// TIA Portal project "Simulate_HMI_FactoryIO_16" (V14)
// Vorlageprojekt für das Buch mit Zielsystem S7-1200

(* hardware
DEVICE "S7-1200-Station_1"  S7-1200 Station
   slot 0: "Baugruppenträger_0"  Rack  V1.0
   slot 1: "PLC_1"  CPU 1211C DC/DC/DC  6ES7 211-1AE40-0XB0  V4.1
DEVICE "HMI_1"  KTP1200 Basic PN
   slot 0: "KTP1200 Basic PN"  KTP1200 Basic PN  6AV2 123-2MB03-0AX0  14.0.1.0
   slot 1: "HMI_RT_1"  KTP1200 Basic PN  6AV2 123-2MB03-0AX0  14.0.1.0
   slot 5: "HMI_1.IE_CP_1"  PROFINET Interface  14.0.1.0
      slot 1: "PROFINET Interface_1"  PROFINET Interface
         slot 1: "Port_1"  Port
*)

// ===== PLC "PLC_1"  CPU 1211C DC/DC/DC =====

VAR_GLOBAL   // PLC tag table "Modes"
   "B_Pharmacy_ChooseRoom" AT %M0.1 : Bool;
   "B_Pharmacy_Go" AT %M0.2 : Bool;
   "B_Pharmacy_Room1" AT %MW2 : Int;
   "B_Pharmacy_Room2" AT %MW4 : Int;
   "B_Pharmacy_Room3" AT %MW6 : Int;
   "B_Pharmacy_Start" AT %M0.0 : Bool;
   "B_R1_Continue" AT %M20.2 : Bool;
   "B_R1_Return" AT %M20.3 : Bool;
   "B_R2_Continue" AT %M20.4 : Bool;
   "B_R2_Return" AT %M20.5 : Bool;
   "M_A_0_L2-L1_1" AT %M32.5 : Bool;
   "M_A_0_L2-L1_1_Trig" AT %M33.5 : Bool;
   "M_A_0_L2-L1_2" AT %M32.6 : Bool;
   "M_A_0_L2-L1_3" AT %M32.7 : Bool;
   "M_A_0_L2-L1_3_Trig" AT %M33.6 : Bool;
   "M_A_0_L2-L1_4" AT %M33.0 : Bool;
   "M_A_0_L2-L1_5" AT %M33.1 : Bool;
   "M_A_1to2_L1-L1_1" AT %M12.5 : Bool;
   "M_A_1to2_L1-L1_1_Trig" AT %M13.0 : Bool;
   "M_A_1to2_L1-L1_2" AT %M12.6 : Bool;
   "M_A_1to2_L1-L1_3" AT %M12.7 : Bool;
   "M_A_1to2_L1-L1_2_Trig" AT %M13.1 : Bool;
   "M_A_1to2_L1-L1_4" AT %M13.2 : Bool;
   "M_A_1to2_L1-L3_1" AT %M13.3 : Bool;
   "M_A_1to2_L1-L3_1_Trig" AT %M13.4 : Bool;
   "M_A_1to2_L1-L3_2" AT %M13.5 : Bool;
   "M_A_1to2_L1-L3_3" AT %M13.6 : Bool;
   "M_A_1to2_L1-L3_2_Trig" AT %M14.2 : Bool;
   "M_A_1to2_L1-L3_4" AT %M14.0 : Bool;
   "M_A_1to2_L1-L3_4_Trig" AT %M13.7 : Bool;
   "M_A_1to2_L1-L3_5" AT %M14.1 : Bool;
   "M_A_1to2_L2-L2_1" AT %M25.5 : Bool;
   "M_A_1to2_L2-L2_1_Trig" AT %M26.1 : Bool;
   "M_A_1to2_L2-L2_2" AT %M25.6 : Bool;
   "M_A_1to2_L2-L2_3" AT %M25.7 : Bool;
   "M_A_1to2_L2-L2_2_Trig" AT %M26.2 : Bool;
   "M_A_1to2_L2-L2_4" AT %M26.0 : Bool;
   "M_A_1to2_L2-L3_1" AT %M28.2 : Bool;
   "M_A_1to2_L2-L3_1_Trig" AT %M28.3 : Bool;
   "M_A_1to2_L2-L3_2" AT %M28.4 : Bool;
   "M_A_1to2_L2-L3_3" AT %M28.5 : Bool;
   "M_A_1to2_L2-L3_3_Trig" AT %M28.6 : Bool;
   "M_A_1to2_L2-L3_4" AT %M28.7 : Bool;
   "M_A_1to2_L2-L3_5" AT %M29.0 : Bool;
   "M_A_1to2_L4-L2_1" AT %M31.6 : Bool;
   "M_A_1to2_L4-L2_1_Trig" AT %M31.7 : Bool;
   "M_A_1to2_L4-L2_2" AT %M32.0 : Bool;
   "M_A_1to2_L4-L2_3" AT %M32.1 : Bool;
   "M_A_1to2_L4-L2_3_Trig" AT %M32.2 : Bool;
   "M_A_1to2_L4-L2_4" AT %M32.3 : Bool;
   "M_A_1to2_L4-L2_5" AT %M32.4 : Bool;
   "M_A_2to3_L1-L2_F1" AT %M14.3 : Bool;
   "M_A_2to3_L1-L2_F1_Trig" AT %M15.1 : Bool;
   "M_A_2to3_L1-L2_F2" AT %M14.4 : Bool;
   "M_A_2to3_L1-L2_F3" AT %M14.5 : Bool;
   "M_A_2to3_L1-L2_F2_Trig" AT %M15.2 : Bool;
   "M_A_2to3_L1-L2_F4" AT %M14.6 : Bool;
   "M_A_2to3_L2-L2_B1" AT %M24.0 : Bool;
   "M_A_2to3_L2-L2_B1_Trig" AT %M24.4 : Bool;
   "M_A_2to3_L2-L2_B2" AT %M24.1 : Bool;
   "M_A_2to3_L2-L2_B3" AT %M24.2 : Bool;
   "M_A_2to3_L2-L2_B3_Trig" AT %M24.5 : Bool;
   "M_A_2to3_L2-L2_B4" AT %M24.3 : Bool;
   "M_A_2to3_L2-L2_B5" AT %M24.6 : Bool;
   "M_A_2to4_L1-L2_F1" AT %M15.5 : Bool;
   "M_A_2to4_L1-L2_F1_Trig" AT %M15.6 : Bool;
   "M_A_2to4_L1-L2_F2" AT %M15.7 : Bool;
   "M_A_2to4_L1-L2_F3" AT %M16.0 : Bool;
   "M_A_2to4_L1-L2_F2_Trig" AT %M16.1 : Bool;
   "M_A_2to4_L1-L2_F4" AT %M16.2 : Bool;
   "M_A_2to4_L2-L2_B1" AT %M30.1 : Bool;
   "M_A_2to4_L2-L2_B1_Trig" AT %M30.2 : Bool;
   "M_A_2to4_L2-L2_B2" AT %M30.3 : Bool;
   "M_A_2to4_L2-L2_B3" AT %M30.4 : Bool;
   "M_A_2to4_L2-L2_B3_Trig" AT %M30.5 : Bool;
   "M_A_2to4_L2-L2_B4" AT %M30.6 : Bool;
   "M_A_2to4_L2-L2_B5" AT %M30.7 : Bool;
   "M_B_S0_1" AT %M27.7 : Bool;
   "M_B_S0_1_Trig" AT %M28.1 : Bool;
   "M_B_S0_2" AT %M28.0 : Bool;
   "M_B_S0_2_Trig1" AT %M33.2 : Bool;
   "M_B_S0_2_Trig2" AT %M33.3 : Bool;
   "M_B_S0_2_Trig3" AT %M33.4 : Bool;
   "M_B_S1-Cnv1_1" AT %M26.3 : Bool;
   "M_B_S1-Cnv1_1_Trig" AT %M26.4 : Bool;
   "M_B_S1-Cnv1_2" AT %M26.5 : Bool;
   "M_B_S1-Cnv1_2_Trig1" AT %M26.6 : Bool;
   "M_B_S1-Cnv1_2_Trig2" AT %M26.7 : Bool;
   "M_B_S2-1_1" AT %M24.7 : Bool;
   "M_B_S2-1_1_Trig" AT %M25.0 : Bool;
   "M_B_S2-1_2" AT %M25.1 : Bool;
   "M_B_S2-1_2_Trig1" AT %M25.2 : Bool;
   "M_B_S2-1_2_Trig2" AT %M25.3 : Bool;
   "M_B_S2-1_2_Trig3" AT %M25.4 : Bool;
   "M_B_S2-2_1" AT %M31.0 : Bool;
   "M_B_S2-2_1_Trig" AT %M31.1 : Bool;
   "M_B_S2-2_2" AT %M31.2 : Bool;
   "M_B_S2-2_2_Trig1" AT %M31.3 : Bool;
   "M_B_S2-2_2_Trig2" AT %M31.4 : Bool;
   "M_B_S2-2_2_Trig3" AT %M31.5 : Bool;
   "M_B2H_S3_1" AT %M23.2 : Bool;
   "M_B2H_S3_1_Trig" AT %M23.3 : Bool;
   "M_B2H_S3_2" AT %M23.4 : Bool;
   "M_B2H_S3_2_Trig1" AT %M23.5 : Bool;
   "M_B2H_S3_2_Trig2" AT %M23.6 : Bool;
   "M_B2H_S3_2_Trig3" AT %M23.7 : Bool;
   "M_B2H_S4_1" AT %M29.3 : Bool;
   "M_B2H_S4_1_Trig" AT %M29.4 : Bool;
   "M_B2H_S4_2" AT %M29.5 : Bool;
   "M_B2H_S4_2_Trig1" AT %M29.6 : Bool;
   "M_B2H_S4_2_Trig2" AT %M29.7 : Bool;
   "M_B2H_S4_2_Trig3" AT %M30.0 : Bool;
   "M_B2L_S3_1" AT %M20.6 : Bool;
   "M_B2L_S3_2" AT %M20.7 : Bool;
   "M_B2L_S3_2_Trig1" AT %M21.2 : Bool;
   "M_B2L_S3_2_Trig2" AT %M21.3 : Bool;
   "M_B2L_S4_1" AT %M21.0 : Bool;
   "M_B2L_S4_2" AT %M21.1 : Bool;
   "M_B2L_S4_2_Trig1" AT %M29.1 : Bool;
   "M_B2L_S4_2_Trig2" AT %M29.2 : Bool;
   "M_F_S0_1" AT %M1.1 : Bool;
   "M_F_S0_1_Trig" AT %M1.2 : Bool;
   "M_F_S0_2" AT %M1.3 : Bool;
   "M_F_S0_2_Trig1" AT %M1.4 : Bool;
   "M_F_S0_2_Trig2" AT %M8.0 : Bool;
   "M_F_S1_1" AT %M1.5 : Bool;
   "M_F_S1_1_Trig" AT %M1.6 : Bool;
   "M_F_S1_2" AT %M1.7 : Bool;
   "M_F_S1-Cnv1_2_Trig1" AT %M10.0 : Bool;
   "M_F_S1-Cnv1_2_Trig2" AT %M12.3 : Bool;
   "M_F_S1_2_Trig3" AT %M12.4 : Bool;
   "M_F_S2-1_1" AT %M10.1 : Bool;
   "M_F_S2-1_1_Trig" AT %M10.2 : Bool;
   "M_F_S2-1_2" AT %M10.3 : Bool;
   "M_F_S2-1_2_Trig1" AT %M10.4 : Bool;
   "M_F_S2-1_2_Trig2" AT %M14.7 : Bool;
   "M_F_S2-1_2_Trig3" AT %M15.0 : Bool;
   "M_F_S2-2_1" AT %M10.5 : Bool;
   "M_F_S2-2_1_Trig" AT %M10.6 : Bool;
   "M_F_S2-2_2" AT %M10.7 : Bool;
   "M_F_S2-2_2_Trig1" AT %M11.0 : Bool;
   "M_F_S2-2_2_Trig2" AT %M15.3 : Bool;
   "M_F_S2-2_2_Trig3" AT %M15.4 : Bool;
   "M_F2H_S3_1" AT %M8.1 : Bool;
   "M_F2H_S3_1_Trig" AT %M8.2 : Bool;
   "M_F2H_S3_2" AT %M8.3 : Bool;
   "M_F2H_S3_2_Trig1" AT %M8.4 : Bool;
   "M_F2H_S3_2_Trig2" AT %M8.5 : Bool;
   "M_F2H_S3_2_Trig3" AT %M8.6 : Bool;
   "M_F2H_S4_1" AT %M8.7 : Bool;
   "M_F2H_S4_1_Trig" AT %M9.0 : Bool;
   "M_F2H_S4_2" AT %M9.1 : Bool;
   "M_F2H_S4_2_Trig1" AT %M9.2 : Bool;
   "M_F2H_S4_2_Trig2" AT %M9.3 : Bool;
   "M_F2H_S4_2_Trig3" AT %M9.4 : Bool;
   "M_F2L_S3_1" AT %M9.5 : Bool;
   "M_F2L_S3_1_Trig" AT %M9.6 : Bool;
   "M_F2L_S3_2" AT %M9.7 : Bool;
   "M_F2L_S3_2_Trig" AT %M18.6 : Bool;
   "M_F2L_S4_1" AT %M19.6 : Bool;
   "M_F2L_S4_1_Trig" AT %M19.7 : Bool;
   "M_F2L_S4_2" AT %M20.0 : Bool;
   "M_F2L_S4_2_Trig" AT %M20.1 : Bool;
   "M_Pharmacy_ChooseRoom" AT %M0.6 : Bool;
   "M_Pharmacy_Go" AT %M0.7 : Bool;
   "M_Pharmacy_Go_Trig" AT %M1.0 : Bool;
   "M_Pharmacy_Start" AT %M0.4 : Bool;
   "M_Pharmacy_Start_Trig" AT %M0.5 : Bool;
   "M_Pharmacy_Wait" AT %M0.3 : Bool;
   "M_R1_ChooseRoom" AT %M17.2 : Bool;
   "M_R1_Go" AT %M17.3 : Bool;
   "M_R1_Go_Trig" AT %M17.4 : Bool;
   "M_R1_Start" AT %M17.5 : Bool;
   "M_R1_Start_Trig" AT %M17.6 : Bool;
   "M_R1_Wait" AT %M17.7 : Bool;
   "M_R2_ChooseRoom" AT %M18.0 : Bool;
   "M_R2_Go" AT %M18.1 : Bool;
   "M_R2_Go_Trig" AT %M18.2 : Bool;
   "M_R2_Start" AT %M18.3 : Bool;
   "M_R2_Start_Trig" AT %M18.4 : Bool;
   "M_R2_Wait" AT %M18.5 : Bool;
   "M_UD_0to1_B_1" AT %M27.0 : Bool;
   "M_UD_0to1_B_1_Trig" AT %M27.5 : Bool;
   "M_UD_0to1_B_2" AT %M27.1 : Bool;
   "M_UD_0to1_B_3" AT %M27.2 : Bool;
   "M_UD_0to1_B_3_Trig" AT %M27.6 : Bool;
   "M_UD_0to1_B_4" AT %M27.3 : Bool;
   "M_UD_0to1_B_5" AT %M27.4 : Bool;
   "M_UD_0to1_F_1" AT %M11.1 : Bool;
   "M_UD_0to1_F_1_Trig" AT %M11.2 : Bool;
   "M_UD_0to1_F_2" AT %M11.3 : Bool;
   "M_UD_0to1_F_2_Trig" AT %M11.4 : Bool;
   "M_UD_0to1_F_3" AT %M11.5 : Bool;
   "M_UD_0to1_F_3_Trig" AT %M11.6 : Bool;
   "M_UD_0to1_F_4" AT %M11.7 : Bool;
   "M_UD_0to1_F_4_Trig" AT %M12.0 : Bool;
   "M_UD_0to1_F_5" AT %M12.1 : Bool;
   "M_UD_3_B_1" AT %M21.4 : Bool;
   "M_UD_3_B_1_Trig" AT %M21.5 : Bool;
   "M_UD_3_B_2" AT %M21.6 : Bool;
   "M_UD_3_B_3" AT %M21.7 : Bool;
   "M_UD_3_B_3_Trig" AT %M22.0 : Bool;
   "M_UD_3_B_4" AT %M22.1 : Bool;
   "M_UD_3_B_5" AT %M22.2 : Bool;
   "M_UD_3_F_1" AT %M16.3 : Bool;
   "M_UD_3_F_1_Trig" AT %M17.0 : Bool;
   "M_UD_3_F_2" AT %M16.4 : Bool;
   "M_UD_3_F_3" AT %M16.5 : Bool;
   "M_UD_3_F_3_Trig" AT %M17.1 : Bool;
   "M_UD_3_F_4" AT %M16.6 : Bool;
   "M_UD_3_F_5" AT %M16.7 : Bool;
   "M_UD_4_B_1" AT %M22.3 : Bool;
   "M_UD_4_B_1_Trig" AT %M22.4 : Bool;
   "M_UD_4_B_2" AT %M22.5 : Bool;
   "M_UD_4_B_3" AT %M22.6 : Bool;
   "M_UD_4_B_3_Trig" AT %M22.7 : Bool;
   "M_UD_4_B_4" AT %M23.0 : Bool;
   "M_UD_4_B_5" AT %M23.1 : Bool;
   "M_UD_4_F_1" AT %M18.7 : Bool;
   "M_UD_4_F_1_Trig" AT %M19.0 : Bool;
   "M_UD_4_F_2" AT %M19.1 : Bool;
   "M_UD_4_F_3" AT %M19.2 : Bool;
   "M_UD_4_F_3_Trig" AT %M19.3 : Bool;
   "M_UD_4_F_4" AT %M19.4 : Bool;
   "M_UD_4_F_5" AT %M19.5 : Bool;
   "M_Elevator1_Trig1" AT %M33.7 : Bool;
   "M_UD_0to1_F_6" AT %M34.0 : Bool;
   "M_UD_3_F_6" AT %M34.1 : Bool;
   "M_UD_0to1_F_7" AT %M34.2 : Bool;
   "M_UD_3_F_7" AT %M34.3 : Bool;
   "M_Elevator3_Trig1" AT %M34.4 : Bool;
   "M_Elevator4_Trig1" AT %M34.5 : Bool;
   "M_UD_4_F_6" AT %M34.6 : Bool;
   "M_UD_4_F_7" AT %M34.7 : Bool;
   "M_Elevator3_Trig2" AT %M35.0 : Bool;
   "M_UD_3_B_6" AT %M35.1 : Bool;
   "M_UD_3_B_7" AT %M35.2 : Bool;
   "M_Elevator4_Trig2" AT %M35.3 : Bool;
   "M_UD_4_B_6" AT %M35.4 : Bool;
   "M_UD_4_B_7" AT %M35.5 : Bool;
   "M_B_S1-Cnv2_1" AT %M35.6 : Bool;
   "M_B_S1-Cnv2_1_Trig1" AT %M35.7 : Bool;
   "M_B_S1-Cnv2_2" AT %M36.0 : Bool;
   "M_B_S1-Cnv2_2_Trig1" AT %M36.1 : Bool;
   "M_B_S1-Cnv2_1_Trig2" AT %M36.2 : Bool;
   "M_B_S1-Cnv2_3" AT %M36.3 : Bool;
   "M_B_S1-Cnv2_3_Trig1" AT %M36.4 : Bool;
   "M_B_S1-Cnv2_3_Trig2" AT %M36.5 : Bool;
   "M_UD_0to1_B_6" AT %M36.6 : Bool;
   "M_UD_0to1_B_7" AT %M36.7 : Bool;
   "M_Elevator2_Trig1" AT %M37.0 : Bool;
   "M_A_0_L2-L1_2_Trig1" AT %M37.1 : Bool;
   "M_A_0_L2-L1_Trig" AT %M37.2 : Bool;
   "M_A_0_L2-L1_2_Trig2" AT %M37.3 : Bool;
   "F_0_1_1_Stt" AT %MW100 : Int;
   "F_1_1_1_Stt" AT %MW102 : Int;
   "F_2_1_1_Stt" AT %MW104 : Int;
   "F_2_2_1_Stt" AT %MW106 : Int;
   "B_0_1_1_Stt" AT %MW108 : Int;
   "B_1_1_1_Stt" AT %MW110 : Int;
   "B_2_1_1_Stt" AT %MW112 : Int;
   "B_2_2_1_Stt" AT %MW114 : Int;
   "2d_3_H_Stt" AT %MW116 : Int;
   "2d_3_H_Dir" AT %MW118 : Int;
   "2d_3_L_Stt" AT %MW120 : Int;
   "2d_3_L_Dir" AT %MW122 : Int;
   "2d_4_H_Stt" AT %MW124 : Int;
   "2d_4_H_Dir" AT %MW126 : Int;
   "2d_4_L_Stt" AT %MW128 : Int;
   "2d_4_L_Dir" AT %MW130 : Int;
   "av2_0to0_Stt" AT %MW132 : Int;
   "av2_0to0_Dir" AT %MW134 : Int;
   "av4_1to2_Stt" AT %MW136 : Word;
   "av4_1to2_Dir" AT %MW138 : Word;
   "av2_2to3_Stt" AT %MW140 : Int;
   "av2_2to3_Dir" AT %MW142 : Int;
   "av2_2to4_Stt" AT %MW144 : Int;
   "av2_2to4_Dir" AT %MW146 : Int;
   "ud_0to1_1_Stt" AT %MW148 : Int;
   "ud_0to1_1_Dir" AT %MW150 : Int;
   "ud_0to1_2_Stt" AT %MW152 : Int;
   "ud_0to1_2_Dir" AT %MW154 : Int;
   "ud_3_Stt" AT %MW156 : Int;
   "ud_3_Dir" AT %MW158 : Int;
   "ud_4_Stt" AT %MW160 : Int;
   "ud_4_Dir" AT %MW162 : Int;
   "av2_0to0_LS1" AT %M300.0 : Bool;
   "av2_0to0_LS2" AT %M300.1 : Bool;
   "av4_1to2_LS1" AT %M300.2 : Bool;
   "av4_1to2_LS2" AT %M300.3 : Bool;
   "av4_1to2_LS3" AT %M300.4 : Bool;
   "av4_1to2_LS4" AT %M300.5 : Bool;
   "av2_2to3_LS1" AT %M300.6 : Bool;
   "av2_2to3_LS2" AT %M300.7 : Bool;
   "av2_2to4_LS1" AT %M301.0 : Bool;
   "av2_2to4_LS2" AT %M301.1 : Bool;
   "ud_0to1_f_ls_H" AT %M301.2 : Bool;
   "ud_0to1_f_ls_L" AT %M301.3 : Bool;
   "ud_3_ls_H" AT %M301.6 : Bool;
   "ud_3_ls_L" AT %M301.7 : Bool;
   "ud_4_ls_H" AT %M302.0 : Bool;
   "ud_4_ls_L" AT %M302.1 : Bool;
   "ud_0to1_b_ls_H" AT %M301.4 : Bool;
   "ud_0to1_b_ls_L" AT %M301.5 : Bool;
   "M_B_S1-Cnv2_3_Trig3" AT %M37.4 : Bool;
   "box1_f_0_1_1" AT %MW164 : Int;
   "box2_f_0_1_1" AT %MW166 : Word;
   "box3_f_0_1_1" AT %MW168 : Word;
   "box1_f_1_1_1" AT %MW170 : Word;
   "box2_f_1_1_1" AT %MW172 : Word;
   "box3_f_1_1_1" AT %MW174 : Word;
   "box1_f_2_1_1" AT %MW176 : Word;
   "box2_f_2_1_1" AT %MW178 : Word;
   "box3_f_2_1_1" AT %MW180 : Word;
   "box1_f_2_2_1" AT %MW182 : Word;
   "box2_f_2_2_1" AT %MW184 : Word;
   "box3_f_2_2_1" AT %MW186 : Word;
   "box1_b_0_1_1" AT %MW188 : Word;
   "box2_b_0_1_1" AT %MW190 : Word;
   "box3_b_0_1_1" AT %MW192 : Word;
   "box1_b_1_1_1" AT %MW194 : Word;
   "box2_b_1_1_1" AT %MW196 : Word;
   "box3_b_1_1_1" AT %MW198 : Word;
   "box1_b_2_1_1" AT %MW200 : Word;
   "box2_b_2_1_1" AT %MW202 : Word;
   "box3_b_2_1_1" AT %MW204 : Word;
   "box1_b_2_2_1" AT %MW206 : Word;
   "box2_b_2_2_1" AT %MW208 : Word;
   "box3_b_2_2_1" AT %MW210 : Word;
   "box_av2_0to0" AT %MW212 : Word;
   "box_av4_1to2" AT %MW214 : Word;
   "box_av2_2to3" AT %MW216 : Word;
   "box_av2_2to4" AT %MW218 : Word;
   "box_ud2_0to1_f" AT %MW220 : Word;
   "box_ud2_0to1_b" AT %MW222 : Word;
   "box_ud_3" AT %MW224 : Word;
   "box_ud_4" AT %MW226 : Word;
   "box1_2d_3h" AT %MW228 : Word;
   "box2_2d_3h" AT %MW230 : Word;
   "box3_2d_3h" AT %MW232 : Word;
   "box1_2d_3l" AT %MW234 : Word;
   "box2_2d_3l" AT %MW236 : Word;
   "box3_2d_3l" AT %MW238 : Word;
   "box1_2d_4h" AT %MW240 : Word;
   "box2_2d_4h" AT %MW242 : Word;
   "box3_2d_4h" AT %MW244 : Word;
   "box1_2d_4l" AT %MW246 : Word;
   "box2_2d_4l" AT %MW248 : Word;
   "box3_2d_4l" AT %MW250 : Word;
   "M_R1_Cont_Trig" AT %M37.5 : Bool;
   "M_R1_Return_Trig" AT %M37.6 : Bool;
   "M_R2_Cont_Trig" AT %M37.7 : Bool;
   "M_R2_Return_Trig" AT %M38.0 : Bool;
   "M_A_1to2_L4-L1_1" AT %M38.1 : Bool;
   "M_A_1to2_L4-L1_1_Trig" AT %M38.2 : Bool;
   "M_A_1to2_L4-L1_2" AT %M38.3 : Bool;
   "M_A_1to2_L4-L1_3" AT %M38.4 : Bool;
   "M_A_1to2_L4-L1_3_Trig" AT %M38.5 : Bool;
   "M_A_1to2_L4-L1_4" AT %M38.6 : Bool;
   "M_A_1to2_L4-L1_5" AT %M38.7 : Bool;
   "box1_des1" AT %MW252 : Word;
   "box1_des2" AT %MW254 : Word;
   "box1_des3" AT %MW256 : Word;
   "box2_des1" AT %MW258 : Word;
   "box2_des2" AT %MW260 : Word;
   "box2_des3" AT %MW262 : Word;
   "box3_des1" AT %MW264 : Word;
   "box3_des2" AT %MW266 : Word;
   "box3_des3" AT %MW268 : Word;
   "box4_des1" AT %MW270 : Word;
   "box4_des2" AT %MW272 : Word;
   "box4_des3" AT %MW274 : Word;
   "box5_des1" AT %MW276 : Word;
   "box5_des2" AT %MW278 : Word;
   "box5_des3" AT %MW280 : Word;
   "Tag_1" AT %M500.0 : Bool;
   "R1_has_box" AT %M39.0 : Bool;
   "R2_has_box" AT %M39.1 : Bool;
END_VAR

VAR_GLOBAL   // PLC tag table "Hardware Input"
   "Elevator1_SS_Back" AT %I0.0 : Bool;
   "Elevator1_SS_Front" AT %I0.1 : Bool;
   "Elevator2_SS_Back" AT %I0.2 : Bool;
   "Elevator2_SS_Front" AT %I0.3 : Bool;
   "Elevator3_SS_Back" AT %I0.4 : Bool;
   "Elevator3_SS_Front" AT %I0.5 : Bool;
   "Elevator4_SS_Back" AT %I0.6 : Bool;
   "Elevator4_SS_Front" AT %I0.7 : Bool;
   "Cnv2_S3_H_VS1_Bool0" AT %I1.0 : Bool;
   "Cnv2_S3_H_VS1_Bool1" AT %I1.1 : Bool;
   "Cnv2_S3_H_VS1_Bool2" AT %I1.2 : Bool;
   "Cnv2_S3_H_VS2_Bool0" AT %I1.3 : Bool;
   "Cnv2_S3_H_VS2_Bool1" AT %I1.4 : Bool;
   "Cnv2_S3_H_VS2_Bool2" AT %I1.5 : Bool;
   "Cnv2_S3_L_VS1_Bool0" AT %I1.6 : Bool;
   "Cnv2_S3_L_VS1_Bool1" AT %I1.7 : Bool;
   "Cnv2_S3_L_VS1_Bool2" AT %I2.0 : Bool;
   "Cnv2_S3_L_VS2_Bool0" AT %I2.1 : Bool;
   "Cnv2_S3_L_VS2_Bool1" AT %I2.2 : Bool;
   "Cnv2_S3_L_VS2_Bool2" AT %I2.3 : Bool;
   "Cnv2_S4_H_VS1_Bool0" AT %I2.4 : Bool;
   "Cnv2_S4_H_VS1_Bool1" AT %I2.5 : Bool;
   "Cnv2_S4_H_VS1_Bool2" AT %I2.6 : Bool;
   "Cnv2_S4_H_VS2_Bool0" AT %I2.7 : Bool;
   "Cnv2_S4_H_VS2_Bool1" AT %I3.0 : Bool;
   "Cnv2_S4_H_VS2_Bool2" AT %I3.1 : Bool;
   "Cnv2_S4_L_VS1_Bool0" AT %I3.2 : Bool;
   "Cnv2_S4_L_VS1_Bool1" AT %I3.3 : Bool;
   "Cnv2_S4_L_VS1_Bool2" AT %I3.4 : Bool;
   "Cnv2_S4_L_VS2_Bool0" AT %I3.5 : Bool;
   "Cnv2_S4_L_VS2_Bool1" AT %I3.6 : Bool;
   "Cnv2_S4_L_VS2_Bool2" AT %I3.7 : Bool;
   "CnvB_S0_VS1_Bool0" AT %I4.0 : Bool;
   "CnvB_S0_VS1_Bool1" AT %I4.1 : Bool;
   "CnvB_S0_VS1_Bool2" AT %I4.2 : Bool;
   "CnvB_S0_VS2_Bool0" AT %I4.3 : Bool;
   "CnvB_S0_VS2_Bool1" AT %I4.4 : Bool;
   "CnvB_S0_VS2_Bool2" AT %I4.5 : Bool;
   "CnvB_S1_VS1_Bool0" AT %I4.6 : Bool;
   "CnvB_S1_VS1_Bool1" AT %I4.7 : Bool;
   "CnvB_S1_VS1_Bool2" AT %I5.0 : Bool;
   "CnvB_S1_VS2_Bool0" AT %I5.1 : Bool;
   "CnvB_S1_VS2_Bool1" AT %I5.2 : Bool;
   "CnvB_S1_VS2_Bool2" AT %I5.3 : Bool;
   "CnvB_S2-1_VS1_Bool0" AT %I5.4 : Bool;
   "CnvB_S2-1_VS1_Bool1" AT %I5.5 : Bool;
   "CnvB_S2-1_VS1_Bool2" AT %I5.6 : Bool;
   "CnvB_S2-1_VS2_Bool0" AT %I5.7 : Bool;
   "CnvB_S2-1_VS2_Bool1" AT %I6.0 : Bool;
   "CnvB_S2-1_VS2_Bool2" AT %I6.1 : Bool;
   "CnvB_S2-2_VS1_Bool0" AT %I6.2 : Bool;
   "CnvB_S2-2_VS1_Bool1" AT %I6.3 : Bool;
   "CnvB_S2-2_VS1_Bool2" AT %I6.4 : Bool;
   "CnvB_S2-2_VS2_Bool0" AT %I6.5 : Bool;
   "CnvB_S2-2_VS2_Bool1" AT %I6.6 : Bool;
   "CnvB_S2-2_VS2_Bool2" AT %I6.7 : Bool;
   "CnvF_S0_VS1_Bool0" AT %I7.0 : Bool;
   "CnvF_S0_VS1_Bool1" AT %I7.1 : Bool;
   "CnvF_S0_VS1_Bool2" AT %I7.2 : Bool;
   "CnvF_S0_VS2_Bool0" AT %I7.3 : Bool;
   "CnvF_S0_VS2_Bool1" AT %I7.4 : Bool;
   "CnvF_S0_VS2_Bool2" AT %I7.5 : Bool;
   "CnvF_S1_VS1_Bool0" AT %I7.6 : Bool;
   "CnvF_S1_VS1_Bool1" AT %I7.7 : Bool;
   "CnvF_S1_VS1_Bool2" AT %I8.0 : Bool;
   "CnvF_S1_VS2_Bool0" AT %I8.1 : Bool;
   "CnvF_S1_VS2_Bool1" AT %I8.2 : Bool;
   "CnvF_S1_VS2_Bool2" AT %I8.3 : Bool;
   "CnvF_S2-1_VS1_Bool0" AT %I8.4 : Bool;
   "CnvF_S2-1_VS1_Bool1" AT %I8.5 : Bool;
   "CnvF_S2-1_VS1_Bool2" AT %I8.6 : Bool;
   "CnvF_S2-1_VS2_Bool0" AT %I8.7 : Bool;
   "CnvF_S2-1_VS2_Bool1" AT %I9.0 : Bool;
   "CnvF_S2-1_VS2_Bool2" AT %I9.1 : Bool;
   "CnvF_S2-2_VS1_Bool0" AT %I9.2 : Bool;
   "CnvF_S2-2_VS1_Bool1" AT %I9.3 : Bool;
   "CnvF_S2-2_VS1_Bool2" AT %I9.4 : Bool;
   "CnvF_S2-2_VS2_Bool0" AT %I9.5 : Bool;
   "CnvF_S2-2_VS2_Bool1" AT %I9.6 : Bool;
   "CnvF_S2-2_VS2_Bool2" AT %I9.7 : Bool;
   "Srt_3_SS1" AT %I10.0 : Bool;
   "Srt_3_SS2" AT %I10.1 : Bool;
   "Srt_4_SS1" AT %I10.2 : Bool;
   "Srt_4_SS2" AT %I10.3 : Bool;
   "Srt_1to2_SS1" AT %I10.4 : Bool;
   "Srt_1to2_SS2" AT %I10.5 : Bool;
   "Srt_1to2_SS3" AT %I10.6 : Bool;
   "Srt_1to2_SS4" AT %I10.7 : Bool;
   "CnvB_Srt1_SS" AT %I11.0 : Bool;
   "CnvB_Srt2_SS" AT %I11.1 : Bool;
   "Srt_0_SS1" AT %I11.2 : Bool;
   "Srt_0_SS2" AT %I11.3 : Bool;
   "Elevator1_ssH1" AT %I11.4 : Bool;
   "Elevator1_ssH2" AT %I11.5 : Bool;
   "Elevator1_ssL" AT %I11.6 : Bool;
   "Elevator2_ssH1" AT %I11.7 : Bool;
   "Elevator2_ssH2" AT %I12.0 : Bool;
   "Elevator2_ssL" AT %I12.1 : Bool;
   "Elevator3_ssH1" AT %I12.2 : Bool;
   "Elevator3_ssH2" AT %I12.3 : Bool;
   "Elevator3_ssL" AT %I12.4 : Bool;
   "Elevator4_ssH1" AT %I12.5 : Bool;
   "Elevator4_ssH2" AT %I12.6 : Bool;
   "Elevator4_ssL" AT %I12.7 : Bool;
END_VAR

VAR_GLOBAL   // PLC tag table "Hardware Output"
   "Elevator1_F" AT %Q0.0 : Bool;
   "Elevator1_B" AT %Q0.1 : Bool;
   "Elevator2_F" AT %Q0.2 : Bool;
   "Elevator2_B" AT %Q0.3 : Bool;
   "Elevator3_F" AT %Q0.4 : Bool;
   "Elevator3_B" AT %Q0.5 : Bool;
   "Elevator4_F" AT %Q0.6 : Bool;
   "Elevator4_B" AT %Q0.7 : Bool;
   "Elevator1_U" AT %Q1.0 : Bool;
   "Elevator1_D" AT %Q1.1 : Bool;
   "Elevator1_Slow" AT %Q1.2 : Bool;
   "Elevator2_U" AT %Q1.3 : Bool;
   "Elevator2_D" AT %Q1.4 : Bool;
   "Elevator2_Slow" AT %Q1.5 : Bool;
   "Elevator3_U" AT %Q1.6 : Bool;
   "Elevator3_D" AT %Q1.7 : Bool;
   "Elevator3_Slow" AT %Q2.0 : Bool;
   "Elevator4_U" AT %Q2.1 : Bool;
   "Elevator4_D" AT %Q2.2 : Bool;
   "Elevator4_Slow" AT %Q2.3 : Bool;
   "Cnv2_S4_H_B" AT %Q2.4 : Bool;
   "Cnv2_S4_H_F" AT %Q2.5 : Bool;
   "Cnv2_S3_H_B" AT %Q2.6 : Bool;
   "Cnv2_S3_H_F" AT %Q2.7 : Bool;
   "Cnv2_S3_L_B" AT %Q3.0 : Bool;
   "Cnv2_S3_L_F" AT %Q3.1 : Bool;
   "Cnv2_S4_L_B" AT %Q3.2 : Bool;
   "Cnv2_S4_L_F" AT %Q3.3 : Bool;
   "CnvB_S0" AT %Q3.4 : Bool;
   "CnvB_S1_1" AT %Q3.5 : Bool;
   "CnvB_S1_2" AT %Q3.6 : Bool;
   "CnvB_S2-1" AT %Q4.2 : Bool;
   "CnvB_S2-2" AT %Q4.3 : Bool;
   "CnvF_S0" AT %Q4.4 : Bool;
   "CnvF_S1_1" AT %Q4.5 : Bool;
   "CnvF_S1_2" AT %Q4.6 : Bool;
   "CnvF_S2-1" AT %Q5.0 : Bool;
   "CnvF_S2-2" AT %Q5.1 : Bool;
   "CnvF_S1_Srt" AT %Q5.2 : Bool;
   "Srt_3_B1" AT %Q5.3 : Bool;
   "Srt_3_B2" AT %Q5.4 : Bool;
   "Srt_3_F1" AT %Q5.5 : Bool;
   "Srt_3_F2" AT %Q5.6 : Bool;
   "Srt_3_L1" AT %Q5.7 : Bool;
   "Srt_3_L2" AT %Q6.0 : Bool;
   "Srt_3_R1" AT %Q6.1 : Bool;
   "Srt_3_R2" AT %Q6.2 : Bool;
   "Srt_4_B1" AT %Q6.3 : Bool;
   "Srt_4_B2" AT %Q6.4 : Bool;
   "Srt_4_F1" AT %Q6.5 : Bool;
   "Srt_4_F2" AT %Q6.6 : Bool;
   "Srt_4_L1" AT %Q6.7 : Bool;
   "Srt_4_L2" AT %Q7.0 : Bool;
   "Srt_4_R1" AT %Q7.1 : Bool;
   "Srt_4_R2" AT %Q7.2 : Bool;
   "Srt_1to2_B1" AT %Q7.3 : Bool;
   "Srt_1to2_B2" AT %Q7.4 : Bool;
   "Srt_1to2_B3" AT %Q7.5 : Bool;
   "Srt_1to2_B4" AT %Q7.6 : Bool;
   "Srt_1to2_F1" AT %Q7.7 : Bool;
   "Srt_1to2_F2" AT %Q8.0 : Bool;
   "Srt_1to2_F3" AT %Q8.1 : Bool;
   "Srt_1to2_F4" AT %Q8.2 : Bool;
   "Srt_1to2_L1" AT %Q8.3 : Bool;
   "Srt_1to2_L2" AT %Q8.4 : Bool;
   "Srt_1to2_L3" AT %Q8.5 : Bool;
   "Srt_1to2_L4" AT %Q8.6 : Bool;
   "Srt_1to2_R1" AT %Q8.7 : Bool;
   "Srt_1to2_R2" AT %Q9.0 : Bool;
   "Srt_1to2_R3" AT %Q9.1 : Bool;
   "Srt_1to2_R4" AT %Q9.2 : Bool;
   "Srt_0_F1" AT %Q9.3 : Bool;
   "Srt_0_L1" AT %Q9.4 : Bool;
   "Srt_0_R1" AT %Q9.5 : Bool;
   "Srt_0_B2" AT %Q9.6 : Bool;
   "Srt_0_L2" AT %Q9.7 : Bool;
   "Srt_0_R2" AT %Q10.0 : Bool;
   "Srt_0_Connect" AT %Q10.1 : Bool;
   "CnvB_S1_3" AT %Q3.7 : Bool;
   "CnvB_S1_4" AT %Q4.0 : Bool;
   "CnvB_S1_5" AT %Q4.1 : Bool;
   "CnvF_S1_4" AT %Q10.2 : Bool;
   "CnvF_S1_3" AT %Q4.7 : Bool;
END_VAR

TYPE "Box"
   STRUCT
      V_Destination : Array[1..3] of DInt;
      V_Completed : Array[1..3] of DInt;
      V_SentFrom : DInt;
      V_NumOfDes : DInt;
      V_SectionOn : DInt;
      V_ConveyorOn : DInt;
      V_TypeOn : Byte;
      V_Direction : Byte;
      V_NumOfComp : DInt;
   END_STRUCT;
END_TYPE

TYPE "Cnv2d"
   STRUCT
      I_RFID_1 : DInt;
      I_RFID_2 : DInt;
      O_Motor_F : Bool;
      O_Motor_B : Bool;
      V_Busy : DInt;
      V_ArrayOfBox : Array[1..3] of DInt;
      V_NumOfBox : DInt;
      V_BoxOut : DInt;
   END_STRUCT;
END_TYPE

TYPE "Avoidance4"
   STRUCT
      Srt : Array[1..4] of "Sorter";
      V_BoxQueue : Array[1..3] of DInt;
      V_BoxID : DInt;
      V_Busy : DInt;
      V_NumOfBoxWaiting : DInt;
      V_BoxOut : DInt;
   END_STRUCT;
END_TYPE

TYPE "UpDown2"
   STRUCT
      I_SS_F_1 : Bool;
      I_SS_F_2 : Bool;
      I_SS_B_1 : Bool;
      I_SS_B_2 : Bool;
      I_SS_FH1 : Bool;
      I_SS_FH2 : Bool;
      I_SS_FL : Bool;
      I_SS_BH1 : Bool;
      I_SS_BH2 : Bool;
      I_SS_BL : Bool;
      O_Motor_FU : Bool;
      O_Motor_FD : Bool;
      O_Motor_BU : Bool;
      O_Motor_BD : Bool;
      O_Motor_FU_Slow : Bool;
      O_Motor_BU_Slow : Bool;
      O_Motor_F : Bool;
      O_Motor_B : Bool;
      V_BoxID_F : DInt;
      V_BoxID_B : DInt;
      V_Busy_F : DInt;
      V_Busy_B : DInt;
      V_Waiting_F : Bool;
      V_Waiting_B : Bool;
   END_STRUCT;
END_TYPE

TYPE "Sorter"
   STRUCT
      I_SS : Bool;
      O_Motor_F : Bool;
      O_Motor_B : Bool;
      O_Motor_L : Bool;
      O_Motor_R : Bool;
      V_Busy : Byte;
      V_BoxID : Byte;
   END_STRUCT;
END_TYPE

TYPE "Avoidance2"
   STRUCT
      Srt : Array[1..2] of "Sorter";
      V_BoxQueue : Array[1..3] of DInt;
      V_BoxID : DInt;
      V_Busy : DInt;
      V_NumOfBoxWaiting : DInt;
      V_BoxOut : DInt;
   END_STRUCT;
END_TYPE

TYPE "UpDown1"
   STRUCT
      I_SS_Front : Bool;
      I_SS_Back : Bool;
      I_SS_H1 : Bool;
      I_SS_H2 : Bool;
      I_SS_L : Bool;
      O_Motor_U : Bool;
      O_Motor_D : Bool;
      O_Motor_Slow : Bool;
      O_Motor_F : Bool;
      O_Motor_B : Bool;
      V_BoxID : DInt;
      V_Busy : DInt;
      V_Waiting_F : Bool;
      V_Waiting_B : Bool;
   END_STRUCT;
END_TYPE

TYPE "Cnv1d"
   STRUCT
      I_RFID_1 : DInt;
      I_RFID_2 : DInt;
      O_Motor : Bool;
      V_Busy : DInt;
      V_NumOfBox : DInt;
      V_BoxOut : DInt;
      V_ArrayBox : Array[1..3] of DInt;
   END_STRUCT;
END_TYPE

DATA_BLOCK "Boxes"   // DB1
{ S7_Optimized_Access := 'TRUE' }
VERSION : 0.1
   VAR
      Boxes : Array[1..5] of "Box";
   END_VAR
BEGIN
END_DATA_BLOCK

DATA_BLOCK "CnvF"   // DB2
{ S7_Optimized_Access := 'TRUE' }
VERSION : 0.1
   VAR
      Sect0 : "Cnv1d";
      Sect1 : Struct
         Cnv1 : "Cnv1d";
         Cnv2 : "Cnv1d";
         Cnv3 : "Cnv1d";
         Cnv4 : "Cnv1d";
         V_ArrayBox : Array[1..3] of DInt;
         V_BoxOut : DInt;
         V_NumOfBox : DInt;
         V_Busy : DInt;
      END_STRUCT;
      Sect2_1 : "Cnv1d";
      Sect2_2 : "Cnv1d";
   END_VAR
BEGIN
END_DATA_BLOCK

DATA_BLOCK "Cnv2"   // DB3
{ S7_Optimized_Access := 'TRUE' }
VERSION : 0.1
   VAR
      Sect3 : Struct
         H : "Cnv2d";
         L : "Cnv2d";
         Direction : Byte;
      END_STRUCT;
      Sect4 : Struct
         H : "Cnv2d";
         L : "Cnv2d";
         Direction : Byte;
      END_STRUCT;
   END_VAR
BEGIN
END_DATA_BLOCK

DATA_BLOCK "Avoid"   // DB4
{ S7_Optimized_Access := 'TRUE' }
VERSION : 0.1
   VAR
      Av_0 : Struct
         Av : "Avoidance2";
         Cnv_motor : Bool;
      END_STRUCT;
      Av_1to2 : "Avoidance4";
      Av_2to3 : "Avoidance2";
      Av_2to4 : "Avoidance2";
   END_VAR
BEGIN
END_DATA_BLOCK

DATA_BLOCK "UpDown"   // DB5
{ S7_Optimized_Access := 'TRUE' }
VERSION : 0.1
   VAR
      UD_0to1 : "UpDown2";
      UD_3 : "UpDown1";
      UD_4 : "UpDown1";
   END_VAR
BEGIN
   UD_0to1.I_SS_FL := 1;
   UD_0to1.I_SS_BL := 1;
   UD_3.I_SS_L := 1;
   UD_4.I_SS_L := 1;
END_DATA_BLOCK

DATA_BLOCK "CnvB"   // DB6
{ S7_Optimized_Access := 'TRUE' }
VERSION : 0.1
   VAR
      Sect0 : "Cnv1d";
      Sect1 : Struct
         Cnv1 : "Cnv1d";
         Cnv2 : "Cnv1d";
         Cnv3 : "Cnv1d";
         Cnv4 : "Cnv1d";
         Cnv5 : "Cnv1d";
         V_Busy : DInt;
         V_NumOfBox : DInt;
         V_BoxOut : DInt;
         V_ArrayOfBox : Array[1..3] of DInt;
      END_STRUCT;
      Sect2_1 : "Cnv1d";
      Sect2_2 : "Cnv1d";
   END_VAR
BEGIN
END_DATA_BLOCK

FUNCTION "Enqueue3" : Void   // FC1, SCL
{ S7_Optimized_Access := 'TRUE' }
VERSION : 0.1
   VAR_IN_OUT
      "Array" : Array[1..3] of DInt;
      Input : DInt;
      size : DInt;
   END_VAR
   VAR_TEMP
      idx : DInt;
   END_VAR
BEGIN
   #"Array"[#size+1] := #Input;
   #size := #size + 1;
END_FUNCTION

FUNCTION "Dequeue3" : Void   // FC2, SCL
{ S7_Optimized_Access := 'TRUE' }
VERSION : 0.1
   VAR_IN_OUT
      "array" : Array[1..3] of DInt;
      size : DInt;
      output : DInt;
   END_VAR
   VAR_TEMP
      idx : DInt;
   END_VAR
BEGIN
   #output := #"array"[1];
   FOR #idx := 1 TO 2 DO
       // Statement section FOR
       #"array"[#idx] := #"array"[#idx+1];
       #"array"[#idx + 1] := 0;
   END_FOR;
   #size := #size - 1;
END_FUNCTION

FUNCTION "Read" : Void   // FC3, LAD
{ S7_Optimized_Access := 'TRUE' }
VERSION : 0.1
BEGIN

REGION Network 1: Read RFID sect 0F - 1
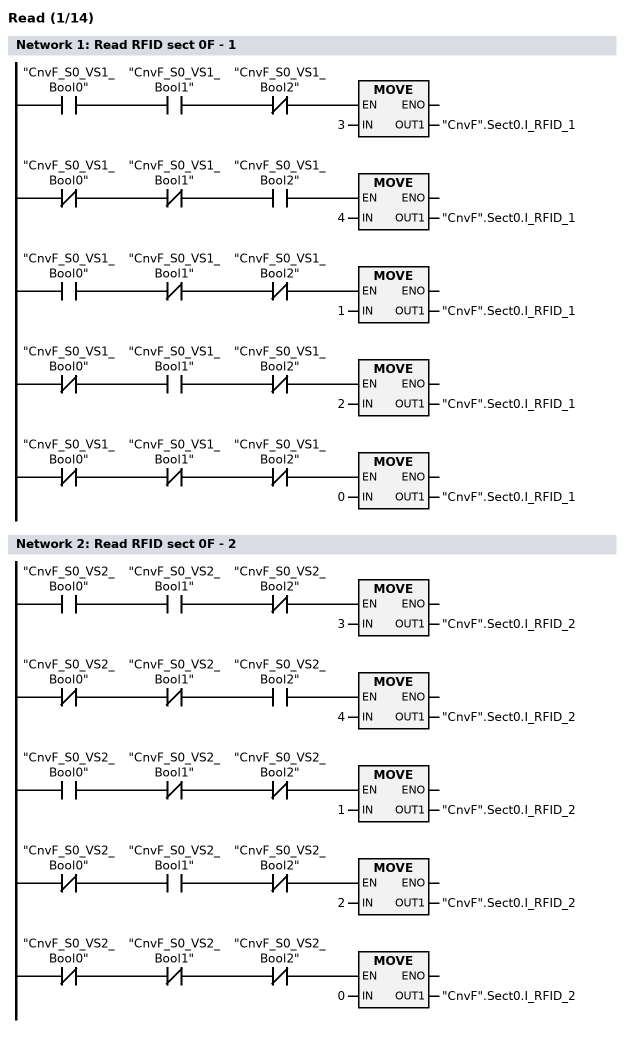
   RUNG wire#powerrail
      Contact( "CnvF_S0_VS1_Bool0" )
      Contact( "CnvF_S0_VS1_Bool1" )
      I_Contact( "CnvF_S0_VS1_Bool2" )
      Move(in := 3, out1 => "CnvF".Sect0.I_RFID_1)
   END_RUNG
   RUNG wire#powerrail
      I_Contact( "CnvF_S0_VS1_Bool0" )
      I_Contact( "CnvF_S0_VS1_Bool1" )
      Contact( "CnvF_S0_VS1_Bool2" )
      Move(in := 4, out1 => "CnvF".Sect0.I_RFID_1)
   END_RUNG
   RUNG wire#powerrail
      Contact( "CnvF_S0_VS1_Bool0" )
      I_Contact( "CnvF_S0_VS1_Bool1" )
      I_Contact( "CnvF_S0_VS1_Bool2" )
      Move(in := 1, out1 => "CnvF".Sect0.I_RFID_1)
   END_RUNG
   RUNG wire#powerrail
      I_Contact( "CnvF_S0_VS1_Bool0" )
      Contact( "CnvF_S0_VS1_Bool1" )
      I_Contact( "CnvF_S0_VS1_Bool2" )
      Move(in := 2, out1 => "CnvF".Sect0.I_RFID_1)
   END_RUNG
   RUNG wire#powerrail
      I_Contact( "CnvF_S0_VS1_Bool0" )
      I_Contact( "CnvF_S0_VS1_Bool1" )
      I_Contact( "CnvF_S0_VS1_Bool2" )
      Move(in := 0, out1 => "CnvF".Sect0.I_RFID_1)
   END_RUNG
   // the same network as SCL:
   IF "CnvF_S0_VS1_Bool0" AND "CnvF_S0_VS1_Bool1" AND NOT "CnvF_S0_VS1_Bool2" THEN
       "CnvF".Sect0.I_RFID_1 := 3;
   END_IF;
   IF NOT "CnvF_S0_VS1_Bool0" AND NOT "CnvF_S0_VS1_Bool1" AND "CnvF_S0_VS1_Bool2" THEN
       "CnvF".Sect0.I_RFID_1 := 4;
   END_IF;
   IF "CnvF_S0_VS1_Bool0" AND NOT "CnvF_S0_VS1_Bool1" AND NOT "CnvF_S0_VS1_Bool2" THEN
       "CnvF".Sect0.I_RFID_1 := 1;
   END_IF;
   IF NOT "CnvF_S0_VS1_Bool0" AND "CnvF_S0_VS1_Bool1" AND NOT "CnvF_S0_VS1_Bool2" THEN
       "CnvF".Sect0.I_RFID_1 := 2;
   END_IF;
   IF NOT "CnvF_S0_VS1_Bool0" AND NOT "CnvF_S0_VS1_Bool1" AND NOT "CnvF_S0_VS1_Bool2" THEN
       "CnvF".Sect0.I_RFID_1 := 0;
   END_IF;
END_REGION

REGION Network 2: Read RFID sect 0F - 2
   RUNG wire#powerrail
      Contact( "CnvF_S0_VS2_Bool0" )
      Contact( "CnvF_S0_VS2_Bool1" )
      I_Contact( "CnvF_S0_VS2_Bool2" )
      Move(in := 3, out1 => "CnvF".Sect0.I_RFID_2)
   END_RUNG
   RUNG wire#powerrail
      I_Contact( "CnvF_S0_VS2_Bool0" )
      I_Contact( "CnvF_S0_VS2_Bool1" )
      Contact( "CnvF_S0_VS2_Bool2" )
      Move(in := 4, out1 => "CnvF".Sect0.I_RFID_2)
   END_RUNG
   RUNG wire#powerrail
      Contact( "CnvF_S0_VS2_Bool0" )
      I_Contact( "CnvF_S0_VS2_Bool1" )
      I_Contact( "CnvF_S0_VS2_Bool2" )
      Move(in := 1, out1 => "CnvF".Sect0.I_RFID_2)
   END_RUNG
   RUNG wire#powerrail
      I_Contact( "CnvF_S0_VS2_Bool0" )
      Contact( "CnvF_S0_VS2_Bool1" )
      I_Contact( "CnvF_S0_VS2_Bool2" )
      Move(in := 2, out1 => "CnvF".Sect0.I_RFID_2)
   END_RUNG
   RUNG wire#powerrail
      I_Contact( "CnvF_S0_VS2_Bool0" )
      I_Contact( "CnvF_S0_VS2_Bool1" )
      I_Contact( "CnvF_S0_VS2_Bool2" )
      Move(in := 0, out1 => "CnvF".Sect0.I_RFID_2)
   END_RUNG
   // the same network as SCL:
   IF "CnvF_S0_VS2_Bool0" AND "CnvF_S0_VS2_Bool1" AND NOT "CnvF_S0_VS2_Bool2" THEN
       "CnvF".Sect0.I_RFID_2 := 3;
   END_IF;
   IF NOT "CnvF_S0_VS2_Bool0" AND NOT "CnvF_S0_VS2_Bool1" AND "CnvF_S0_VS2_Bool2" THEN
       "CnvF".Sect0.I_RFID_2 := 4;
   END_IF;
   IF "CnvF_S0_VS2_Bool0" AND NOT "CnvF_S0_VS2_Bool1" AND NOT "CnvF_S0_VS2_Bool2" THEN
       "CnvF".Sect0.I_RFID_2 := 1;
   END_IF;
   IF NOT "CnvF_S0_VS2_Bool0" AND "CnvF_S0_VS2_Bool1" AND NOT "CnvF_S0_VS2_Bool2" THEN
       "CnvF".Sect0.I_RFID_2 := 2;
   END_IF;
   IF NOT "CnvF_S0_VS2_Bool0" AND NOT "CnvF_S0_VS2_Bool1" AND NOT "CnvF_S0_VS2_Bool2" THEN
       "CnvF".Sect0.I_RFID_2 := 0;
   END_IF;
END_REGION

REGION Network 3: Read RFID sect 1F - 1
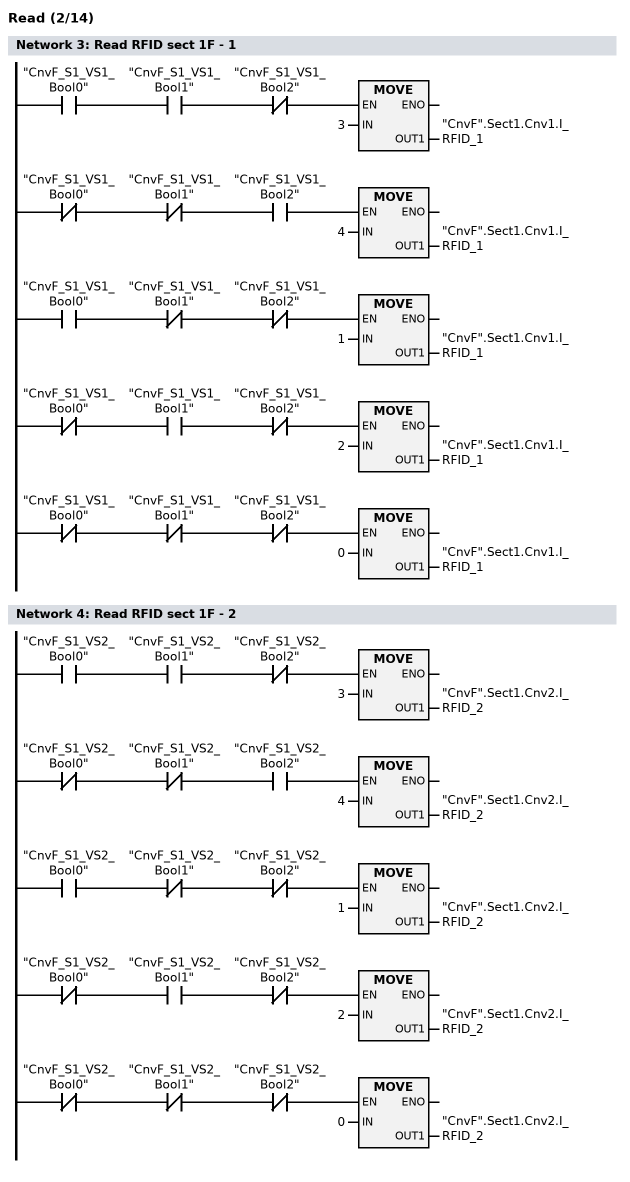
   RUNG wire#powerrail
      Contact( "CnvF_S1_VS1_Bool0" )
      Contact( "CnvF_S1_VS1_Bool1" )
      I_Contact( "CnvF_S1_VS1_Bool2" )
      Move(in := 3, out1 => "CnvF".Sect1.Cnv1.I_RFID_1)
   END_RUNG
   RUNG wire#powerrail
      I_Contact( "CnvF_S1_VS1_Bool0" )
      I_Contact( "CnvF_S1_VS1_Bool1" )
      Contact( "CnvF_S1_VS1_Bool2" )
      Move(in := 4, out1 => "CnvF".Sect1.Cnv1.I_RFID_1)
   END_RUNG
   RUNG wire#powerrail
      Contact( "CnvF_S1_VS1_Bool0" )
      I_Contact( "CnvF_S1_VS1_Bool1" )
      I_Contact( "CnvF_S1_VS1_Bool2" )
      Move(in := 1, out1 => "CnvF".Sect1.Cnv1.I_RFID_1)
   END_RUNG
   RUNG wire#powerrail
      I_Contact( "CnvF_S1_VS1_Bool0" )
      Contact( "CnvF_S1_VS1_Bool1" )
      I_Contact( "CnvF_S1_VS1_Bool2" )
      Move(in := 2, out1 => "CnvF".Sect1.Cnv1.I_RFID_1)
   END_RUNG
   RUNG wire#powerrail
      I_Contact( "CnvF_S1_VS1_Bool0" )
      I_Contact( "CnvF_S1_VS1_Bool1" )
      I_Contact( "CnvF_S1_VS1_Bool2" )
      Move(in := 0, out1 => "CnvF".Sect1.Cnv1.I_RFID_1)
   END_RUNG
   // the same network as SCL:
   IF "CnvF_S1_VS1_Bool0" AND "CnvF_S1_VS1_Bool1" AND NOT "CnvF_S1_VS1_Bool2" THEN
       "CnvF".Sect1.Cnv1.I_RFID_1 := 3;
   END_IF;
   IF NOT "CnvF_S1_VS1_Bool0" AND NOT "CnvF_S1_VS1_Bool1" AND "CnvF_S1_VS1_Bool2" THEN
       "CnvF".Sect1.Cnv1.I_RFID_1 := 4;
   END_IF;
   IF "CnvF_S1_VS1_Bool0" AND NOT "CnvF_S1_VS1_Bool1" AND NOT "CnvF_S1_VS1_Bool2" THEN
       "CnvF".Sect1.Cnv1.I_RFID_1 := 1;
   END_IF;
   IF NOT "CnvF_S1_VS1_Bool0" AND "CnvF_S1_VS1_Bool1" AND NOT "CnvF_S1_VS1_Bool2" THEN
       "CnvF".Sect1.Cnv1.I_RFID_1 := 2;
   END_IF;
   IF NOT "CnvF_S1_VS1_Bool0" AND NOT "CnvF_S1_VS1_Bool1" AND NOT "CnvF_S1_VS1_Bool2" THEN
       "CnvF".Sect1.Cnv1.I_RFID_1 := 0;
   END_IF;
END_REGION

REGION Network 4: Read RFID sect 1F - 2
   RUNG wire#powerrail
      Contact( "CnvF_S1_VS2_Bool0" )
      Contact( "CnvF_S1_VS2_Bool1" )
      I_Contact( "CnvF_S1_VS2_Bool2" )
      Move(in := 3, out1 => "CnvF".Sect1.Cnv2.I_RFID_2)
   END_RUNG
   RUNG wire#powerrail
      I_Contact( "CnvF_S1_VS2_Bool0" )
      I_Contact( "CnvF_S1_VS2_Bool1" )
      Contact( "CnvF_S1_VS2_Bool2" )
      Move(in := 4, out1 => "CnvF".Sect1.Cnv2.I_RFID_2)
   END_RUNG
   RUNG wire#powerrail
      Contact( "CnvF_S1_VS2_Bool0" )
      I_Contact( "CnvF_S1_VS2_Bool1" )
      I_Contact( "CnvF_S1_VS2_Bool2" )
      Move(in := 1, out1 => "CnvF".Sect1.Cnv2.I_RFID_2)
   END_RUNG
   RUNG wire#powerrail
      I_Contact( "CnvF_S1_VS2_Bool0" )
      Contact( "CnvF_S1_VS2_Bool1" )
      I_Contact( "CnvF_S1_VS2_Bool2" )
      Move(in := 2, out1 => "CnvF".Sect1.Cnv2.I_RFID_2)
   END_RUNG
   RUNG wire#powerrail
      I_Contact( "CnvF_S1_VS2_Bool0" )
      I_Contact( "CnvF_S1_VS2_Bool1" )
      I_Contact( "CnvF_S1_VS2_Bool2" )
      Move(in := 0, out1 => "CnvF".Sect1.Cnv2.I_RFID_2)
   END_RUNG
   // the same network as SCL:
   IF "CnvF_S1_VS2_Bool0" AND "CnvF_S1_VS2_Bool1" AND NOT "CnvF_S1_VS2_Bool2" THEN
       "CnvF".Sect1.Cnv2.I_RFID_2 := 3;
   END_IF;
   IF NOT "CnvF_S1_VS2_Bool0" AND NOT "CnvF_S1_VS2_Bool1" AND "CnvF_S1_VS2_Bool2" THEN
       "CnvF".Sect1.Cnv2.I_RFID_2 := 4;
   END_IF;
   IF "CnvF_S1_VS2_Bool0" AND NOT "CnvF_S1_VS2_Bool1" AND NOT "CnvF_S1_VS2_Bool2" THEN
       "CnvF".Sect1.Cnv2.I_RFID_2 := 1;
   END_IF;
   IF NOT "CnvF_S1_VS2_Bool0" AND "CnvF_S1_VS2_Bool1" AND NOT "CnvF_S1_VS2_Bool2" THEN
       "CnvF".Sect1.Cnv2.I_RFID_2 := 2;
   END_IF;
   IF NOT "CnvF_S1_VS2_Bool0" AND NOT "CnvF_S1_VS2_Bool1" AND NOT "CnvF_S1_VS2_Bool2" THEN
       "CnvF".Sect1.Cnv2.I_RFID_2 := 0;
   END_IF;
END_REGION

REGION Network 5: Read RFID sect 2-1F - 1
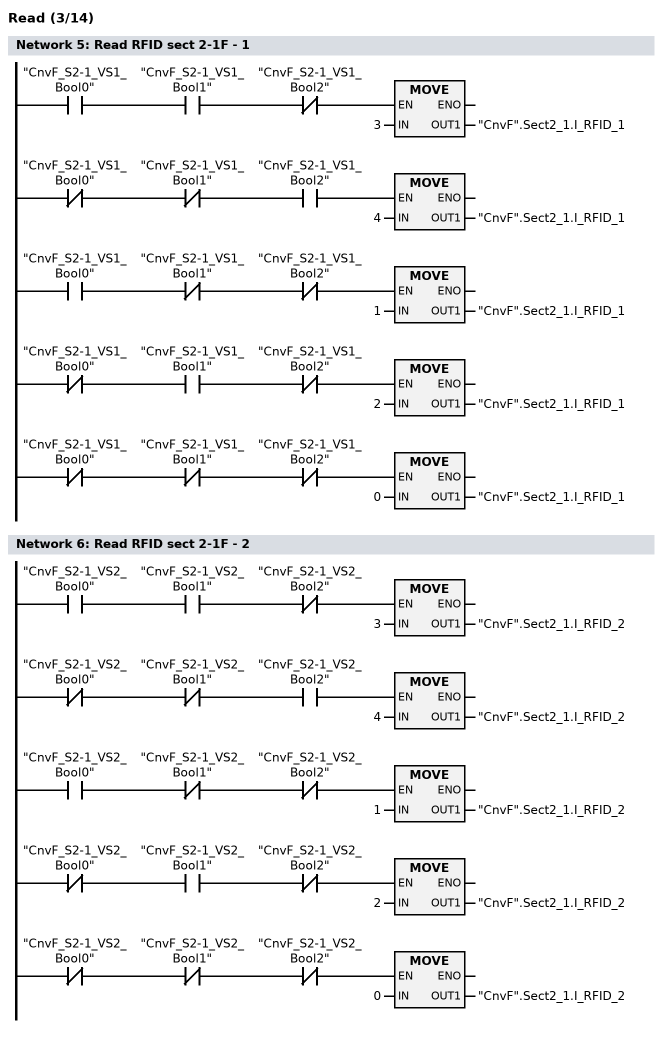
   RUNG wire#powerrail
      Contact( "CnvF_S2-1_VS1_Bool0" )
      Contact( "CnvF_S2-1_VS1_Bool1" )
      I_Contact( "CnvF_S2-1_VS1_Bool2" )
      Move(in := 3, out1 => "CnvF".Sect2_1.I_RFID_1)
   END_RUNG
   RUNG wire#powerrail
      I_Contact( "CnvF_S2-1_VS1_Bool0" )
      I_Contact( "CnvF_S2-1_VS1_Bool1" )
      Contact( "CnvF_S2-1_VS1_Bool2" )
      Move(in := 4, out1 => "CnvF".Sect2_1.I_RFID_1)
   END_RUNG
   RUNG wire#powerrail
      Contact( "CnvF_S2-1_VS1_Bool0" )
      I_Contact( "CnvF_S2-1_VS1_Bool1" )
      I_Contact( "CnvF_S2-1_VS1_Bool2" )
      Move(in := 1, out1 => "CnvF".Sect2_1.I_RFID_1)
   END_RUNG
   RUNG wire#powerrail
      I_Contact( "CnvF_S2-1_VS1_Bool0" )
      Contact( "CnvF_S2-1_VS1_Bool1" )
      I_Contact( "CnvF_S2-1_VS1_Bool2" )
      Move(in := 2, out1 => "CnvF".Sect2_1.I_RFID_1)
   END_RUNG
   RUNG wire#powerrail
      I_Contact( "CnvF_S2-1_VS1_Bool0" )
      I_Contact( "CnvF_S2-1_VS1_Bool1" )
      I_Contact( "CnvF_S2-1_VS1_Bool2" )
      Move(in := 0, out1 => "CnvF".Sect2_1.I_RFID_1)
   END_RUNG
   // the same network as SCL:
   IF "CnvF_S2-1_VS1_Bool0" AND "CnvF_S2-1_VS1_Bool1" AND NOT "CnvF_S2-1_VS1_Bool2" THEN
       "CnvF".Sect2_1.I_RFID_1 := 3;
   END_IF;
   IF NOT "CnvF_S2-1_VS1_Bool0" AND NOT "CnvF_S2-1_VS1_Bool1" AND "CnvF_S2-1_VS1_Bool2" THEN
       "CnvF".Sect2_1.I_RFID_1 := 4;
   END_IF;
   IF "CnvF_S2-1_VS1_Bool0" AND NOT "CnvF_S2-1_VS1_Bool1" AND NOT "CnvF_S2-1_VS1_Bool2" THEN
       "CnvF".Sect2_1.I_RFID_1 := 1;
   END_IF;
   IF NOT "CnvF_S2-1_VS1_Bool0" AND "CnvF_S2-1_VS1_Bool1" AND NOT "CnvF_S2-1_VS1_Bool2" THEN
       "CnvF".Sect2_1.I_RFID_1 := 2;
   END_IF;
   IF NOT "CnvF_S2-1_VS1_Bool0" AND NOT "CnvF_S2-1_VS1_Bool1" AND NOT "CnvF_S2-1_VS1_Bool2" THEN
       "CnvF".Sect2_1.I_RFID_1 := 0;
   END_IF;
END_REGION

REGION Network 6: Read RFID sect 2-1F - 2
   RUNG wire#powerrail
      Contact( "CnvF_S2-1_VS2_Bool0" )
      Contact( "CnvF_S2-1_VS2_Bool1" )
      I_Contact( "CnvF_S2-1_VS2_Bool2" )
      Move(in := 3, out1 => "CnvF".Sect2_1.I_RFID_2)
   END_RUNG
   RUNG wire#powerrail
      I_Contact( "CnvF_S2-1_VS2_Bool0" )
      I_Contact( "CnvF_S2-1_VS2_Bool1" )
      Contact( "CnvF_S2-1_VS2_Bool2" )
      Move(in := 4, out1 => "CnvF".Sect2_1.I_RFID_2)
   END_RUNG
   RUNG wire#powerrail
      Contact( "CnvF_S2-1_VS2_Bool0" )
      I_Contact( "CnvF_S2-1_VS2_Bool1" )
      I_Contact( "CnvF_S2-1_VS2_Bool2" )
      Move(in := 1, out1 => "CnvF".Sect2_1.I_RFID_2)
   END_RUNG
   RUNG wire#powerrail
      I_Contact( "CnvF_S2-1_VS2_Bool0" )
      Contact( "CnvF_S2-1_VS2_Bool1" )
      I_Contact( "CnvF_S2-1_VS2_Bool2" )
      Move(in := 2, out1 => "CnvF".Sect2_1.I_RFID_2)
   END_RUNG
   RUNG wire#powerrail
      I_Contact( "CnvF_S2-1_VS2_Bool0" )
      I_Contact( "CnvF_S2-1_VS2_Bool1" )
      I_Contact( "CnvF_S2-1_VS2_Bool2" )
      Move(in := 0, out1 => "CnvF".Sect2_1.I_RFID_2)
   END_RUNG
   // the same network as SCL:
   IF "CnvF_S2-1_VS2_Bool0" AND "CnvF_S2-1_VS2_Bool1" AND NOT "CnvF_S2-1_VS2_Bool2" THEN
       "CnvF".Sect2_1.I_RFID_2 := 3;
   END_IF;
   IF NOT "CnvF_S2-1_VS2_Bool0" AND NOT "CnvF_S2-1_VS2_Bool1" AND "CnvF_S2-1_VS2_Bool2" THEN
       "CnvF".Sect2_1.I_RFID_2 := 4;
   END_IF;
   IF "CnvF_S2-1_VS2_Bool0" AND NOT "CnvF_S2-1_VS2_Bool1" AND NOT "CnvF_S2-1_VS2_Bool2" THEN
       "CnvF".Sect2_1.I_RFID_2 := 1;
   END_IF;
   IF NOT "CnvF_S2-1_VS2_Bool0" AND "CnvF_S2-1_VS2_Bool1" AND NOT "CnvF_S2-1_VS2_Bool2" THEN
       "CnvF".Sect2_1.I_RFID_2 := 2;
   END_IF;
   IF NOT "CnvF_S2-1_VS2_Bool0" AND NOT "CnvF_S2-1_VS2_Bool1" AND NOT "CnvF_S2-1_VS2_Bool2" THEN
       "CnvF".Sect2_1.I_RFID_2 := 0;
   END_IF;
END_REGION

REGION Network 7: Read RFID sect 2-2F - 1
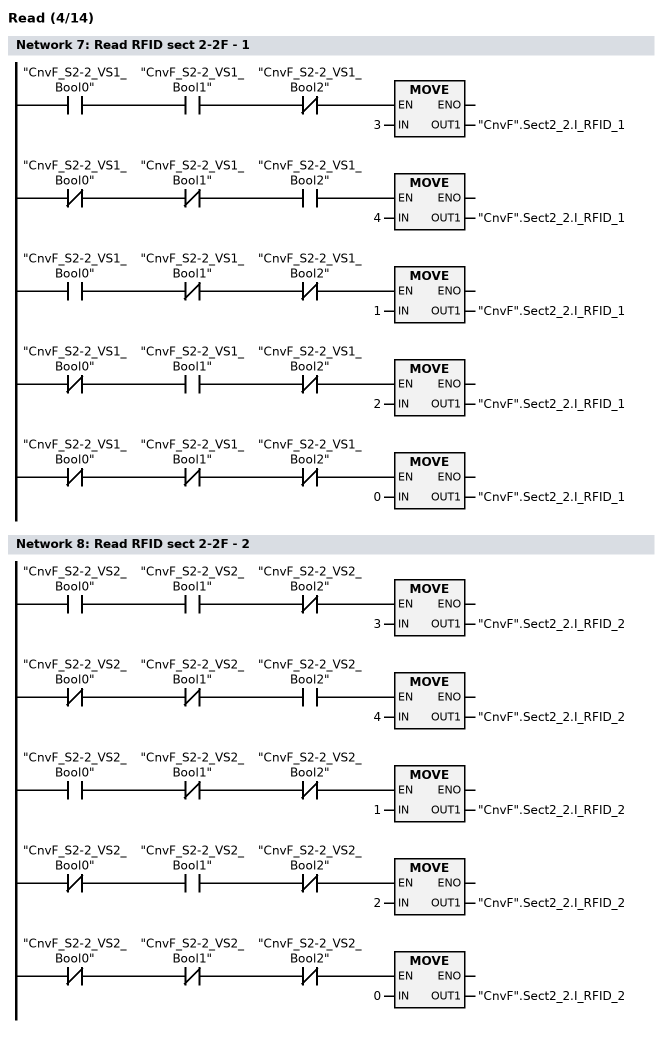
   RUNG wire#powerrail
      Contact( "CnvF_S2-2_VS1_Bool0" )
      Contact( "CnvF_S2-2_VS1_Bool1" )
      I_Contact( "CnvF_S2-2_VS1_Bool2" )
      Move(in := 3, out1 => "CnvF".Sect2_2.I_RFID_1)
   END_RUNG
   RUNG wire#powerrail
      I_Contact( "CnvF_S2-2_VS1_Bool0" )
      I_Contact( "CnvF_S2-2_VS1_Bool1" )
      Contact( "CnvF_S2-2_VS1_Bool2" )
      Move(in := 4, out1 => "CnvF".Sect2_2.I_RFID_1)
   END_RUNG
   RUNG wire#powerrail
      Contact( "CnvF_S2-2_VS1_Bool0" )
      I_Contact( "CnvF_S2-2_VS1_Bool1" )
      I_Contact( "CnvF_S2-2_VS1_Bool2" )
      Move(in := 1, out1 => "CnvF".Sect2_2.I_RFID_1)
   END_RUNG
   RUNG wire#powerrail
      I_Contact( "CnvF_S2-2_VS1_Bool0" )
      Contact( "CnvF_S2-2_VS1_Bool1" )
      I_Contact( "CnvF_S2-2_VS1_Bool2" )
      Move(in := 2, out1 => "CnvF".Sect2_2.I_RFID_1)
   END_RUNG
   RUNG wire#powerrail
      I_Contact( "CnvF_S2-2_VS1_Bool0" )
      I_Contact( "CnvF_S2-2_VS1_Bool1" )
      I_Contact( "CnvF_S2-2_VS1_Bool2" )
      Move(in := 0, out1 => "CnvF".Sect2_2.I_RFID_1)
   END_RUNG
   // the same network as SCL:
   IF "CnvF_S2-2_VS1_Bool0" AND "CnvF_S2-2_VS1_Bool1" AND NOT "CnvF_S2-2_VS1_Bool2" THEN
       "CnvF".Sect2_2.I_RFID_1 := 3;
   END_IF;
   IF NOT "CnvF_S2-2_VS1_Bool0" AND NOT "CnvF_S2-2_VS1_Bool1" AND "CnvF_S2-2_VS1_Bool2" THEN
       "CnvF".Sect2_2.I_RFID_1 := 4;
   END_IF;
   IF "CnvF_S2-2_VS1_Bool0" AND NOT "CnvF_S2-2_VS1_Bool1" AND NOT "CnvF_S2-2_VS1_Bool2" THEN
       "CnvF".Sect2_2.I_RFID_1 := 1;
   END_IF;
   IF NOT "CnvF_S2-2_VS1_Bool0" AND "CnvF_S2-2_VS1_Bool1" AND NOT "CnvF_S2-2_VS1_Bool2" THEN
       "CnvF".Sect2_2.I_RFID_1 := 2;
   END_IF;
   IF NOT "CnvF_S2-2_VS1_Bool0" AND NOT "CnvF_S2-2_VS1_Bool1" AND NOT "CnvF_S2-2_VS1_Bool2" THEN
       "CnvF".Sect2_2.I_RFID_1 := 0;
   END_IF;
END_REGION

REGION Network 8: Read RFID sect 2-2F - 2
   RUNG wire#powerrail
      Contact( "CnvF_S2-2_VS2_Bool0" )
      Contact( "CnvF_S2-2_VS2_Bool1" )
      I_Contact( "CnvF_S2-2_VS2_Bool2" )
      Move(in := 3, out1 => "CnvF".Sect2_2.I_RFID_2)
   END_RUNG
   RUNG wire#powerrail
      I_Contact( "CnvF_S2-2_VS2_Bool0" )
      I_Contact( "CnvF_S2-2_VS2_Bool1" )
      Contact( "CnvF_S2-2_VS2_Bool2" )
      Move(in := 4, out1 => "CnvF".Sect2_2.I_RFID_2)
   END_RUNG
   RUNG wire#powerrail
      Contact( "CnvF_S2-2_VS2_Bool0" )
      I_Contact( "CnvF_S2-2_VS2_Bool1" )
      I_Contact( "CnvF_S2-2_VS2_Bool2" )
      Move(in := 1, out1 => "CnvF".Sect2_2.I_RFID_2)
   END_RUNG
   RUNG wire#powerrail
      I_Contact( "CnvF_S2-2_VS2_Bool0" )
      Contact( "CnvF_S2-2_VS2_Bool1" )
      I_Contact( "CnvF_S2-2_VS2_Bool2" )
      Move(in := 2, out1 => "CnvF".Sect2_2.I_RFID_2)
   END_RUNG
   RUNG wire#powerrail
      I_Contact( "CnvF_S2-2_VS2_Bool0" )
      I_Contact( "CnvF_S2-2_VS2_Bool1" )
      I_Contact( "CnvF_S2-2_VS2_Bool2" )
      Move(in := 0, out1 => "CnvF".Sect2_2.I_RFID_2)
   END_RUNG
   // the same network as SCL:
   IF "CnvF_S2-2_VS2_Bool0" AND "CnvF_S2-2_VS2_Bool1" AND NOT "CnvF_S2-2_VS2_Bool2" THEN
       "CnvF".Sect2_2.I_RFID_2 := 3;
   END_IF;
   IF NOT "CnvF_S2-2_VS2_Bool0" AND NOT "CnvF_S2-2_VS2_Bool1" AND "CnvF_S2-2_VS2_Bool2" THEN
       "CnvF".Sect2_2.I_RFID_2 := 4;
   END_IF;
   IF "CnvF_S2-2_VS2_Bool0" AND NOT "CnvF_S2-2_VS2_Bool1" AND NOT "CnvF_S2-2_VS2_Bool2" THEN
       "CnvF".Sect2_2.I_RFID_2 := 1;
   END_IF;
   IF NOT "CnvF_S2-2_VS2_Bool0" AND "CnvF_S2-2_VS2_Bool1" AND NOT "CnvF_S2-2_VS2_Bool2" THEN
       "CnvF".Sect2_2.I_RFID_2 := 2;
   END_IF;
   IF NOT "CnvF_S2-2_VS2_Bool0" AND NOT "CnvF_S2-2_VS2_Bool1" AND NOT "CnvF_S2-2_VS2_Bool2" THEN
       "CnvF".Sect2_2.I_RFID_2 := 0;
   END_IF;
END_REGION

REGION Network 9: Read RFID sect 3H - 1
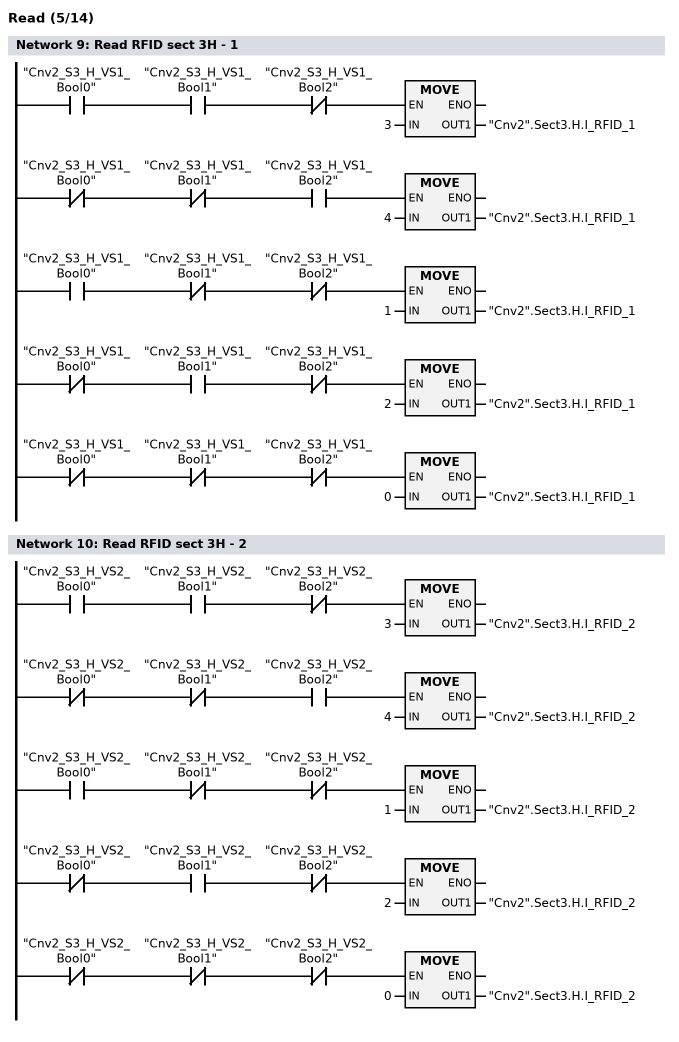
   RUNG wire#powerrail
      Contact( "Cnv2_S3_H_VS1_Bool0" )
      Contact( "Cnv2_S3_H_VS1_Bool1" )
      I_Contact( "Cnv2_S3_H_VS1_Bool2" )
      Move(in := 3, out1 => "Cnv2".Sect3.H.I_RFID_1)
   END_RUNG
   RUNG wire#powerrail
      I_Contact( "Cnv2_S3_H_VS1_Bool0" )
      I_Contact( "Cnv2_S3_H_VS1_Bool1" )
      Contact( "Cnv2_S3_H_VS1_Bool2" )
      Move(in := 4, out1 => "Cnv2".Sect3.H.I_RFID_1)
   END_RUNG
   RUNG wire#powerrail
      Contact( "Cnv2_S3_H_VS1_Bool0" )
      I_Contact( "Cnv2_S3_H_VS1_Bool1" )
      I_Contact( "Cnv2_S3_H_VS1_Bool2" )
      Move(in := 1, out1 => "Cnv2".Sect3.H.I_RFID_1)
   END_RUNG
   RUNG wire#powerrail
      I_Contact( "Cnv2_S3_H_VS1_Bool0" )
      Contact( "Cnv2_S3_H_VS1_Bool1" )
      I_Contact( "Cnv2_S3_H_VS1_Bool2" )
      Move(in := 2, out1 => "Cnv2".Sect3.H.I_RFID_1)
   END_RUNG
   RUNG wire#powerrail
      I_Contact( "Cnv2_S3_H_VS1_Bool0" )
      I_Contact( "Cnv2_S3_H_VS1_Bool1" )
      I_Contact( "Cnv2_S3_H_VS1_Bool2" )
      Move(in := 0, out1 => "Cnv2".Sect3.H.I_RFID_1)
   END_RUNG
   // the same network as SCL:
   IF "Cnv2_S3_H_VS1_Bool0" AND "Cnv2_S3_H_VS1_Bool1" AND NOT "Cnv2_S3_H_VS1_Bool2" THEN
       "Cnv2".Sect3.H.I_RFID_1 := 3;
   END_IF;
   IF NOT "Cnv2_S3_H_VS1_Bool0" AND NOT "Cnv2_S3_H_VS1_Bool1" AND "Cnv2_S3_H_VS1_Bool2" THEN
       "Cnv2".Sect3.H.I_RFID_1 := 4;
   END_IF;
   IF "Cnv2_S3_H_VS1_Bool0" AND NOT "Cnv2_S3_H_VS1_Bool1" AND NOT "Cnv2_S3_H_VS1_Bool2" THEN
       "Cnv2".Sect3.H.I_RFID_1 := 1;
   END_IF;
   IF NOT "Cnv2_S3_H_VS1_Bool0" AND "Cnv2_S3_H_VS1_Bool1" AND NOT "Cnv2_S3_H_VS1_Bool2" THEN
       "Cnv2".Sect3.H.I_RFID_1 := 2;
   END_IF;
   IF NOT "Cnv2_S3_H_VS1_Bool0" AND NOT "Cnv2_S3_H_VS1_Bool1" AND NOT "Cnv2_S3_H_VS1_Bool2" THEN
       "Cnv2".Sect3.H.I_RFID_1 := 0;
   END_IF;
END_REGION

REGION Network 10: Read RFID sect 3H - 2
   RUNG wire#powerrail
      Contact( "Cnv2_S3_H_VS2_Bool0" )
      Contact( "Cnv2_S3_H_VS2_Bool1" )
      I_Contact( "Cnv2_S3_H_VS2_Bool2" )
      Move(in := 3, out1 => "Cnv2".Sect3.H.I_RFID_2)
   END_RUNG
   RUNG wire#powerrail
      I_Contact( "Cnv2_S3_H_VS2_Bool0" )
      I_Contact( "Cnv2_S3_H_VS2_Bool1" )
      Contact( "Cnv2_S3_H_VS2_Bool2" )
      Move(in := 4, out1 => "Cnv2".Sect3.H.I_RFID_2)
   END_RUNG
   RUNG wire#powerrail
      Contact( "Cnv2_S3_H_VS2_Bool0" )
      I_Contact( "Cnv2_S3_H_VS2_Bool1" )
      I_Contact( "Cnv2_S3_H_VS2_Bool2" )
      Move(in := 1, out1 => "Cnv2".Sect3.H.I_RFID_2)
   END_RUNG
   RUNG wire#powerrail
      I_Contact( "Cnv2_S3_H_VS2_Bool0" )
      Contact( "Cnv2_S3_H_VS2_Bool1" )
      I_Contact( "Cnv2_S3_H_VS2_Bool2" )
      Move(in := 2, out1 => "Cnv2".Sect3.H.I_RFID_2)
   END_RUNG
   RUNG wire#powerrail
      I_Contact( "Cnv2_S3_H_VS2_Bool0" )
      I_Contact( "Cnv2_S3_H_VS2_Bool1" )
      I_Contact( "Cnv2_S3_H_VS2_Bool2" )
      Move(in := 0, out1 => "Cnv2".Sect3.H.I_RFID_2)
   END_RUNG
   // the same network as SCL:
   IF "Cnv2_S3_H_VS2_Bool0" AND "Cnv2_S3_H_VS2_Bool1" AND NOT "Cnv2_S3_H_VS2_Bool2" THEN
       "Cnv2".Sect3.H.I_RFID_2 := 3;
   END_IF;
   IF NOT "Cnv2_S3_H_VS2_Bool0" AND NOT "Cnv2_S3_H_VS2_Bool1" AND "Cnv2_S3_H_VS2_Bool2" THEN
       "Cnv2".Sect3.H.I_RFID_2 := 4;
   END_IF;
   IF "Cnv2_S3_H_VS2_Bool0" AND NOT "Cnv2_S3_H_VS2_Bool1" AND NOT "Cnv2_S3_H_VS2_Bool2" THEN
       "Cnv2".Sect3.H.I_RFID_2 := 1;
   END_IF;
   IF NOT "Cnv2_S3_H_VS2_Bool0" AND "Cnv2_S3_H_VS2_Bool1" AND NOT "Cnv2_S3_H_VS2_Bool2" THEN
       "Cnv2".Sect3.H.I_RFID_2 := 2;
   END_IF;
   IF NOT "Cnv2_S3_H_VS2_Bool0" AND NOT "Cnv2_S3_H_VS2_Bool1" AND NOT "Cnv2_S3_H_VS2_Bool2" THEN
       "Cnv2".Sect3.H.I_RFID_2 := 0;
   END_IF;
END_REGION

REGION Network 11: Read RFID sect 3L - 1
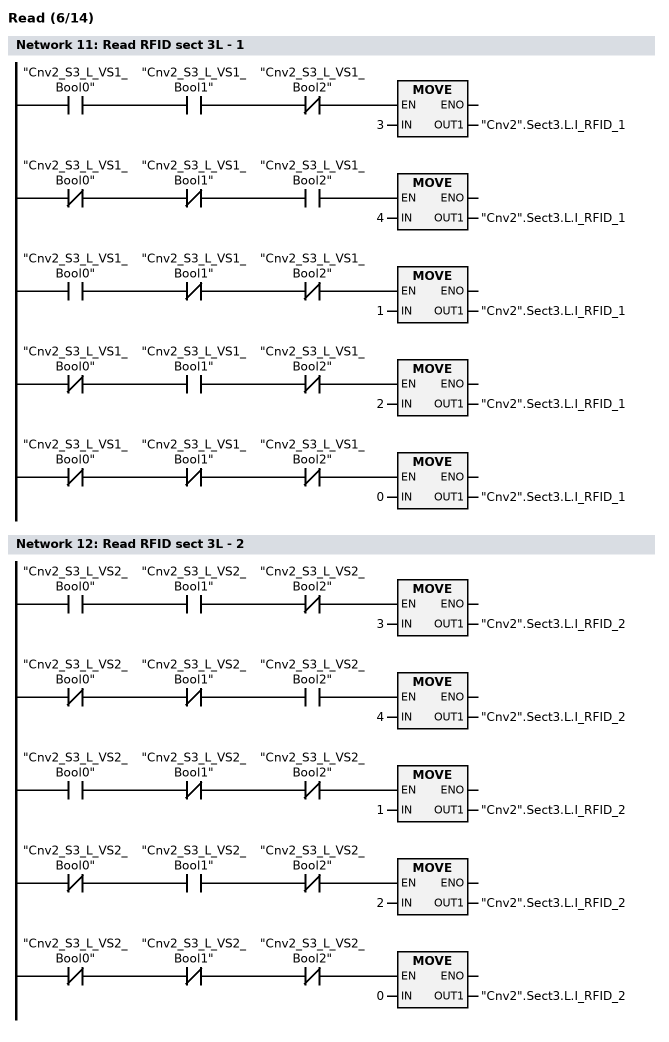
   RUNG wire#powerrail
      Contact( "Cnv2_S3_L_VS1_Bool0" )
      Contact( "Cnv2_S3_L_VS1_Bool1" )
      I_Contact( "Cnv2_S3_L_VS1_Bool2" )
      Move(in := 3, out1 => "Cnv2".Sect3.L.I_RFID_1)
   END_RUNG
   RUNG wire#powerrail
      I_Contact( "Cnv2_S3_L_VS1_Bool0" )
      I_Contact( "Cnv2_S3_L_VS1_Bool1" )
      Contact( "Cnv2_S3_L_VS1_Bool2" )
      Move(in := 4, out1 => "Cnv2".Sect3.L.I_RFID_1)
   END_RUNG
   RUNG wire#powerrail
      Contact( "Cnv2_S3_L_VS1_Bool0" )
      I_Contact( "Cnv2_S3_L_VS1_Bool1" )
      I_Contact( "Cnv2_S3_L_VS1_Bool2" )
      Move(in := 1, out1 => "Cnv2".Sect3.L.I_RFID_1)
   END_RUNG
   RUNG wire#powerrail
      I_Contact( "Cnv2_S3_L_VS1_Bool0" )
      Contact( "Cnv2_S3_L_VS1_Bool1" )
      I_Contact( "Cnv2_S3_L_VS1_Bool2" )
      Move(in := 2, out1 => "Cnv2".Sect3.L.I_RFID_1)
   END_RUNG
   RUNG wire#powerrail
      I_Contact( "Cnv2_S3_L_VS1_Bool0" )
      I_Contact( "Cnv2_S3_L_VS1_Bool1" )
      I_Contact( "Cnv2_S3_L_VS1_Bool2" )
      Move(in := 0, out1 => "Cnv2".Sect3.L.I_RFID_1)
   END_RUNG
   // the same network as SCL:
   IF "Cnv2_S3_L_VS1_Bool0" AND "Cnv2_S3_L_VS1_Bool1" AND NOT "Cnv2_S3_L_VS1_Bool2" THEN
       "Cnv2".Sect3.L.I_RFID_1 := 3;
   END_IF;
   IF NOT "Cnv2_S3_L_VS1_Bool0" AND NOT "Cnv2_S3_L_VS1_Bool1" AND "Cnv2_S3_L_VS1_Bool2" THEN
       "Cnv2".Sect3.L.I_RFID_1 := 4;
   END_IF;
   IF "Cnv2_S3_L_VS1_Bool0" AND NOT "Cnv2_S3_L_VS1_Bool1" AND NOT "Cnv2_S3_L_VS1_Bool2" THEN
       "Cnv2".Sect3.L.I_RFID_1 := 1;
   END_IF;
   IF NOT "Cnv2_S3_L_VS1_Bool0" AND "Cnv2_S3_L_VS1_Bool1" AND NOT "Cnv2_S3_L_VS1_Bool2" THEN
       "Cnv2".Sect3.L.I_RFID_1 := 2;
   END_IF;
   IF NOT "Cnv2_S3_L_VS1_Bool0" AND NOT "Cnv2_S3_L_VS1_Bool1" AND NOT "Cnv2_S3_L_VS1_Bool2" THEN
       "Cnv2".Sect3.L.I_RFID_1 := 0;
   END_IF;
END_REGION

REGION Network 12: Read RFID sect 3L - 2
   RUNG wire#powerrail
      Contact( "Cnv2_S3_L_VS2_Bool0" )
      Contact( "Cnv2_S3_L_VS2_Bool1" )
      I_Contact( "Cnv2_S3_L_VS2_Bool2" )
      Move(in := 3, out1 => "Cnv2".Sect3.L.I_RFID_2)
   END_RUNG
   RUNG wire#powerrail
      I_Contact( "Cnv2_S3_L_VS2_Bool0" )
      I_Contact( "Cnv2_S3_L_VS2_Bool1" )
      Contact( "Cnv2_S3_L_VS2_Bool2" )
      Move(in := 4, out1 => "Cnv2".Sect3.L.I_RFID_2)
   END_RUNG
   RUNG wire#powerrail
      Contact( "Cnv2_S3_L_VS2_Bool0" )
      I_Contact( "Cnv2_S3_L_VS2_Bool1" )
      I_Contact( "Cnv2_S3_L_VS2_Bool2" )
      Move(in := 1, out1 => "Cnv2".Sect3.L.I_RFID_2)
   END_RUNG
   RUNG wire#powerrail
      I_Contact( "Cnv2_S3_L_VS2_Bool0" )
      Contact( "Cnv2_S3_L_VS2_Bool1" )
      I_Contact( "Cnv2_S3_L_VS2_Bool2" )
      Move(in := 2, out1 => "Cnv2".Sect3.L.I_RFID_2)
   END_RUNG
   RUNG wire#powerrail
      I_Contact( "Cnv2_S3_L_VS2_Bool0" )
      I_Contact( "Cnv2_S3_L_VS2_Bool1" )
      I_Contact( "Cnv2_S3_L_VS2_Bool2" )
      Move(in := 0, out1 => "Cnv2".Sect3.L.I_RFID_2)
   END_RUNG
   // the same network as SCL:
   IF "Cnv2_S3_L_VS2_Bool0" AND "Cnv2_S3_L_VS2_Bool1" AND NOT "Cnv2_S3_L_VS2_Bool2" THEN
       "Cnv2".Sect3.L.I_RFID_2 := 3;
   END_IF;
   IF NOT "Cnv2_S3_L_VS2_Bool0" AND NOT "Cnv2_S3_L_VS2_Bool1" AND "Cnv2_S3_L_VS2_Bool2" THEN
       "Cnv2".Sect3.L.I_RFID_2 := 4;
   END_IF;
   IF "Cnv2_S3_L_VS2_Bool0" AND NOT "Cnv2_S3_L_VS2_Bool1" AND NOT "Cnv2_S3_L_VS2_Bool2" THEN
       "Cnv2".Sect3.L.I_RFID_2 := 1;
   END_IF;
   IF NOT "Cnv2_S3_L_VS2_Bool0" AND "Cnv2_S3_L_VS2_Bool1" AND NOT "Cnv2_S3_L_VS2_Bool2" THEN
       "Cnv2".Sect3.L.I_RFID_2 := 2;
   END_IF;
   IF NOT "Cnv2_S3_L_VS2_Bool0" AND NOT "Cnv2_S3_L_VS2_Bool1" AND NOT "Cnv2_S3_L_VS2_Bool2" THEN
       "Cnv2".Sect3.L.I_RFID_2 := 0;
   END_IF;
END_REGION

REGION Network 13: Read RFID sect 4H - 1
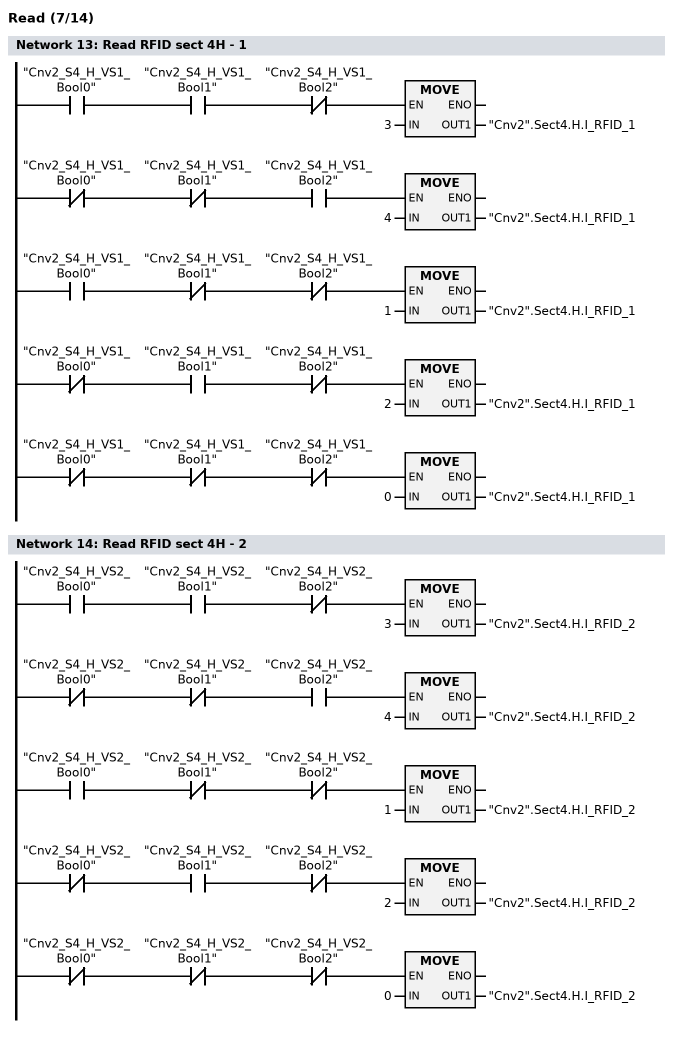
   RUNG wire#powerrail
      Contact( "Cnv2_S4_H_VS1_Bool0" )
      Contact( "Cnv2_S4_H_VS1_Bool1" )
      I_Contact( "Cnv2_S4_H_VS1_Bool2" )
      Move(in := 3, out1 => "Cnv2".Sect4.H.I_RFID_1)
   END_RUNG
   RUNG wire#powerrail
      I_Contact( "Cnv2_S4_H_VS1_Bool0" )
      I_Contact( "Cnv2_S4_H_VS1_Bool1" )
      Contact( "Cnv2_S4_H_VS1_Bool2" )
      Move(in := 4, out1 => "Cnv2".Sect4.H.I_RFID_1)
   END_RUNG
   RUNG wire#powerrail
      Contact( "Cnv2_S4_H_VS1_Bool0" )
      I_Contact( "Cnv2_S4_H_VS1_Bool1" )
      I_Contact( "Cnv2_S4_H_VS1_Bool2" )
      Move(in := 1, out1 => "Cnv2".Sect4.H.I_RFID_1)
   END_RUNG
   RUNG wire#powerrail
      I_Contact( "Cnv2_S4_H_VS1_Bool0" )
      Contact( "Cnv2_S4_H_VS1_Bool1" )
      I_Contact( "Cnv2_S4_H_VS1_Bool2" )
      Move(in := 2, out1 => "Cnv2".Sect4.H.I_RFID_1)
   END_RUNG
   RUNG wire#powerrail
      I_Contact( "Cnv2_S4_H_VS1_Bool0" )
      I_Contact( "Cnv2_S4_H_VS1_Bool1" )
      I_Contact( "Cnv2_S4_H_VS1_Bool2" )
      Move(in := 0, out1 => "Cnv2".Sect4.H.I_RFID_1)
   END_RUNG
   // the same network as SCL:
   IF "Cnv2_S4_H_VS1_Bool0" AND "Cnv2_S4_H_VS1_Bool1" AND NOT "Cnv2_S4_H_VS1_Bool2" THEN
       "Cnv2".Sect4.H.I_RFID_1 := 3;
   END_IF;
   IF NOT "Cnv2_S4_H_VS1_Bool0" AND NOT "Cnv2_S4_H_VS1_Bool1" AND "Cnv2_S4_H_VS1_Bool2" THEN
       "Cnv2".Sect4.H.I_RFID_1 := 4;
   END_IF;
   IF "Cnv2_S4_H_VS1_Bool0" AND NOT "Cnv2_S4_H_VS1_Bool1" AND NOT "Cnv2_S4_H_VS1_Bool2" THEN
       "Cnv2".Sect4.H.I_RFID_1 := 1;
   END_IF;
   IF NOT "Cnv2_S4_H_VS1_Bool0" AND "Cnv2_S4_H_VS1_Bool1" AND NOT "Cnv2_S4_H_VS1_Bool2" THEN
       "Cnv2".Sect4.H.I_RFID_1 := 2;
   END_IF;
   IF NOT "Cnv2_S4_H_VS1_Bool0" AND NOT "Cnv2_S4_H_VS1_Bool1" AND NOT "Cnv2_S4_H_VS1_Bool2" THEN
       "Cnv2".Sect4.H.I_RFID_1 := 0;
   END_IF;
END_REGION

REGION Network 14: Read RFID sect 4H - 2
   RUNG wire#powerrail
      Contact( "Cnv2_S4_H_VS2_Bool0" )
      Contact( "Cnv2_S4_H_VS2_Bool1" )
      I_Contact( "Cnv2_S4_H_VS2_Bool2" )
      Move(in := 3, out1 => "Cnv2".Sect4.H.I_RFID_2)
   END_RUNG
   RUNG wire#powerrail
      I_Contact( "Cnv2_S4_H_VS2_Bool0" )
      I_Contact( "Cnv2_S4_H_VS2_Bool1" )
      Contact( "Cnv2_S4_H_VS2_Bool2" )
      Move(in := 4, out1 => "Cnv2".Sect4.H.I_RFID_2)
   END_RUNG
   RUNG wire#powerrail
      Contact( "Cnv2_S4_H_VS2_Bool0" )
      I_Contact( "Cnv2_S4_H_VS2_Bool1" )
      I_Contact( "Cnv2_S4_H_VS2_Bool2" )
      Move(in := 1, out1 => "Cnv2".Sect4.H.I_RFID_2)
   END_RUNG
   RUNG wire#powerrail
      I_Contact( "Cnv2_S4_H_VS2_Bool0" )
      Contact( "Cnv2_S4_H_VS2_Bool1" )
      I_Contact( "Cnv2_S4_H_VS2_Bool2" )
      Move(in := 2, out1 => "Cnv2".Sect4.H.I_RFID_2)
   END_RUNG
   RUNG wire#powerrail
      I_Contact( "Cnv2_S4_H_VS2_Bool0" )
      I_Contact( "Cnv2_S4_H_VS2_Bool1" )
      I_Contact( "Cnv2_S4_H_VS2_Bool2" )
      Move(in := 0, out1 => "Cnv2".Sect4.H.I_RFID_2)
   END_RUNG
   // the same network as SCL:
   IF "Cnv2_S4_H_VS2_Bool0" AND "Cnv2_S4_H_VS2_Bool1" AND NOT "Cnv2_S4_H_VS2_Bool2" THEN
       "Cnv2".Sect4.H.I_RFID_2 := 3;
   END_IF;
   IF NOT "Cnv2_S4_H_VS2_Bool0" AND NOT "Cnv2_S4_H_VS2_Bool1" AND "Cnv2_S4_H_VS2_Bool2" THEN
       "Cnv2".Sect4.H.I_RFID_2 := 4;
   END_IF;
   IF "Cnv2_S4_H_VS2_Bool0" AND NOT "Cnv2_S4_H_VS2_Bool1" AND NOT "Cnv2_S4_H_VS2_Bool2" THEN
       "Cnv2".Sect4.H.I_RFID_2 := 1;
   END_IF;
   IF NOT "Cnv2_S4_H_VS2_Bool0" AND "Cnv2_S4_H_VS2_Bool1" AND NOT "Cnv2_S4_H_VS2_Bool2" THEN
       "Cnv2".Sect4.H.I_RFID_2 := 2;
   END_IF;
   IF NOT "Cnv2_S4_H_VS2_Bool0" AND NOT "Cnv2_S4_H_VS2_Bool1" AND NOT "Cnv2_S4_H_VS2_Bool2" THEN
       "Cnv2".Sect4.H.I_RFID_2 := 0;
   END_IF;
END_REGION

REGION Network 15: Read RFID sect 4L - 1
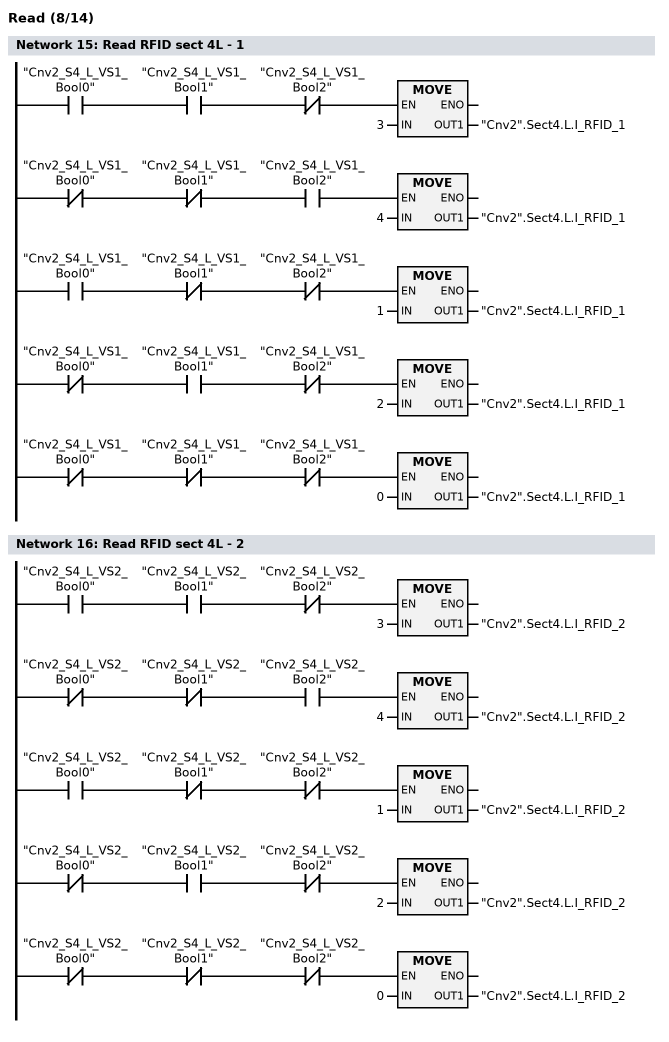
   RUNG wire#powerrail
      Contact( "Cnv2_S4_L_VS1_Bool0" )
      Contact( "Cnv2_S4_L_VS1_Bool1" )
      I_Contact( "Cnv2_S4_L_VS1_Bool2" )
      Move(in := 3, out1 => "Cnv2".Sect4.L.I_RFID_1)
   END_RUNG
   RUNG wire#powerrail
      I_Contact( "Cnv2_S4_L_VS1_Bool0" )
      I_Contact( "Cnv2_S4_L_VS1_Bool1" )
      Contact( "Cnv2_S4_L_VS1_Bool2" )
      Move(in := 4, out1 => "Cnv2".Sect4.L.I_RFID_1)
   END_RUNG
   RUNG wire#powerrail
      Contact( "Cnv2_S4_L_VS1_Bool0" )
      I_Contact( "Cnv2_S4_L_VS1_Bool1" )
      I_Contact( "Cnv2_S4_L_VS1_Bool2" )
      Move(in := 1, out1 => "Cnv2".Sect4.L.I_RFID_1)
   END_RUNG
   RUNG wire#powerrail
      I_Contact( "Cnv2_S4_L_VS1_Bool0" )
      Contact( "Cnv2_S4_L_VS1_Bool1" )
      I_Contact( "Cnv2_S4_L_VS1_Bool2" )
      Move(in := 2, out1 => "Cnv2".Sect4.L.I_RFID_1)
   END_RUNG
   RUNG wire#powerrail
      I_Contact( "Cnv2_S4_L_VS1_Bool0" )
      I_Contact( "Cnv2_S4_L_VS1_Bool1" )
      I_Contact( "Cnv2_S4_L_VS1_Bool2" )
      Move(in := 0, out1 => "Cnv2".Sect4.L.I_RFID_1)
   END_RUNG
   // the same network as SCL:
   IF "Cnv2_S4_L_VS1_Bool0" AND "Cnv2_S4_L_VS1_Bool1" AND NOT "Cnv2_S4_L_VS1_Bool2" THEN
       "Cnv2".Sect4.L.I_RFID_1 := 3;
   END_IF;
   IF NOT "Cnv2_S4_L_VS1_Bool0" AND NOT "Cnv2_S4_L_VS1_Bool1" AND "Cnv2_S4_L_VS1_Bool2" THEN
       "Cnv2".Sect4.L.I_RFID_1 := 4;
   END_IF;
   IF "Cnv2_S4_L_VS1_Bool0" AND NOT "Cnv2_S4_L_VS1_Bool1" AND NOT "Cnv2_S4_L_VS1_Bool2" THEN
       "Cnv2".Sect4.L.I_RFID_1 := 1;
   END_IF;
   IF NOT "Cnv2_S4_L_VS1_Bool0" AND "Cnv2_S4_L_VS1_Bool1" AND NOT "Cnv2_S4_L_VS1_Bool2" THEN
       "Cnv2".Sect4.L.I_RFID_1 := 2;
   END_IF;
   IF NOT "Cnv2_S4_L_VS1_Bool0" AND NOT "Cnv2_S4_L_VS1_Bool1" AND NOT "Cnv2_S4_L_VS1_Bool2" THEN
       "Cnv2".Sect4.L.I_RFID_1 := 0;
   END_IF;
END_REGION

REGION Network 16: Read RFID sect 4L - 2
   RUNG wire#powerrail
      Contact( "Cnv2_S4_L_VS2_Bool0" )
      Contact( "Cnv2_S4_L_VS2_Bool1" )
      I_Contact( "Cnv2_S4_L_VS2_Bool2" )
      Move(in := 3, out1 => "Cnv2".Sect4.L.I_RFID_2)
   END_RUNG
   RUNG wire#powerrail
      I_Contact( "Cnv2_S4_L_VS2_Bool0" )
      I_Contact( "Cnv2_S4_L_VS2_Bool1" )
      Contact( "Cnv2_S4_L_VS2_Bool2" )
      Move(in := 4, out1 => "Cnv2".Sect4.L.I_RFID_2)
   END_RUNG
   RUNG wire#powerrail
      Contact( "Cnv2_S4_L_VS2_Bool0" )
      I_Contact( "Cnv2_S4_L_VS2_Bool1" )
      I_Contact( "Cnv2_S4_L_VS2_Bool2" )
      Move(in := 1, out1 => "Cnv2".Sect4.L.I_RFID_2)
   END_RUNG
   RUNG wire#powerrail
      I_Contact( "Cnv2_S4_L_VS2_Bool0" )
      Contact( "Cnv2_S4_L_VS2_Bool1" )
      I_Contact( "Cnv2_S4_L_VS2_Bool2" )
      Move(in := 2, out1 => "Cnv2".Sect4.L.I_RFID_2)
   END_RUNG
   RUNG wire#powerrail
      I_Contact( "Cnv2_S4_L_VS2_Bool0" )
      I_Contact( "Cnv2_S4_L_VS2_Bool1" )
      I_Contact( "Cnv2_S4_L_VS2_Bool2" )
      Move(in := 0, out1 => "Cnv2".Sect4.L.I_RFID_2)
   END_RUNG
   // the same network as SCL:
   IF "Cnv2_S4_L_VS2_Bool0" AND "Cnv2_S4_L_VS2_Bool1" AND NOT "Cnv2_S4_L_VS2_Bool2" THEN
       "Cnv2".Sect4.L.I_RFID_2 := 3;
   END_IF;
   IF NOT "Cnv2_S4_L_VS2_Bool0" AND NOT "Cnv2_S4_L_VS2_Bool1" AND "Cnv2_S4_L_VS2_Bool2" THEN
       "Cnv2".Sect4.L.I_RFID_2 := 4;
   END_IF;
   IF "Cnv2_S4_L_VS2_Bool0" AND NOT "Cnv2_S4_L_VS2_Bool1" AND NOT "Cnv2_S4_L_VS2_Bool2" THEN
       "Cnv2".Sect4.L.I_RFID_2 := 1;
   END_IF;
   IF NOT "Cnv2_S4_L_VS2_Bool0" AND "Cnv2_S4_L_VS2_Bool1" AND NOT "Cnv2_S4_L_VS2_Bool2" THEN
       "Cnv2".Sect4.L.I_RFID_2 := 2;
   END_IF;
   IF NOT "Cnv2_S4_L_VS2_Bool0" AND NOT "Cnv2_S4_L_VS2_Bool1" AND NOT "Cnv2_S4_L_VS2_Bool2" THEN
       "Cnv2".Sect4.L.I_RFID_2 := 0;
   END_IF;
END_REGION

REGION Network 17: Read RFID sect 0B - 1
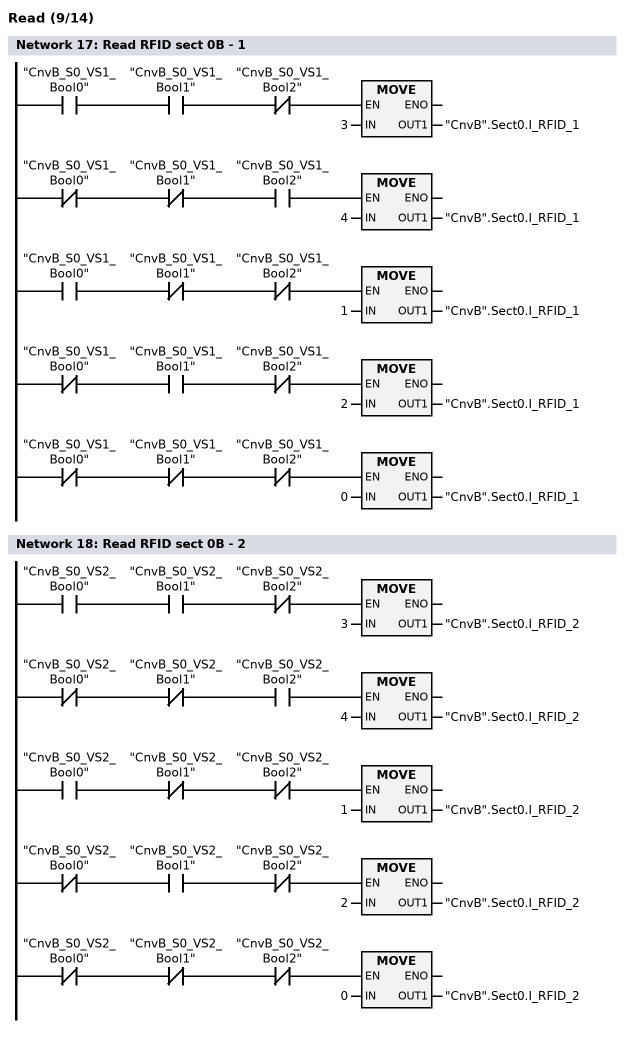
   RUNG wire#powerrail
      Contact( "CnvB_S0_VS1_Bool0" )
      Contact( "CnvB_S0_VS1_Bool1" )
      I_Contact( "CnvB_S0_VS1_Bool2" )
      Move(in := 3, out1 => "CnvB".Sect0.I_RFID_1)
   END_RUNG
   RUNG wire#powerrail
      I_Contact( "CnvB_S0_VS1_Bool0" )
      I_Contact( "CnvB_S0_VS1_Bool1" )
      Contact( "CnvB_S0_VS1_Bool2" )
      Move(in := 4, out1 => "CnvB".Sect0.I_RFID_1)
   END_RUNG
   RUNG wire#powerrail
      Contact( "CnvB_S0_VS1_Bool0" )
      I_Contact( "CnvB_S0_VS1_Bool1" )
      I_Contact( "CnvB_S0_VS1_Bool2" )
      Move(in := 1, out1 => "CnvB".Sect0.I_RFID_1)
   END_RUNG
   RUNG wire#powerrail
      I_Contact( "CnvB_S0_VS1_Bool0" )
      Contact( "CnvB_S0_VS1_Bool1" )
      I_Contact( "CnvB_S0_VS1_Bool2" )
      Move(in := 2, out1 => "CnvB".Sect0.I_RFID_1)
   END_RUNG
   RUNG wire#powerrail
      I_Contact( "CnvB_S0_VS1_Bool0" )
      I_Contact( "CnvB_S0_VS1_Bool1" )
      I_Contact( "CnvB_S0_VS1_Bool2" )
      Move(in := 0, out1 => "CnvB".Sect0.I_RFID_1)
   END_RUNG
   // the same network as SCL:
   IF "CnvB_S0_VS1_Bool0" AND "CnvB_S0_VS1_Bool1" AND NOT "CnvB_S0_VS1_Bool2" THEN
       "CnvB".Sect0.I_RFID_1 := 3;
   END_IF;
   IF NOT "CnvB_S0_VS1_Bool0" AND NOT "CnvB_S0_VS1_Bool1" AND "CnvB_S0_VS1_Bool2" THEN
       "CnvB".Sect0.I_RFID_1 := 4;
   END_IF;
   IF "CnvB_S0_VS1_Bool0" AND NOT "CnvB_S0_VS1_Bool1" AND NOT "CnvB_S0_VS1_Bool2" THEN
       "CnvB".Sect0.I_RFID_1 := 1;
   END_IF;
   IF NOT "CnvB_S0_VS1_Bool0" AND "CnvB_S0_VS1_Bool1" AND NOT "CnvB_S0_VS1_Bool2" THEN
       "CnvB".Sect0.I_RFID_1 := 2;
   END_IF;
   IF NOT "CnvB_S0_VS1_Bool0" AND NOT "CnvB_S0_VS1_Bool1" AND NOT "CnvB_S0_VS1_Bool2" THEN
       "CnvB".Sect0.I_RFID_1 := 0;
   END_IF;
END_REGION

REGION Network 18: Read RFID sect 0B - 2
   RUNG wire#powerrail
      Contact( "CnvB_S0_VS2_Bool0" )
      Contact( "CnvB_S0_VS2_Bool1" )
      I_Contact( "CnvB_S0_VS2_Bool2" )
      Move(in := 3, out1 => "CnvB".Sect0.I_RFID_2)
   END_RUNG
   RUNG wire#powerrail
      I_Contact( "CnvB_S0_VS2_Bool0" )
      I_Contact( "CnvB_S0_VS2_Bool1" )
      Contact( "CnvB_S0_VS2_Bool2" )
      Move(in := 4, out1 => "CnvB".Sect0.I_RFID_2)
   END_RUNG
   RUNG wire#powerrail
      Contact( "CnvB_S0_VS2_Bool0" )
      I_Contact( "CnvB_S0_VS2_Bool1" )
      I_Contact( "CnvB_S0_VS2_Bool2" )
      Move(in := 1, out1 => "CnvB".Sect0.I_RFID_2)
   END_RUNG
   RUNG wire#powerrail
      I_Contact( "CnvB_S0_VS2_Bool0" )
      Contact( "CnvB_S0_VS2_Bool1" )
      I_Contact( "CnvB_S0_VS2_Bool2" )
      Move(in := 2, out1 => "CnvB".Sect0.I_RFID_2)
   END_RUNG
   RUNG wire#powerrail
      I_Contact( "CnvB_S0_VS2_Bool0" )
      I_Contact( "CnvB_S0_VS2_Bool1" )
      I_Contact( "CnvB_S0_VS2_Bool2" )
      Move(in := 0, out1 => "CnvB".Sect0.I_RFID_2)
   END_RUNG
   // the same network as SCL:
   IF "CnvB_S0_VS2_Bool0" AND "CnvB_S0_VS2_Bool1" AND NOT "CnvB_S0_VS2_Bool2" THEN
       "CnvB".Sect0.I_RFID_2 := 3;
   END_IF;
   IF NOT "CnvB_S0_VS2_Bool0" AND NOT "CnvB_S0_VS2_Bool1" AND "CnvB_S0_VS2_Bool2" THEN
       "CnvB".Sect0.I_RFID_2 := 4;
   END_IF;
   IF "CnvB_S0_VS2_Bool0" AND NOT "CnvB_S0_VS2_Bool1" AND NOT "CnvB_S0_VS2_Bool2" THEN
       "CnvB".Sect0.I_RFID_2 := 1;
   END_IF;
   IF NOT "CnvB_S0_VS2_Bool0" AND "CnvB_S0_VS2_Bool1" AND NOT "CnvB_S0_VS2_Bool2" THEN
       "CnvB".Sect0.I_RFID_2 := 2;
   END_IF;
   IF NOT "CnvB_S0_VS2_Bool0" AND NOT "CnvB_S0_VS2_Bool1" AND NOT "CnvB_S0_VS2_Bool2" THEN
       "CnvB".Sect0.I_RFID_2 := 0;
   END_IF;
END_REGION

REGION Network 19: Read RFID sect 1B - 1
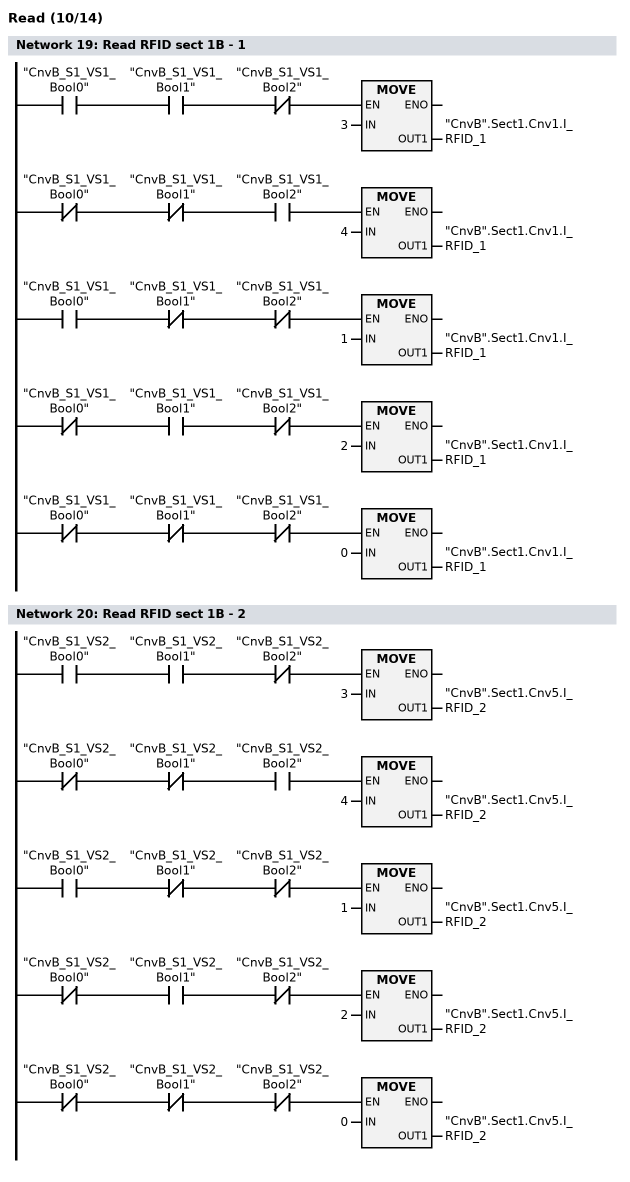
   RUNG wire#powerrail
      Contact( "CnvB_S1_VS1_Bool0" )
      Contact( "CnvB_S1_VS1_Bool1" )
      I_Contact( "CnvB_S1_VS1_Bool2" )
      Move(in := 3, out1 => "CnvB".Sect1.Cnv1.I_RFID_1)
   END_RUNG
   RUNG wire#powerrail
      I_Contact( "CnvB_S1_VS1_Bool0" )
      I_Contact( "CnvB_S1_VS1_Bool1" )
      Contact( "CnvB_S1_VS1_Bool2" )
      Move(in := 4, out1 => "CnvB".Sect1.Cnv1.I_RFID_1)
   END_RUNG
   RUNG wire#powerrail
      Contact( "CnvB_S1_VS1_Bool0" )
      I_Contact( "CnvB_S1_VS1_Bool1" )
      I_Contact( "CnvB_S1_VS1_Bool2" )
      Move(in := 1, out1 => "CnvB".Sect1.Cnv1.I_RFID_1)
   END_RUNG
   RUNG wire#powerrail
      I_Contact( "CnvB_S1_VS1_Bool0" )
      Contact( "CnvB_S1_VS1_Bool1" )
      I_Contact( "CnvB_S1_VS1_Bool2" )
      Move(in := 2, out1 => "CnvB".Sect1.Cnv1.I_RFID_1)
   END_RUNG
   RUNG wire#powerrail
      I_Contact( "CnvB_S1_VS1_Bool0" )
      I_Contact( "CnvB_S1_VS1_Bool1" )
      I_Contact( "CnvB_S1_VS1_Bool2" )
      Move(in := 0, out1 => "CnvB".Sect1.Cnv1.I_RFID_1)
   END_RUNG
   // the same network as SCL:
   IF "CnvB_S1_VS1_Bool0" AND "CnvB_S1_VS1_Bool1" AND NOT "CnvB_S1_VS1_Bool2" THEN
       "CnvB".Sect1.Cnv1.I_RFID_1 := 3;
   END_IF;
   IF NOT "CnvB_S1_VS1_Bool0" AND NOT "CnvB_S1_VS1_Bool1" AND "CnvB_S1_VS1_Bool2" THEN
       "CnvB".Sect1.Cnv1.I_RFID_1 := 4;
   END_IF;
   IF "CnvB_S1_VS1_Bool0" AND NOT "CnvB_S1_VS1_Bool1" AND NOT "CnvB_S1_VS1_Bool2" THEN
       "CnvB".Sect1.Cnv1.I_RFID_1 := 1;
   END_IF;
   IF NOT "CnvB_S1_VS1_Bool0" AND "CnvB_S1_VS1_Bool1" AND NOT "CnvB_S1_VS1_Bool2" THEN
       "CnvB".Sect1.Cnv1.I_RFID_1 := 2;
   END_IF;
   IF NOT "CnvB_S1_VS1_Bool0" AND NOT "CnvB_S1_VS1_Bool1" AND NOT "CnvB_S1_VS1_Bool2" THEN
       "CnvB".Sect1.Cnv1.I_RFID_1 := 0;
   END_IF;
END_REGION

REGION Network 20: Read RFID sect 1B - 2
   RUNG wire#powerrail
      Contact( "CnvB_S1_VS2_Bool0" )
      Contact( "CnvB_S1_VS2_Bool1" )
      I_Contact( "CnvB_S1_VS2_Bool2" )
      Move(in := 3, out1 => "CnvB".Sect1.Cnv5.I_RFID_2)
   END_RUNG
   RUNG wire#powerrail
      I_Contact( "CnvB_S1_VS2_Bool0" )
      I_Contact( "CnvB_S1_VS2_Bool1" )
      Contact( "CnvB_S1_VS2_Bool2" )
      Move(in := 4, out1 => "CnvB".Sect1.Cnv5.I_RFID_2)
   END_RUNG
   RUNG wire#powerrail
      Contact( "CnvB_S1_VS2_Bool0" )
      I_Contact( "CnvB_S1_VS2_Bool1" )
      I_Contact( "CnvB_S1_VS2_Bool2" )
      Move(in := 1, out1 => "CnvB".Sect1.Cnv5.I_RFID_2)
   END_RUNG
   RUNG wire#powerrail
      I_Contact( "CnvB_S1_VS2_Bool0" )
      Contact( "CnvB_S1_VS2_Bool1" )
      I_Contact( "CnvB_S1_VS2_Bool2" )
      Move(in := 2, out1 => "CnvB".Sect1.Cnv5.I_RFID_2)
   END_RUNG
   RUNG wire#powerrail
      I_Contact( "CnvB_S1_VS2_Bool0" )
      I_Contact( "CnvB_S1_VS2_Bool1" )
      I_Contact( "CnvB_S1_VS2_Bool2" )
      Move(in := 0, out1 => "CnvB".Sect1.Cnv5.I_RFID_2)
   END_RUNG
   // the same network as SCL:
   IF "CnvB_S1_VS2_Bool0" AND "CnvB_S1_VS2_Bool1" AND NOT "CnvB_S1_VS2_Bool2" THEN
       "CnvB".Sect1.Cnv5.I_RFID_2 := 3;
   END_IF;
   IF NOT "CnvB_S1_VS2_Bool0" AND NOT "CnvB_S1_VS2_Bool1" AND "CnvB_S1_VS2_Bool2" THEN
       "CnvB".Sect1.Cnv5.I_RFID_2 := 4;
   END_IF;
   IF "CnvB_S1_VS2_Bool0" AND NOT "CnvB_S1_VS2_Bool1" AND NOT "CnvB_S1_VS2_Bool2" THEN
       "CnvB".Sect1.Cnv5.I_RFID_2 := 1;
   END_IF;
   IF NOT "CnvB_S1_VS2_Bool0" AND "CnvB_S1_VS2_Bool1" AND NOT "CnvB_S1_VS2_Bool2" THEN
       "CnvB".Sect1.Cnv5.I_RFID_2 := 2;
   END_IF;
   IF NOT "CnvB_S1_VS2_Bool0" AND NOT "CnvB_S1_VS2_Bool1" AND NOT "CnvB_S1_VS2_Bool2" THEN
       "CnvB".Sect1.Cnv5.I_RFID_2 := 0;
   END_IF;
END_REGION

REGION Network 21: Read RFID sect 2-1B - 1
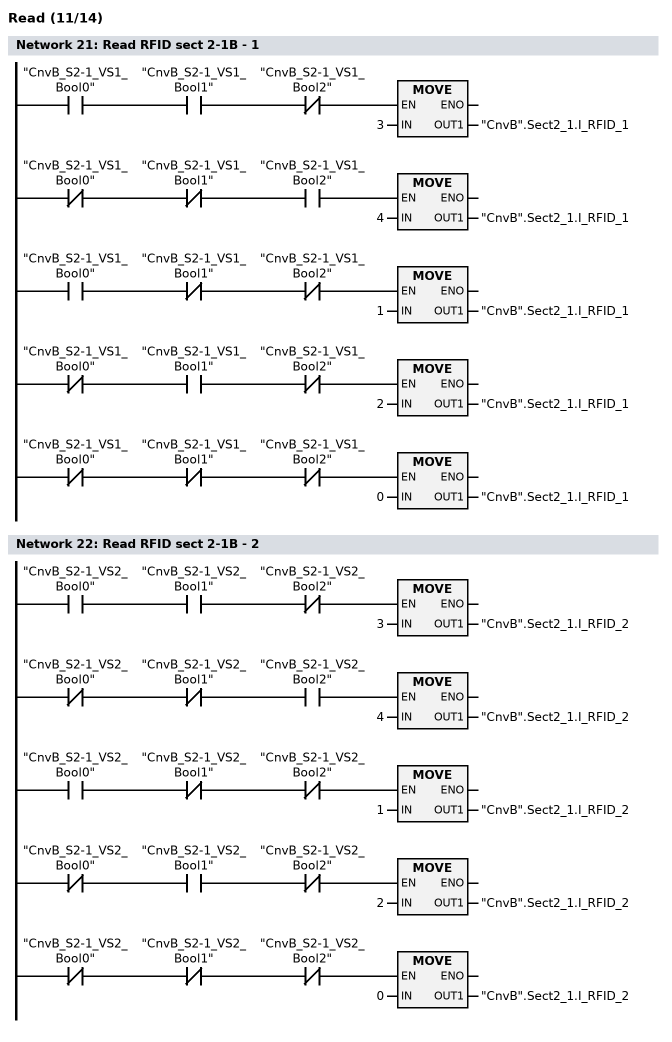
   RUNG wire#powerrail
      Contact( "CnvB_S2-1_VS1_Bool0" )
      Contact( "CnvB_S2-1_VS1_Bool1" )
      I_Contact( "CnvB_S2-1_VS1_Bool2" )
      Move(in := 3, out1 => "CnvB".Sect2_1.I_RFID_1)
   END_RUNG
   RUNG wire#powerrail
      I_Contact( "CnvB_S2-1_VS1_Bool0" )
      I_Contact( "CnvB_S2-1_VS1_Bool1" )
      Contact( "CnvB_S2-1_VS1_Bool2" )
      Move(in := 4, out1 => "CnvB".Sect2_1.I_RFID_1)
   END_RUNG
   RUNG wire#powerrail
      Contact( "CnvB_S2-1_VS1_Bool0" )
      I_Contact( "CnvB_S2-1_VS1_Bool1" )
      I_Contact( "CnvB_S2-1_VS1_Bool2" )
      Move(in := 1, out1 => "CnvB".Sect2_1.I_RFID_1)
   END_RUNG
   RUNG wire#powerrail
      I_Contact( "CnvB_S2-1_VS1_Bool0" )
      Contact( "CnvB_S2-1_VS1_Bool1" )
      I_Contact( "CnvB_S2-1_VS1_Bool2" )
      Move(in := 2, out1 => "CnvB".Sect2_1.I_RFID_1)
   END_RUNG
   RUNG wire#powerrail
      I_Contact( "CnvB_S2-1_VS1_Bool0" )
      I_Contact( "CnvB_S2-1_VS1_Bool1" )
      I_Contact( "CnvB_S2-1_VS1_Bool2" )
      Move(in := 0, out1 => "CnvB".Sect2_1.I_RFID_1)
   END_RUNG
   // the same network as SCL:
   IF "CnvB_S2-1_VS1_Bool0" AND "CnvB_S2-1_VS1_Bool1" AND NOT "CnvB_S2-1_VS1_Bool2" THEN
       "CnvB".Sect2_1.I_RFID_1 := 3;
   END_IF;
   IF NOT "CnvB_S2-1_VS1_Bool0" AND NOT "CnvB_S2-1_VS1_Bool1" AND "CnvB_S2-1_VS1_Bool2" THEN
       "CnvB".Sect2_1.I_RFID_1 := 4;
   END_IF;
   IF "CnvB_S2-1_VS1_Bool0" AND NOT "CnvB_S2-1_VS1_Bool1" AND NOT "CnvB_S2-1_VS1_Bool2" THEN
       "CnvB".Sect2_1.I_RFID_1 := 1;
   END_IF;
   IF NOT "CnvB_S2-1_VS1_Bool0" AND "CnvB_S2-1_VS1_Bool1" AND NOT "CnvB_S2-1_VS1_Bool2" THEN
       "CnvB".Sect2_1.I_RFID_1 := 2;
   END_IF;
   IF NOT "CnvB_S2-1_VS1_Bool0" AND NOT "CnvB_S2-1_VS1_Bool1" AND NOT "CnvB_S2-1_VS1_Bool2" THEN
       "CnvB".Sect2_1.I_RFID_1 := 0;
   END_IF;
END_REGION

REGION Network 22: Read RFID sect 2-1B - 2
   RUNG wire#powerrail
      Contact( "CnvB_S2-1_VS2_Bool0" )
      Contact( "CnvB_S2-1_VS2_Bool1" )
      I_Contact( "CnvB_S2-1_VS2_Bool2" )
      Move(in := 3, out1 => "CnvB".Sect2_1.I_RFID_2)
   END_RUNG
   RUNG wire#powerrail
      I_Contact( "CnvB_S2-1_VS2_Bool0" )
      I_Contact( "CnvB_S2-1_VS2_Bool1" )
      Contact( "CnvB_S2-1_VS2_Bool2" )
      Move(in := 4, out1 => "CnvB".Sect2_1.I_RFID_2)
   END_RUNG
   RUNG wire#powerrail
      Contact( "CnvB_S2-1_VS2_Bool0" )
      I_Contact( "CnvB_S2-1_VS2_Bool1" )
      I_Contact( "CnvB_S2-1_VS2_Bool2" )
      Move(in := 1, out1 => "CnvB".Sect2_1.I_RFID_2)
   END_RUNG
   RUNG wire#powerrail
      I_Contact( "CnvB_S2-1_VS2_Bool0" )
      Contact( "CnvB_S2-1_VS2_Bool1" )
      I_Contact( "CnvB_S2-1_VS2_Bool2" )
      Move(in := 2, out1 => "CnvB".Sect2_1.I_RFID_2)
   END_RUNG
   RUNG wire#powerrail
      I_Contact( "CnvB_S2-1_VS2_Bool0" )
      I_Contact( "CnvB_S2-1_VS2_Bool1" )
      I_Contact( "CnvB_S2-1_VS2_Bool2" )
      Move(in := 0, out1 => "CnvB".Sect2_1.I_RFID_2)
   END_RUNG
   // the same network as SCL:
   IF "CnvB_S2-1_VS2_Bool0" AND "CnvB_S2-1_VS2_Bool1" AND NOT "CnvB_S2-1_VS2_Bool2" THEN
       "CnvB".Sect2_1.I_RFID_2 := 3;
   END_IF;
   IF NOT "CnvB_S2-1_VS2_Bool0" AND NOT "CnvB_S2-1_VS2_Bool1" AND "CnvB_S2-1_VS2_Bool2" THEN
       "CnvB".Sect2_1.I_RFID_2 := 4;
   END_IF;
   IF "CnvB_S2-1_VS2_Bool0" AND NOT "CnvB_S2-1_VS2_Bool1" AND NOT "CnvB_S2-1_VS2_Bool2" THEN
       "CnvB".Sect2_1.I_RFID_2 := 1;
   END_IF;
   IF NOT "CnvB_S2-1_VS2_Bool0" AND "CnvB_S2-1_VS2_Bool1" AND NOT "CnvB_S2-1_VS2_Bool2" THEN
       "CnvB".Sect2_1.I_RFID_2 := 2;
   END_IF;
   IF NOT "CnvB_S2-1_VS2_Bool0" AND NOT "CnvB_S2-1_VS2_Bool1" AND NOT "CnvB_S2-1_VS2_Bool2" THEN
       "CnvB".Sect2_1.I_RFID_2 := 0;
   END_IF;
END_REGION

REGION Network 23: Read RFID sect 2-2B - 1
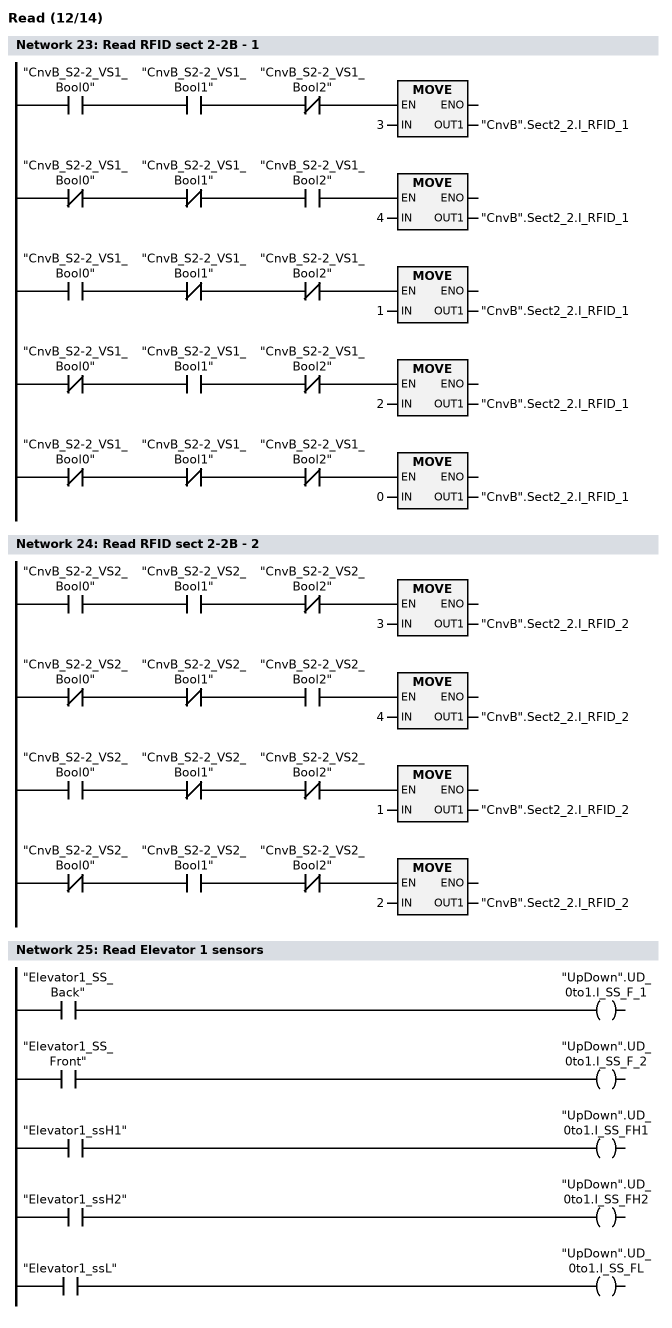
   RUNG wire#powerrail
      Contact( "CnvB_S2-2_VS1_Bool0" )
      Contact( "CnvB_S2-2_VS1_Bool1" )
      I_Contact( "CnvB_S2-2_VS1_Bool2" )
      Move(in := 3, out1 => "CnvB".Sect2_2.I_RFID_1)
   END_RUNG
   RUNG wire#powerrail
      I_Contact( "CnvB_S2-2_VS1_Bool0" )
      I_Contact( "CnvB_S2-2_VS1_Bool1" )
      Contact( "CnvB_S2-2_VS1_Bool2" )
      Move(in := 4, out1 => "CnvB".Sect2_2.I_RFID_1)
   END_RUNG
   RUNG wire#powerrail
      Contact( "CnvB_S2-2_VS1_Bool0" )
      I_Contact( "CnvB_S2-2_VS1_Bool1" )
      I_Contact( "CnvB_S2-2_VS1_Bool2" )
      Move(in := 1, out1 => "CnvB".Sect2_2.I_RFID_1)
   END_RUNG
   RUNG wire#powerrail
      I_Contact( "CnvB_S2-2_VS1_Bool0" )
      Contact( "CnvB_S2-2_VS1_Bool1" )
      I_Contact( "CnvB_S2-2_VS1_Bool2" )
      Move(in := 2, out1 => "CnvB".Sect2_2.I_RFID_1)
   END_RUNG
   RUNG wire#powerrail
      I_Contact( "CnvB_S2-2_VS1_Bool0" )
      I_Contact( "CnvB_S2-2_VS1_Bool1" )
      I_Contact( "CnvB_S2-2_VS1_Bool2" )
      Move(in := 0, out1 => "CnvB".Sect2_2.I_RFID_1)
   END_RUNG
   // the same network as SCL:
   IF "CnvB_S2-2_VS1_Bool0" AND "CnvB_S2-2_VS1_Bool1" AND NOT "CnvB_S2-2_VS1_Bool2" THEN
       "CnvB".Sect2_2.I_RFID_1 := 3;
   END_IF;
   IF NOT "CnvB_S2-2_VS1_Bool0" AND NOT "CnvB_S2-2_VS1_Bool1" AND "CnvB_S2-2_VS1_Bool2" THEN
       "CnvB".Sect2_2.I_RFID_1 := 4;
   END_IF;
   IF "CnvB_S2-2_VS1_Bool0" AND NOT "CnvB_S2-2_VS1_Bool1" AND NOT "CnvB_S2-2_VS1_Bool2" THEN
       "CnvB".Sect2_2.I_RFID_1 := 1;
   END_IF;
   IF NOT "CnvB_S2-2_VS1_Bool0" AND "CnvB_S2-2_VS1_Bool1" AND NOT "CnvB_S2-2_VS1_Bool2" THEN
       "CnvB".Sect2_2.I_RFID_1 := 2;
   END_IF;
   IF NOT "CnvB_S2-2_VS1_Bool0" AND NOT "CnvB_S2-2_VS1_Bool1" AND NOT "CnvB_S2-2_VS1_Bool2" THEN
       "CnvB".Sect2_2.I_RFID_1 := 0;
   END_IF;
END_REGION

REGION Network 24: Read RFID sect 2-2B - 2
   RUNG wire#powerrail
      Contact( "CnvB_S2-2_VS2_Bool0" )
      Contact( "CnvB_S2-2_VS2_Bool1" )
      I_Contact( "CnvB_S2-2_VS2_Bool2" )
      Move(in := 3, out1 => "CnvB".Sect2_2.I_RFID_2)
   END_RUNG
   RUNG wire#powerrail
      I_Contact( "CnvB_S2-2_VS2_Bool0" )
      I_Contact( "CnvB_S2-2_VS2_Bool1" )
      Contact( "CnvB_S2-2_VS2_Bool2" )
      Move(in := 4, out1 => "CnvB".Sect2_2.I_RFID_2)
   END_RUNG
   RUNG wire#powerrail
      Contact( "CnvB_S2-2_VS2_Bool0" )
      I_Contact( "CnvB_S2-2_VS2_Bool1" )
      I_Contact( "CnvB_S2-2_VS2_Bool2" )
      Move(in := 1, out1 => "CnvB".Sect2_2.I_RFID_2)
   END_RUNG
   RUNG wire#powerrail
      I_Contact( "CnvB_S2-2_VS2_Bool0" )
      Contact( "CnvB_S2-2_VS2_Bool1" )
      I_Contact( "CnvB_S2-2_VS2_Bool2" )
      Move(in := 2, out1 => "CnvB".Sect2_2.I_RFID_2)
   END_RUNG
   // the same network as SCL:
   IF "CnvB_S2-2_VS2_Bool0" AND "CnvB_S2-2_VS2_Bool1" AND NOT "CnvB_S2-2_VS2_Bool2" THEN
       "CnvB".Sect2_2.I_RFID_2 := 3;
   END_IF;
   IF NOT "CnvB_S2-2_VS2_Bool0" AND NOT "CnvB_S2-2_VS2_Bool1" AND "CnvB_S2-2_VS2_Bool2" THEN
       "CnvB".Sect2_2.I_RFID_2 := 4;
   END_IF;
   IF "CnvB_S2-2_VS2_Bool0" AND NOT "CnvB_S2-2_VS2_Bool1" AND NOT "CnvB_S2-2_VS2_Bool2" THEN
       "CnvB".Sect2_2.I_RFID_2 := 1;
   END_IF;
   IF NOT "CnvB_S2-2_VS2_Bool0" AND "CnvB_S2-2_VS2_Bool1" AND NOT "CnvB_S2-2_VS2_Bool2" THEN
       "CnvB".Sect2_2.I_RFID_2 := 2;
   END_IF;
END_REGION

REGION Network 25: Read Elevator 1 sensors
   RUNG wire#powerrail
      Contact( "Elevator1_SS_Back" )
      Coil( "UpDown".UD_0to1.I_SS_F_1 )
   END_RUNG
   RUNG wire#powerrail
      Contact( "Elevator1_SS_Front" )
      Coil( "UpDown".UD_0to1.I_SS_F_2 )
   END_RUNG
   RUNG wire#powerrail
      Contact( "Elevator1_ssH1" )
      Coil( "UpDown".UD_0to1.I_SS_FH1 )
   END_RUNG
   RUNG wire#powerrail
      Contact( "Elevator1_ssH2" )
      Coil( "UpDown".UD_0to1.I_SS_FH2 )
   END_RUNG
   RUNG wire#powerrail
      Contact( "Elevator1_ssL" )
      Coil( "UpDown".UD_0to1.I_SS_FL )
   END_RUNG
   // the same network as SCL:
   "UpDown".UD_0to1.I_SS_F_1 := "Elevator1_SS_Back";
   "UpDown".UD_0to1.I_SS_F_2 := "Elevator1_SS_Front";
   "UpDown".UD_0to1.I_SS_FH1 := "Elevator1_ssH1";
   "UpDown".UD_0to1.I_SS_FH2 := "Elevator1_ssH2";
   "UpDown".UD_0to1.I_SS_FL := "Elevator1_ssL";
END_REGION

REGION Network 26: Read Elevator 2 sensors
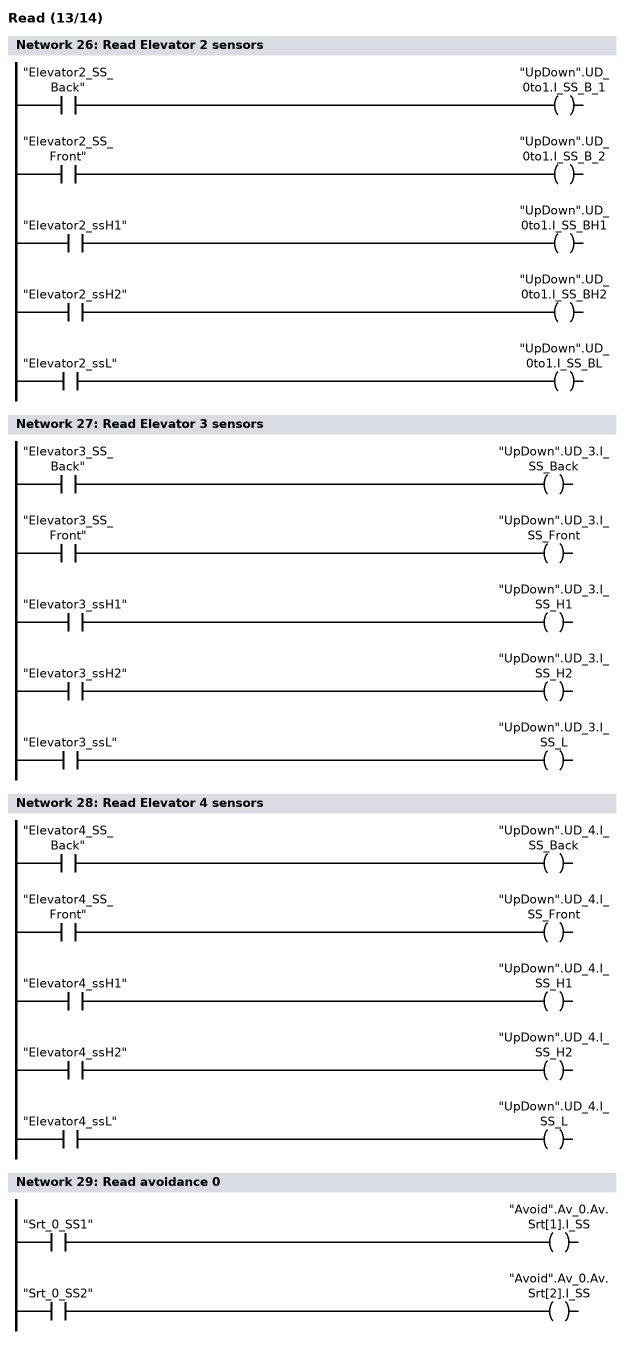
   RUNG wire#powerrail
      Contact( "Elevator2_SS_Back" )
      Coil( "UpDown".UD_0to1.I_SS_B_1 )
   END_RUNG
   RUNG wire#powerrail
      Contact( "Elevator2_SS_Front" )
      Coil( "UpDown".UD_0to1.I_SS_B_2 )
   END_RUNG
   RUNG wire#powerrail
      Contact( "Elevator2_ssH1" )
      Coil( "UpDown".UD_0to1.I_SS_BH1 )
   END_RUNG
   RUNG wire#powerrail
      Contact( "Elevator2_ssH2" )
      Coil( "UpDown".UD_0to1.I_SS_BH2 )
   END_RUNG
   RUNG wire#powerrail
      Contact( "Elevator2_ssL" )
      Coil( "UpDown".UD_0to1.I_SS_BL )
   END_RUNG
   // the same network as SCL:
   "UpDown".UD_0to1.I_SS_B_1 := "Elevator2_SS_Back";
   "UpDown".UD_0to1.I_SS_B_2 := "Elevator2_SS_Front";
   "UpDown".UD_0to1.I_SS_BH1 := "Elevator2_ssH1";
   "UpDown".UD_0to1.I_SS_BH2 := "Elevator2_ssH2";
   "UpDown".UD_0to1.I_SS_BL := "Elevator2_ssL";
END_REGION

REGION Network 27: Read Elevator 3 sensors
   RUNG wire#powerrail
      Contact( "Elevator3_SS_Back" )
      Coil( "UpDown".UD_3.I_SS_Back )
   END_RUNG
   RUNG wire#powerrail
      Contact( "Elevator3_SS_Front" )
      Coil( "UpDown".UD_3.I_SS_Front )
   END_RUNG
   RUNG wire#powerrail
      Contact( "Elevator3_ssH1" )
      Coil( "UpDown".UD_3.I_SS_H1 )
   END_RUNG
   RUNG wire#powerrail
      Contact( "Elevator3_ssH2" )
      Coil( "UpDown".UD_3.I_SS_H2 )
   END_RUNG
   RUNG wire#powerrail
      Contact( "Elevator3_ssL" )
      Coil( "UpDown".UD_3.I_SS_L )
   END_RUNG
   // the same network as SCL:
   "UpDown".UD_3.I_SS_Back := "Elevator3_SS_Back";
   "UpDown".UD_3.I_SS_Front := "Elevator3_SS_Front";
   "UpDown".UD_3.I_SS_H1 := "Elevator3_ssH1";
   "UpDown".UD_3.I_SS_H2 := "Elevator3_ssH2";
   "UpDown".UD_3.I_SS_L := "Elevator3_ssL";
END_REGION

REGION Network 28: Read Elevator 4 sensors
   RUNG wire#powerrail
      Contact( "Elevator4_SS_Back" )
      Coil( "UpDown".UD_4.I_SS_Back )
   END_RUNG
   RUNG wire#powerrail
      Contact( "Elevator4_SS_Front" )
      Coil( "UpDown".UD_4.I_SS_Front )
   END_RUNG
   RUNG wire#powerrail
      Contact( "Elevator4_ssH1" )
      Coil( "UpDown".UD_4.I_SS_H1 )
   END_RUNG
   RUNG wire#powerrail
      Contact( "Elevator4_ssH2" )
      Coil( "UpDown".UD_4.I_SS_H2 )
   END_RUNG
   RUNG wire#powerrail
      Contact( "Elevator4_ssL" )
      Coil( "UpDown".UD_4.I_SS_L )
   END_RUNG
   // the same network as SCL:
   "UpDown".UD_4.I_SS_Back := "Elevator4_SS_Back";
   "UpDown".UD_4.I_SS_Front := "Elevator4_SS_Front";
   "UpDown".UD_4.I_SS_H1 := "Elevator4_ssH1";
   "UpDown".UD_4.I_SS_H2 := "Elevator4_ssH2";
   "UpDown".UD_4.I_SS_L := "Elevator4_ssL";
END_REGION

REGION Network 29: Read avoidance 0
   RUNG wire#powerrail
      Contact( "Srt_0_SS1" )
      Coil( "Avoid".Av_0.Av.Srt[1].I_SS )
   END_RUNG
   RUNG wire#powerrail
      Contact( "Srt_0_SS2" )
      Coil( "Avoid".Av_0.Av.Srt[2].I_SS )
   END_RUNG
   // the same network as SCL:
   "Avoid".Av_0.Av.Srt[1].I_SS := "Srt_0_SS1";
   "Avoid".Av_0.Av.Srt[2].I_SS := "Srt_0_SS2";
END_REGION

REGION Network 30: Read avoidance 1to2
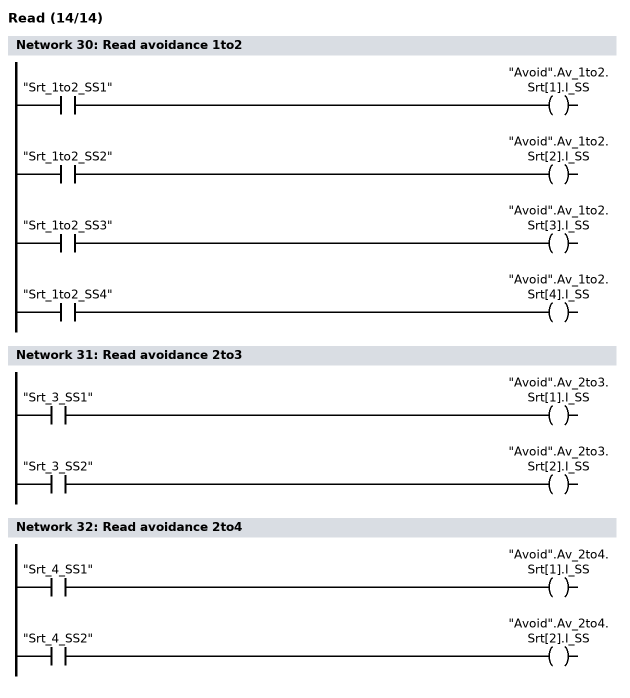
   RUNG wire#powerrail
      Contact( "Srt_1to2_SS1" )
      Coil( "Avoid".Av_1to2.Srt[1].I_SS )
   END_RUNG
   RUNG wire#powerrail
      Contact( "Srt_1to2_SS2" )
      Coil( "Avoid".Av_1to2.Srt[2].I_SS )
   END_RUNG
   RUNG wire#powerrail
      Contact( "Srt_1to2_SS3" )
      Coil( "Avoid".Av_1to2.Srt[3].I_SS )
   END_RUNG
   RUNG wire#powerrail
      Contact( "Srt_1to2_SS4" )
      Coil( "Avoid".Av_1to2.Srt[4].I_SS )
   END_RUNG
   // the same network as SCL:
   "Avoid".Av_1to2.Srt[1].I_SS := "Srt_1to2_SS1";
   "Avoid".Av_1to2.Srt[2].I_SS := "Srt_1to2_SS2";
   "Avoid".Av_1to2.Srt[3].I_SS := "Srt_1to2_SS3";
   "Avoid".Av_1to2.Srt[4].I_SS := "Srt_1to2_SS4";
END_REGION

REGION Network 31: Read avoidance 2to3
   RUNG wire#powerrail
      Contact( "Srt_3_SS1" )
      Coil( "Avoid".Av_2to3.Srt[1].I_SS )
   END_RUNG
   RUNG wire#powerrail
      Contact( "Srt_3_SS2" )
      Coil( "Avoid".Av_2to3.Srt[2].I_SS )
   END_RUNG
   // the same network as SCL:
   "Avoid".Av_2to3.Srt[1].I_SS := "Srt_3_SS1";
   "Avoid".Av_2to3.Srt[2].I_SS := "Srt_3_SS2";
END_REGION

REGION Network 32: Read avoidance 2to4
   RUNG wire#powerrail
      Contact( "Srt_4_SS1" )
      Coil( "Avoid".Av_2to4.Srt[1].I_SS )
   END_RUNG
   RUNG wire#powerrail
      Contact( "Srt_4_SS2" )
      Coil( "Avoid".Av_2to4.Srt[2].I_SS )
   END_RUNG
   // the same network as SCL:
   "Avoid".Av_2to4.Srt[1].I_SS := "Srt_4_SS1";
   "Avoid".Av_2to4.Srt[2].I_SS := "Srt_4_SS2";
END_REGION
END_FUNCTION

FUNCTION "Write" : Void   // FC4, LAD
{ S7_Optimized_Access := 'TRUE' }
VERSION : 0.1
BEGIN

REGION Network 1: Write CnvF
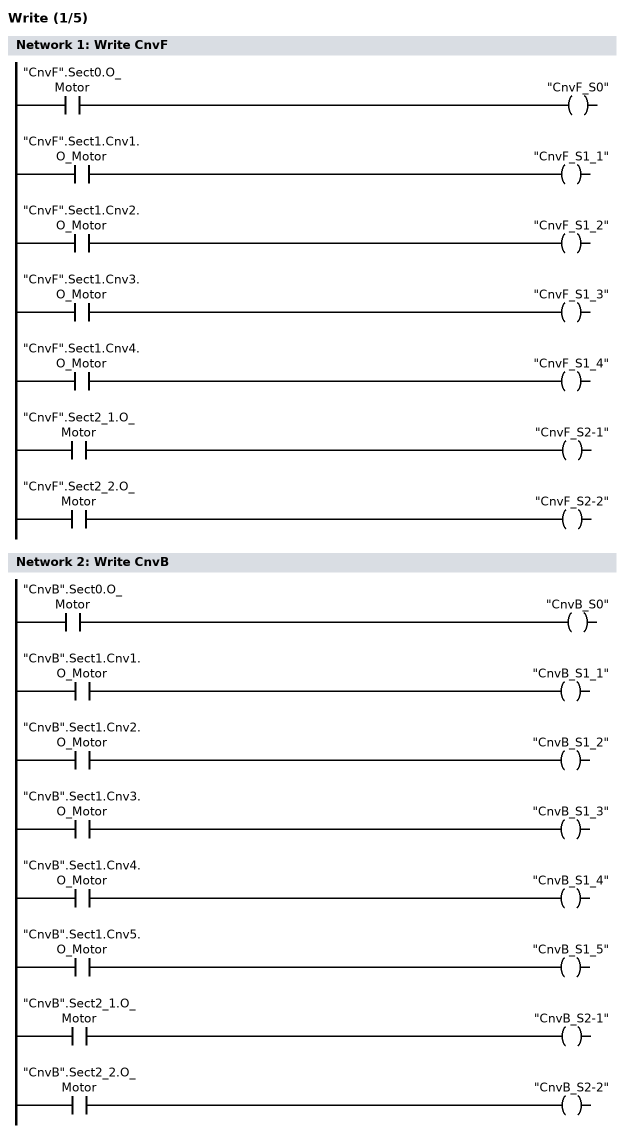
   RUNG wire#powerrail
      Contact( "CnvF".Sect0.O_Motor )
      Coil( "CnvF_S0" )
   END_RUNG
   RUNG wire#powerrail
      Contact( "CnvF".Sect1.Cnv1.O_Motor )
      Coil( "CnvF_S1_1" )
   END_RUNG
   RUNG wire#powerrail
      Contact( "CnvF".Sect1.Cnv2.O_Motor )
      Coil( "CnvF_S1_2" )
   END_RUNG
   RUNG wire#powerrail
      Contact( "CnvF".Sect1.Cnv3.O_Motor )
      Coil( "CnvF_S1_3" )
   END_RUNG
   RUNG wire#powerrail
      Contact( "CnvF".Sect1.Cnv4.O_Motor )
      Coil( "CnvF_S1_4" )
   END_RUNG
   RUNG wire#powerrail
      Contact( "CnvF".Sect2_1.O_Motor )
      Coil( "CnvF_S2-1" )
   END_RUNG
   RUNG wire#powerrail
      Contact( "CnvF".Sect2_2.O_Motor )
      Coil( "CnvF_S2-2" )
   END_RUNG
   // the same network as SCL:
   "CnvF_S0" := "CnvF".Sect0.O_Motor;
   "CnvF_S1_1" := "CnvF".Sect1.Cnv1.O_Motor;
   "CnvF_S1_2" := "CnvF".Sect1.Cnv2.O_Motor;
   "CnvF_S1_3" := "CnvF".Sect1.Cnv3.O_Motor;
   "CnvF_S1_4" := "CnvF".Sect1.Cnv4.O_Motor;
   "CnvF_S2-1" := "CnvF".Sect2_1.O_Motor;
   "CnvF_S2-2" := "CnvF".Sect2_2.O_Motor;
END_REGION

REGION Network 2: Write CnvB
   RUNG wire#powerrail
      Contact( "CnvB".Sect0.O_Motor )
      Coil( "CnvB_S0" )
   END_RUNG
   RUNG wire#powerrail
      Contact( "CnvB".Sect1.Cnv1.O_Motor )
      Coil( "CnvB_S1_1" )
   END_RUNG
   RUNG wire#powerrail
      Contact( "CnvB".Sect1.Cnv2.O_Motor )
      Coil( "CnvB_S1_2" )
   END_RUNG
   RUNG wire#powerrail
      Contact( "CnvB".Sect1.Cnv3.O_Motor )
      Coil( "CnvB_S1_3" )
   END_RUNG
   RUNG wire#powerrail
      Contact( "CnvB".Sect1.Cnv4.O_Motor )
      Coil( "CnvB_S1_4" )
   END_RUNG
   RUNG wire#powerrail
      Contact( "CnvB".Sect1.Cnv5.O_Motor )
      Coil( "CnvB_S1_5" )
   END_RUNG
   RUNG wire#powerrail
      Contact( "CnvB".Sect2_1.O_Motor )
      Coil( "CnvB_S2-1" )
   END_RUNG
   RUNG wire#powerrail
      Contact( "CnvB".Sect2_2.O_Motor )
      Coil( "CnvB_S2-2" )
   END_RUNG
   // the same network as SCL:
   "CnvB_S0" := "CnvB".Sect0.O_Motor;
   "CnvB_S1_1" := "CnvB".Sect1.Cnv1.O_Motor;
   "CnvB_S1_2" := "CnvB".Sect1.Cnv2.O_Motor;
   "CnvB_S1_3" := "CnvB".Sect1.Cnv3.O_Motor;
   "CnvB_S1_4" := "CnvB".Sect1.Cnv4.O_Motor;
   "CnvB_S1_5" := "CnvB".Sect1.Cnv5.O_Motor;
   "CnvB_S2-1" := "CnvB".Sect2_1.O_Motor;
   "CnvB_S2-2" := "CnvB".Sect2_2.O_Motor;
END_REGION

REGION Network 3: Write Cnv2
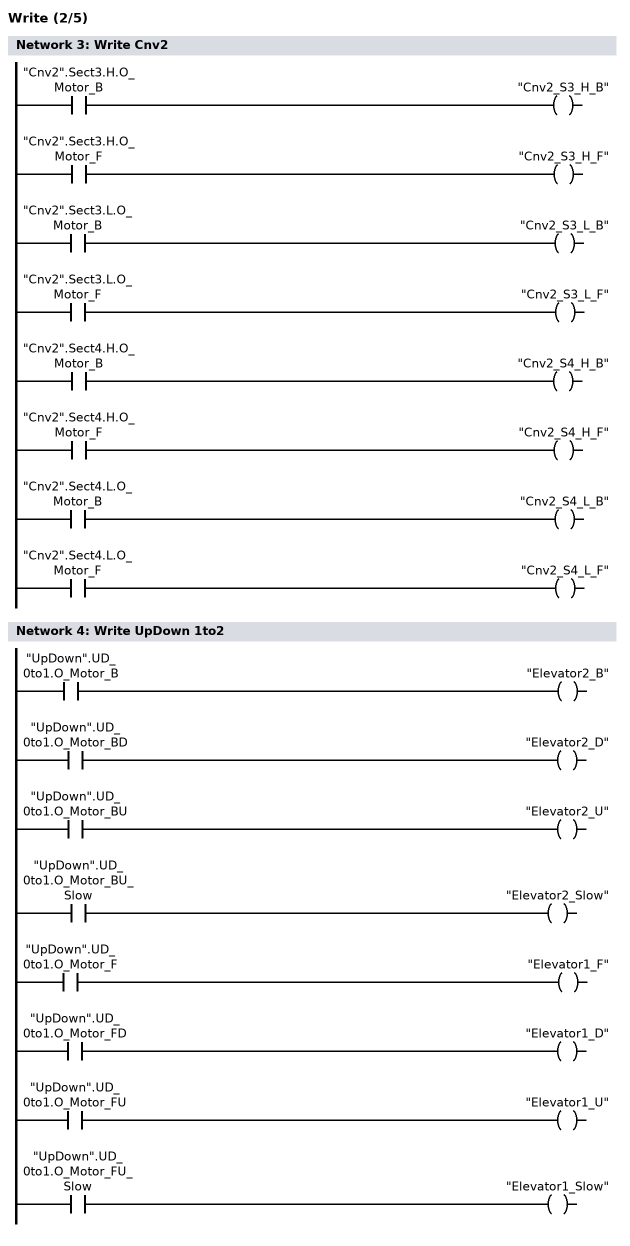
   RUNG wire#powerrail
      Contact( "Cnv2".Sect3.H.O_Motor_B )
      Coil( "Cnv2_S3_H_B" )
   END_RUNG
   RUNG wire#powerrail
      Contact( "Cnv2".Sect3.H.O_Motor_F )
      Coil( "Cnv2_S3_H_F" )
   END_RUNG
   RUNG wire#powerrail
      Contact( "Cnv2".Sect3.L.O_Motor_B )
      Coil( "Cnv2_S3_L_B" )
   END_RUNG
   RUNG wire#powerrail
      Contact( "Cnv2".Sect3.L.O_Motor_F )
      Coil( "Cnv2_S3_L_F" )
   END_RUNG
   RUNG wire#powerrail
      Contact( "Cnv2".Sect4.H.O_Motor_B )
      Coil( "Cnv2_S4_H_B" )
   END_RUNG
   RUNG wire#powerrail
      Contact( "Cnv2".Sect4.H.O_Motor_F )
      Coil( "Cnv2_S4_H_F" )
   END_RUNG
   RUNG wire#powerrail
      Contact( "Cnv2".Sect4.L.O_Motor_B )
      Coil( "Cnv2_S4_L_B" )
   END_RUNG
   RUNG wire#powerrail
      Contact( "Cnv2".Sect4.L.O_Motor_F )
      Coil( "Cnv2_S4_L_F" )
   END_RUNG
   // the same network as SCL:
   "Cnv2_S3_H_B" := "Cnv2".Sect3.H.O_Motor_B;
   "Cnv2_S3_H_F" := "Cnv2".Sect3.H.O_Motor_F;
   "Cnv2_S3_L_B" := "Cnv2".Sect3.L.O_Motor_B;
   "Cnv2_S3_L_F" := "Cnv2".Sect3.L.O_Motor_F;
   "Cnv2_S4_H_B" := "Cnv2".Sect4.H.O_Motor_B;
   "Cnv2_S4_H_F" := "Cnv2".Sect4.H.O_Motor_F;
   "Cnv2_S4_L_B" := "Cnv2".Sect4.L.O_Motor_B;
   "Cnv2_S4_L_F" := "Cnv2".Sect4.L.O_Motor_F;
END_REGION

REGION Network 4: Write UpDown 1to2
   RUNG wire#powerrail
      Contact( "UpDown".UD_0to1.O_Motor_B )
      Coil( "Elevator2_B" )
   END_RUNG
   RUNG wire#powerrail
      Contact( "UpDown".UD_0to1.O_Motor_BD )
      Coil( "Elevator2_D" )
   END_RUNG
   RUNG wire#powerrail
      Contact( "UpDown".UD_0to1.O_Motor_BU )
      Coil( "Elevator2_U" )
   END_RUNG
   RUNG wire#powerrail
      Contact( "UpDown".UD_0to1.O_Motor_BU_Slow )
      Coil( "Elevator2_Slow" )
   END_RUNG
   RUNG wire#powerrail
      Contact( "UpDown".UD_0to1.O_Motor_F )
      Coil( "Elevator1_F" )
   END_RUNG
   RUNG wire#powerrail
      Contact( "UpDown".UD_0to1.O_Motor_FD )
      Coil( "Elevator1_D" )
   END_RUNG
   RUNG wire#powerrail
      Contact( "UpDown".UD_0to1.O_Motor_FU )
      Coil( "Elevator1_U" )
   END_RUNG
   RUNG wire#powerrail
      Contact( "UpDown".UD_0to1.O_Motor_FU_Slow )
      Coil( "Elevator1_Slow" )
   END_RUNG
   // the same network as SCL:
   "Elevator2_B" := "UpDown".UD_0to1.O_Motor_B;
   "Elevator2_D" := "UpDown".UD_0to1.O_Motor_BD;
   "Elevator2_U" := "UpDown".UD_0to1.O_Motor_BU;
   "Elevator2_Slow" := "UpDown".UD_0to1.O_Motor_BU_Slow;
   "Elevator1_F" := "UpDown".UD_0to1.O_Motor_F;
   "Elevator1_D" := "UpDown".UD_0to1.O_Motor_FD;
   "Elevator1_U" := "UpDown".UD_0to1.O_Motor_FU;
   "Elevator1_Slow" := "UpDown".UD_0to1.O_Motor_FU_Slow;
END_REGION

REGION Network 5: Write Elevator 3
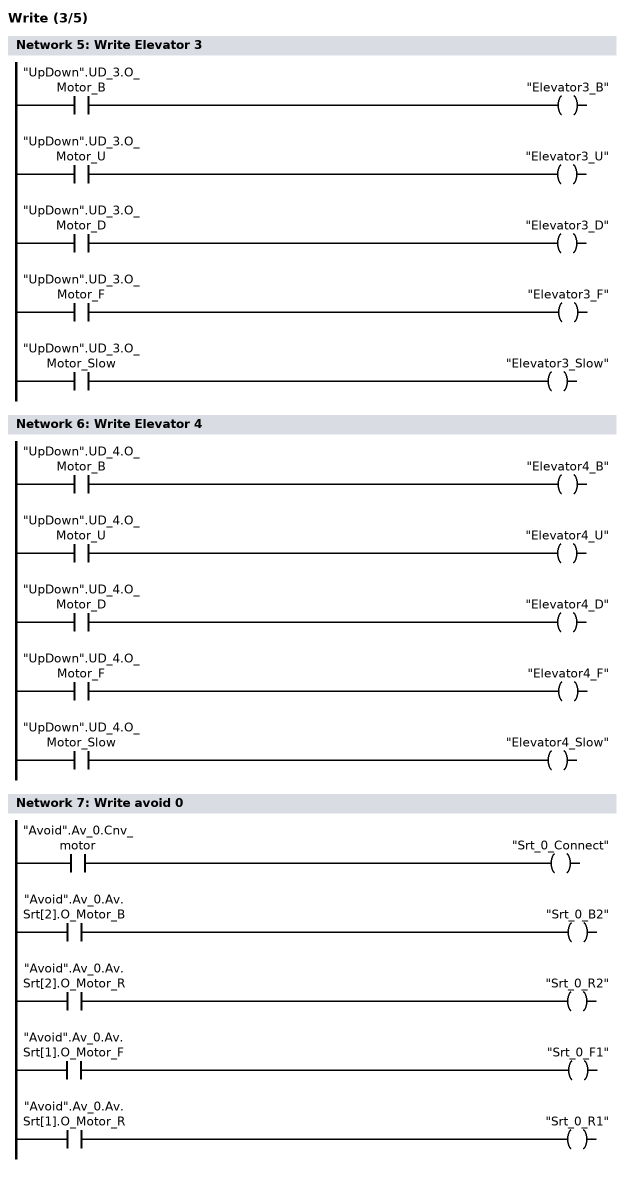
   RUNG wire#powerrail
      Contact( "UpDown".UD_3.O_Motor_B )
      Coil( "Elevator3_B" )
   END_RUNG
   RUNG wire#powerrail
      Contact( "UpDown".UD_3.O_Motor_U )
      Coil( "Elevator3_U" )
   END_RUNG
   RUNG wire#powerrail
      Contact( "UpDown".UD_3.O_Motor_D )
      Coil( "Elevator3_D" )
   END_RUNG
   RUNG wire#powerrail
      Contact( "UpDown".UD_3.O_Motor_F )
      Coil( "Elevator3_F" )
   END_RUNG
   RUNG wire#powerrail
      Contact( "UpDown".UD_3.O_Motor_Slow )
      Coil( "Elevator3_Slow" )
   END_RUNG
   // the same network as SCL:
   "Elevator3_B" := "UpDown".UD_3.O_Motor_B;
   "Elevator3_U" := "UpDown".UD_3.O_Motor_U;
   "Elevator3_D" := "UpDown".UD_3.O_Motor_D;
   "Elevator3_F" := "UpDown".UD_3.O_Motor_F;
   "Elevator3_Slow" := "UpDown".UD_3.O_Motor_Slow;
END_REGION

REGION Network 6: Write Elevator 4
   RUNG wire#powerrail
      Contact( "UpDown".UD_4.O_Motor_B )
      Coil( "Elevator4_B" )
   END_RUNG
   RUNG wire#powerrail
      Contact( "UpDown".UD_4.O_Motor_U )
      Coil( "Elevator4_U" )
   END_RUNG
   RUNG wire#powerrail
      Contact( "UpDown".UD_4.O_Motor_D )
      Coil( "Elevator4_D" )
   END_RUNG
   RUNG wire#powerrail
      Contact( "UpDown".UD_4.O_Motor_F )
      Coil( "Elevator4_F" )
   END_RUNG
   RUNG wire#powerrail
      Contact( "UpDown".UD_4.O_Motor_Slow )
      Coil( "Elevator4_Slow" )
   END_RUNG
   // the same network as SCL:
   "Elevator4_B" := "UpDown".UD_4.O_Motor_B;
   "Elevator4_U" := "UpDown".UD_4.O_Motor_U;
   "Elevator4_D" := "UpDown".UD_4.O_Motor_D;
   "Elevator4_F" := "UpDown".UD_4.O_Motor_F;
   "Elevator4_Slow" := "UpDown".UD_4.O_Motor_Slow;
END_REGION

REGION Network 7: Write avoid 0
   RUNG wire#powerrail
      Contact( "Avoid".Av_0.Cnv_motor )
      Coil( "Srt_0_Connect" )
   END_RUNG
   RUNG wire#powerrail
      Contact( "Avoid".Av_0.Av.Srt[2].O_Motor_B )
      Coil( "Srt_0_B2" )
   END_RUNG
   RUNG wire#powerrail
      Contact( "Avoid".Av_0.Av.Srt[2].O_Motor_R )
      Coil( "Srt_0_R2" )
   END_RUNG
   RUNG wire#powerrail
      Contact( "Avoid".Av_0.Av.Srt[1].O_Motor_F )
      Coil( "Srt_0_F1" )
   END_RUNG
   RUNG wire#powerrail
      Contact( "Avoid".Av_0.Av.Srt[1].O_Motor_R )
      Coil( "Srt_0_R1" )
   END_RUNG
   // the same network as SCL:
   "Srt_0_Connect" := "Avoid".Av_0.Cnv_motor;
   "Srt_0_B2" := "Avoid".Av_0.Av.Srt[2].O_Motor_B;
   "Srt_0_R2" := "Avoid".Av_0.Av.Srt[2].O_Motor_R;
   "Srt_0_F1" := "Avoid".Av_0.Av.Srt[1].O_Motor_F;
   "Srt_0_R1" := "Avoid".Av_0.Av.Srt[1].O_Motor_R;
END_REGION

REGION Network 8: Write avoid 1to2
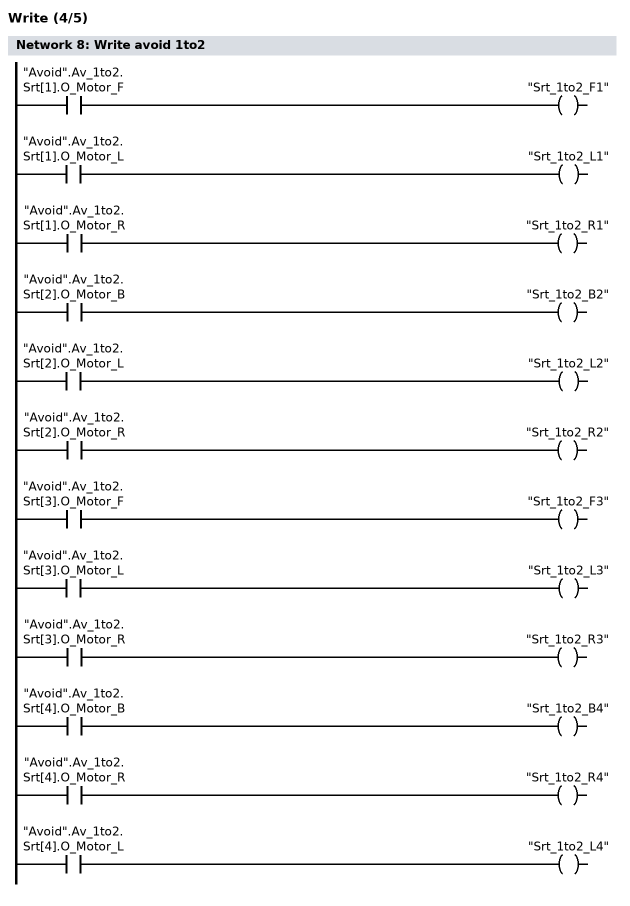
   RUNG wire#powerrail
      Contact( "Avoid".Av_1to2.Srt[1].O_Motor_F )
      Coil( "Srt_1to2_F1" )
   END_RUNG
   RUNG wire#powerrail
      Contact( "Avoid".Av_1to2.Srt[1].O_Motor_L )
      Coil( "Srt_1to2_L1" )
   END_RUNG
   RUNG wire#powerrail
      Contact( "Avoid".Av_1to2.Srt[1].O_Motor_R )
      Coil( "Srt_1to2_R1" )
   END_RUNG
   RUNG wire#powerrail
      Contact( "Avoid".Av_1to2.Srt[2].O_Motor_B )
      Coil( "Srt_1to2_B2" )
   END_RUNG
   RUNG wire#powerrail
      Contact( "Avoid".Av_1to2.Srt[2].O_Motor_L )
      Coil( "Srt_1to2_L2" )
   END_RUNG
   RUNG wire#powerrail
      Contact( "Avoid".Av_1to2.Srt[2].O_Motor_R )
      Coil( "Srt_1to2_R2" )
   END_RUNG
   RUNG wire#powerrail
      Contact( "Avoid".Av_1to2.Srt[3].O_Motor_F )
      Coil( "Srt_1to2_F3" )
   END_RUNG
   RUNG wire#powerrail
      Contact( "Avoid".Av_1to2.Srt[3].O_Motor_L )
      Coil( "Srt_1to2_L3" )
   END_RUNG
   RUNG wire#powerrail
      Contact( "Avoid".Av_1to2.Srt[3].O_Motor_R )
      Coil( "Srt_1to2_R3" )
   END_RUNG
   RUNG wire#powerrail
      Contact( "Avoid".Av_1to2.Srt[4].O_Motor_B )
      Coil( "Srt_1to2_B4" )
   END_RUNG
   RUNG wire#powerrail
      Contact( "Avoid".Av_1to2.Srt[4].O_Motor_R )
      Coil( "Srt_1to2_R4" )
   END_RUNG
   RUNG wire#powerrail
      Contact( "Avoid".Av_1to2.Srt[4].O_Motor_L )
      Coil( "Srt_1to2_L4" )
   END_RUNG
   // the same network as SCL:
   "Srt_1to2_F1" := "Avoid".Av_1to2.Srt[1].O_Motor_F;
   "Srt_1to2_L1" := "Avoid".Av_1to2.Srt[1].O_Motor_L;
   "Srt_1to2_R1" := "Avoid".Av_1to2.Srt[1].O_Motor_R;
   "Srt_1to2_B2" := "Avoid".Av_1to2.Srt[2].O_Motor_B;
   "Srt_1to2_L2" := "Avoid".Av_1to2.Srt[2].O_Motor_L;
   "Srt_1to2_R2" := "Avoid".Av_1to2.Srt[2].O_Motor_R;
   "Srt_1to2_F3" := "Avoid".Av_1to2.Srt[3].O_Motor_F;
   "Srt_1to2_L3" := "Avoid".Av_1to2.Srt[3].O_Motor_L;
   "Srt_1to2_R3" := "Avoid".Av_1to2.Srt[3].O_Motor_R;
   "Srt_1to2_B4" := "Avoid".Av_1to2.Srt[4].O_Motor_B;
   "Srt_1to2_R4" := "Avoid".Av_1to2.Srt[4].O_Motor_R;
   "Srt_1to2_L4" := "Avoid".Av_1to2.Srt[4].O_Motor_L;
END_REGION

REGION Network 9: Write avoid 2to3
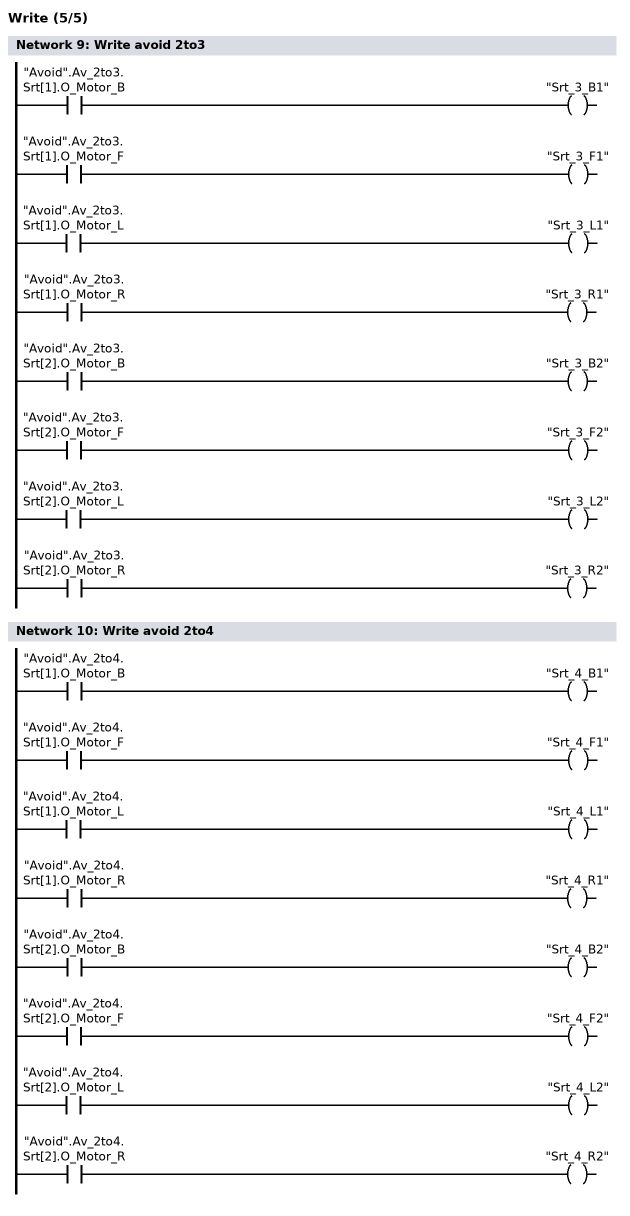
   RUNG wire#powerrail
      Contact( "Avoid".Av_2to3.Srt[1].O_Motor_B )
      Coil( "Srt_3_B1" )
   END_RUNG
   RUNG wire#powerrail
      Contact( "Avoid".Av_2to3.Srt[1].O_Motor_F )
      Coil( "Srt_3_F1" )
   END_RUNG
   RUNG wire#powerrail
      Contact( "Avoid".Av_2to3.Srt[1].O_Motor_L )
      Coil( "Srt_3_L1" )
   END_RUNG
   RUNG wire#powerrail
      Contact( "Avoid".Av_2to3.Srt[1].O_Motor_R )
      Coil( "Srt_3_R1" )
   END_RUNG
   RUNG wire#powerrail
      Contact( "Avoid".Av_2to3.Srt[2].O_Motor_B )
      Coil( "Srt_3_B2" )
   END_RUNG
   RUNG wire#powerrail
      Contact( "Avoid".Av_2to3.Srt[2].O_Motor_F )
      Coil( "Srt_3_F2" )
   END_RUNG
   RUNG wire#powerrail
      Contact( "Avoid".Av_2to3.Srt[2].O_Motor_L )
      Coil( "Srt_3_L2" )
   END_RUNG
   RUNG wire#powerrail
      Contact( "Avoid".Av_2to3.Srt[2].O_Motor_R )
      Coil( "Srt_3_R2" )
   END_RUNG
   // the same network as SCL:
   "Srt_3_B1" := "Avoid".Av_2to3.Srt[1].O_Motor_B;
   "Srt_3_F1" := "Avoid".Av_2to3.Srt[1].O_Motor_F;
   "Srt_3_L1" := "Avoid".Av_2to3.Srt[1].O_Motor_L;
   "Srt_3_R1" := "Avoid".Av_2to3.Srt[1].O_Motor_R;
   "Srt_3_B2" := "Avoid".Av_2to3.Srt[2].O_Motor_B;
   "Srt_3_F2" := "Avoid".Av_2to3.Srt[2].O_Motor_F;
   "Srt_3_L2" := "Avoid".Av_2to3.Srt[2].O_Motor_L;
   "Srt_3_R2" := "Avoid".Av_2to3.Srt[2].O_Motor_R;
END_REGION

REGION Network 10: Write avoid 2to4
   RUNG wire#powerrail
      Contact( "Avoid".Av_2to4.Srt[1].O_Motor_B )
      Coil( "Srt_4_B1" )
   END_RUNG
   RUNG wire#powerrail
      Contact( "Avoid".Av_2to4.Srt[1].O_Motor_F )
      Coil( "Srt_4_F1" )
   END_RUNG
   RUNG wire#powerrail
      Contact( "Avoid".Av_2to4.Srt[1].O_Motor_L )
      Coil( "Srt_4_L1" )
   END_RUNG
   RUNG wire#powerrail
      Contact( "Avoid".Av_2to4.Srt[1].O_Motor_R )
      Coil( "Srt_4_R1" )
   END_RUNG
   RUNG wire#powerrail
      Contact( "Avoid".Av_2to4.Srt[2].O_Motor_B )
      Coil( "Srt_4_B2" )
   END_RUNG
   RUNG wire#powerrail
      Contact( "Avoid".Av_2to4.Srt[2].O_Motor_F )
      Coil( "Srt_4_F2" )
   END_RUNG
   RUNG wire#powerrail
      Contact( "Avoid".Av_2to4.Srt[2].O_Motor_L )
      Coil( "Srt_4_L2" )
   END_RUNG
   RUNG wire#powerrail
      Contact( "Avoid".Av_2to4.Srt[2].O_Motor_R )
      Coil( "Srt_4_R2" )
   END_RUNG
   // the same network as SCL:
   "Srt_4_B1" := "Avoid".Av_2to4.Srt[1].O_Motor_B;
   "Srt_4_F1" := "Avoid".Av_2to4.Srt[1].O_Motor_F;
   "Srt_4_L1" := "Avoid".Av_2to4.Srt[1].O_Motor_L;
   "Srt_4_R1" := "Avoid".Av_2to4.Srt[1].O_Motor_R;
   "Srt_4_B2" := "Avoid".Av_2to4.Srt[2].O_Motor_B;
   "Srt_4_F2" := "Avoid".Av_2to4.Srt[2].O_Motor_F;
   "Srt_4_L2" := "Avoid".Av_2to4.Srt[2].O_Motor_L;
   "Srt_4_R2" := "Avoid".Av_2to4.Srt[2].O_Motor_R;
END_REGION
END_FUNCTION

FUNCTION "Link_Kepserver" : Void   // FC5, LAD
{ S7_Optimized_Access := 'TRUE' }
VERSION : 0.1
BEGIN

REGION Network 1: Cnv1d
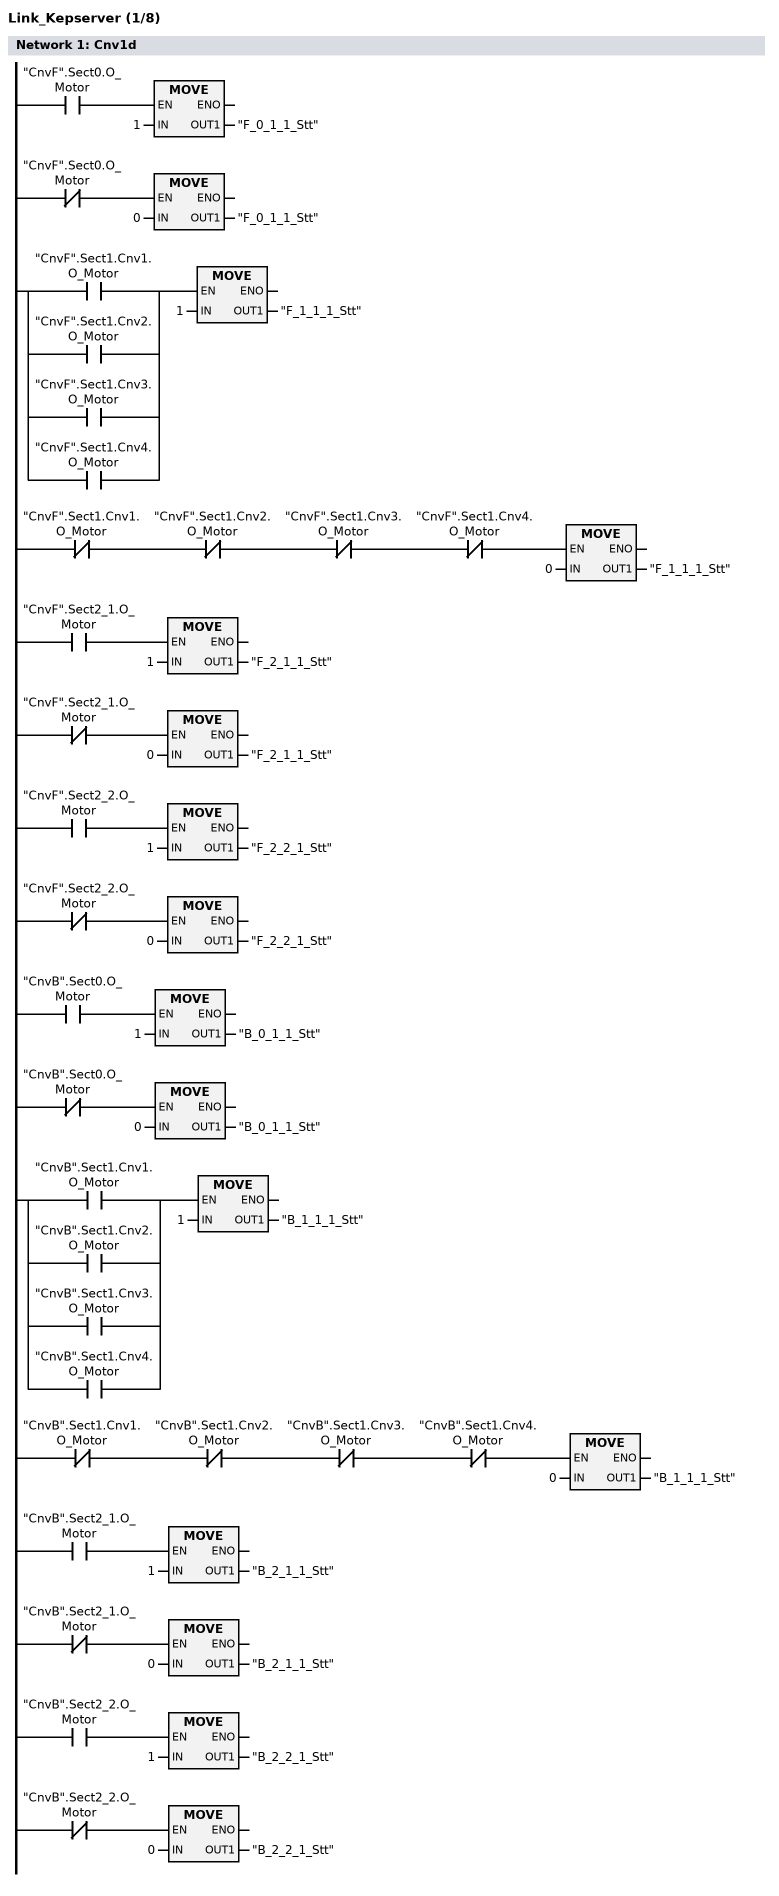
   RUNG wire#powerrail
      Contact( "CnvF".Sect0.O_Motor )
      Move(in := 1, out1 => "F_0_1_1_Stt")
   END_RUNG
   RUNG wire#powerrail
      I_Contact( "CnvF".Sect0.O_Motor )
      Move(in := 0, out1 => "F_0_1_1_Stt")
   END_RUNG
   RUNG wire#powerrail
      Contact( "CnvF".Sect1.Cnv1.O_Motor )
      wire#w1
      Move(in := 1, out1 => "F_1_1_1_Stt")
   END_RUNG
   RUNG wire#powerrail
      Contact( "CnvF".Sect1.Cnv2.O_Motor )
   END_RUNG wire#w1
   RUNG wire#powerrail
      Contact( "CnvF".Sect1.Cnv3.O_Motor )
   END_RUNG wire#w1
   RUNG wire#powerrail
      Contact( "CnvF".Sect1.Cnv4.O_Motor )
   END_RUNG wire#w1
   RUNG wire#powerrail
      I_Contact( "CnvF".Sect1.Cnv1.O_Motor )
      I_Contact( "CnvF".Sect1.Cnv2.O_Motor )
      I_Contact( "CnvF".Sect1.Cnv3.O_Motor )
      I_Contact( "CnvF".Sect1.Cnv4.O_Motor )
      Move(in := 0, out1 => "F_1_1_1_Stt")
   END_RUNG
   RUNG wire#powerrail
      Contact( "CnvF".Sect2_1.O_Motor )
      Move(in := 1, out1 => "F_2_1_1_Stt")
   END_RUNG
   RUNG wire#powerrail
      I_Contact( "CnvF".Sect2_1.O_Motor )
      Move(in := 0, out1 => "F_2_1_1_Stt")
   END_RUNG
   RUNG wire#powerrail
      Contact( "CnvF".Sect2_2.O_Motor )
      Move(in := 1, out1 => "F_2_2_1_Stt")
   END_RUNG
   RUNG wire#powerrail
      I_Contact( "CnvF".Sect2_2.O_Motor )
      Move(in := 0, out1 => "F_2_2_1_Stt")
   END_RUNG
   RUNG wire#powerrail
      Contact( "CnvB".Sect0.O_Motor )
      Move(in := 1, out1 => "B_0_1_1_Stt")
   END_RUNG
   RUNG wire#powerrail
      I_Contact( "CnvB".Sect0.O_Motor )
      Move(in := 0, out1 => "B_0_1_1_Stt")
   END_RUNG
   RUNG wire#powerrail
      Contact( "CnvB".Sect1.Cnv1.O_Motor )
      wire#w2
      Move(in := 1, out1 => "B_1_1_1_Stt")
   END_RUNG
   RUNG wire#powerrail
      Contact( "CnvB".Sect1.Cnv2.O_Motor )
   END_RUNG wire#w2
   RUNG wire#powerrail
      Contact( "CnvB".Sect1.Cnv3.O_Motor )
   END_RUNG wire#w2
   RUNG wire#powerrail
      Contact( "CnvB".Sect1.Cnv4.O_Motor )
   END_RUNG wire#w2
   RUNG wire#powerrail
      I_Contact( "CnvB".Sect1.Cnv1.O_Motor )
      I_Contact( "CnvB".Sect1.Cnv2.O_Motor )
      I_Contact( "CnvB".Sect1.Cnv3.O_Motor )
      I_Contact( "CnvB".Sect1.Cnv4.O_Motor )
      Move(in := 0, out1 => "B_1_1_1_Stt")
   END_RUNG
   RUNG wire#powerrail
      Contact( "CnvB".Sect2_1.O_Motor )
      Move(in := 1, out1 => "B_2_1_1_Stt")
   END_RUNG
   RUNG wire#powerrail
      I_Contact( "CnvB".Sect2_1.O_Motor )
      Move(in := 0, out1 => "B_2_1_1_Stt")
   END_RUNG
   RUNG wire#powerrail
      Contact( "CnvB".Sect2_2.O_Motor )
      Move(in := 1, out1 => "B_2_2_1_Stt")
   END_RUNG
   RUNG wire#powerrail
      I_Contact( "CnvB".Sect2_2.O_Motor )
      Move(in := 0, out1 => "B_2_2_1_Stt")
   END_RUNG
   // the same network as SCL:
   IF "CnvF".Sect0.O_Motor THEN "F_0_1_1_Stt" := 1; END_IF;
   IF NOT "CnvF".Sect0.O_Motor THEN "F_0_1_1_Stt" := 0; END_IF;
   IF "CnvF".Sect1.Cnv1.O_Motor OR "CnvF".Sect1.Cnv2.O_Motor OR "CnvF".Sect1.Cnv3.O_Motor OR "CnvF".Sect1.Cnv4.O_Motor THEN
       "F_1_1_1_Stt" := 1;
   END_IF;
   IF NOT "CnvF".Sect1.Cnv1.O_Motor AND NOT "CnvF".Sect1.Cnv2.O_Motor AND NOT "CnvF".Sect1.Cnv3.O_Motor AND NOT "CnvF".Sect1.Cnv4.O_Motor THEN
       "F_1_1_1_Stt" := 0;
   END_IF;
   IF "CnvF".Sect2_1.O_Motor THEN "F_2_1_1_Stt" := 1; END_IF;
   IF NOT "CnvF".Sect2_1.O_Motor THEN "F_2_1_1_Stt" := 0; END_IF;
   IF "CnvF".Sect2_2.O_Motor THEN "F_2_2_1_Stt" := 1; END_IF;
   IF NOT "CnvF".Sect2_2.O_Motor THEN "F_2_2_1_Stt" := 0; END_IF;
   IF "CnvB".Sect0.O_Motor THEN "B_0_1_1_Stt" := 1; END_IF;
   IF NOT "CnvB".Sect0.O_Motor THEN "B_0_1_1_Stt" := 0; END_IF;
   IF "CnvB".Sect1.Cnv1.O_Motor OR "CnvB".Sect1.Cnv2.O_Motor OR "CnvB".Sect1.Cnv3.O_Motor OR "CnvB".Sect1.Cnv4.O_Motor THEN
       "B_1_1_1_Stt" := 1;
   END_IF;
   IF NOT "CnvB".Sect1.Cnv1.O_Motor AND NOT "CnvB".Sect1.Cnv2.O_Motor AND NOT "CnvB".Sect1.Cnv3.O_Motor AND NOT "CnvB".Sect1.Cnv4.O_Motor THEN
       "B_1_1_1_Stt" := 0;
   END_IF;
   IF "CnvB".Sect2_1.O_Motor THEN "B_2_1_1_Stt" := 1; END_IF;
   IF NOT "CnvB".Sect2_1.O_Motor THEN "B_2_1_1_Stt" := 0; END_IF;
   IF "CnvB".Sect2_2.O_Motor THEN "B_2_2_1_Stt" := 1; END_IF;
   IF NOT "CnvB".Sect2_2.O_Motor THEN "B_2_2_1_Stt" := 0; END_IF;
END_REGION

REGION Network 2: Cnv2d
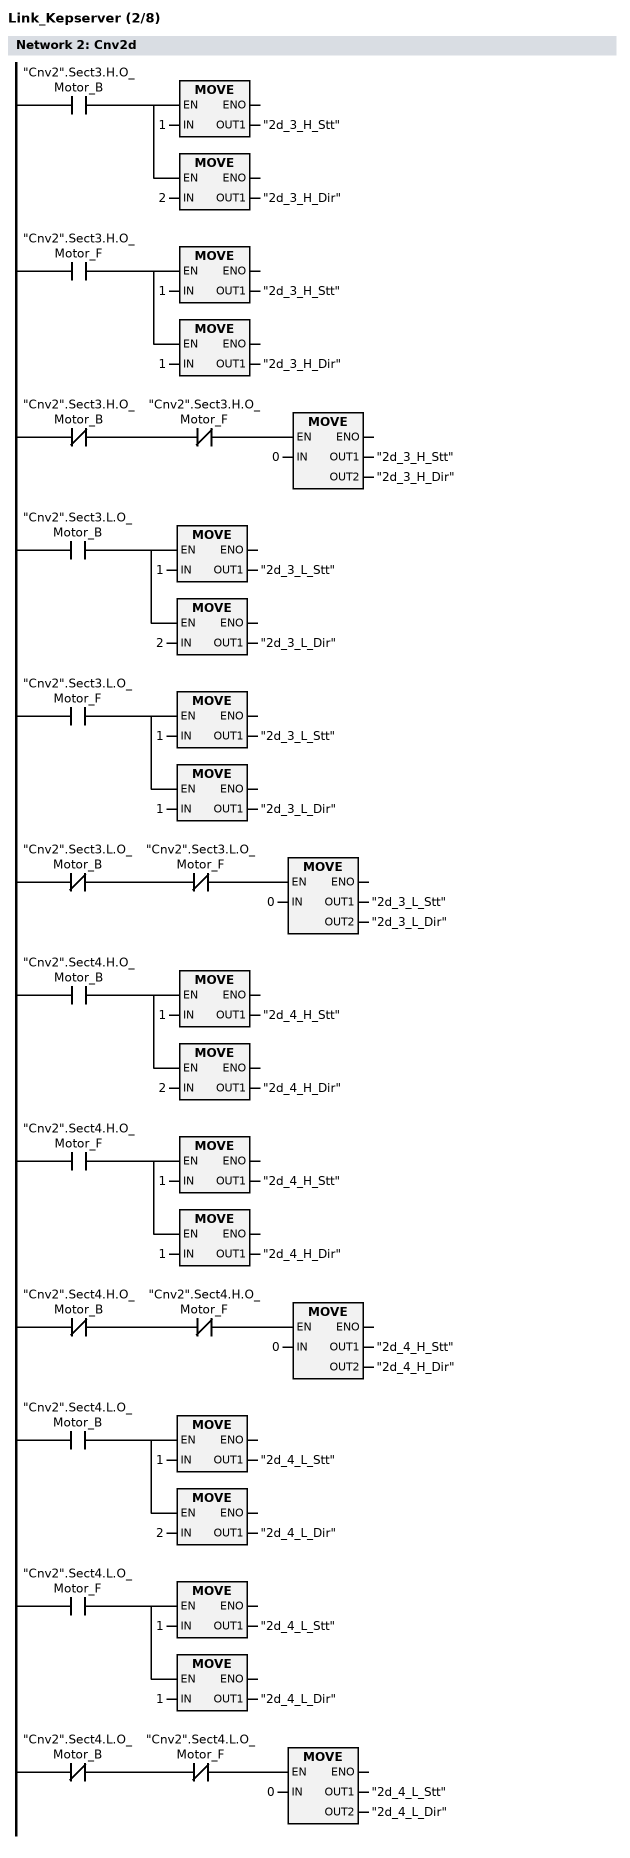
   RUNG wire#powerrail
      Contact( "Cnv2".Sect3.H.O_Motor_B )
      wire#w1
      Move(in := 1, out1 => "2d_3_H_Stt")
   END_RUNG
   RUNG wire#w1
      Move(in := 2, out1 => "2d_3_H_Dir")
   END_RUNG
   RUNG wire#powerrail
      Contact( "Cnv2".Sect3.H.O_Motor_F )
      wire#w2
      Move(in := 1, out1 => "2d_3_H_Stt")
   END_RUNG
   RUNG wire#w2
      Move(in := 1, out1 => "2d_3_H_Dir")
   END_RUNG
   RUNG wire#powerrail
      I_Contact( "Cnv2".Sect3.H.O_Motor_B )
      I_Contact( "Cnv2".Sect3.H.O_Motor_F )
      Move(in := 0, out1 => "2d_3_H_Stt", out2 => "2d_3_H_Dir")
   END_RUNG
   RUNG wire#powerrail
      Contact( "Cnv2".Sect3.L.O_Motor_B )
      wire#w3
      Move(in := 1, out1 => "2d_3_L_Stt")
   END_RUNG
   RUNG wire#w3
      Move(in := 2, out1 => "2d_3_L_Dir")
   END_RUNG
   RUNG wire#powerrail
      Contact( "Cnv2".Sect3.L.O_Motor_F )
      wire#w4
      Move(in := 1, out1 => "2d_3_L_Stt")
   END_RUNG
   RUNG wire#w4
      Move(in := 1, out1 => "2d_3_L_Dir")
   END_RUNG
   RUNG wire#powerrail
      I_Contact( "Cnv2".Sect3.L.O_Motor_B )
      I_Contact( "Cnv2".Sect3.L.O_Motor_F )
      Move(in := 0, out1 => "2d_3_L_Stt", out2 => "2d_3_L_Dir")
   END_RUNG
   RUNG wire#powerrail
      Contact( "Cnv2".Sect4.H.O_Motor_B )
      wire#w5
      Move(in := 1, out1 => "2d_4_H_Stt")
   END_RUNG
   RUNG wire#w5
      Move(in := 2, out1 => "2d_4_H_Dir")
   END_RUNG
   RUNG wire#powerrail
      Contact( "Cnv2".Sect4.H.O_Motor_F )
      wire#w6
      Move(in := 1, out1 => "2d_4_H_Stt")
   END_RUNG
   RUNG wire#w6
      Move(in := 1, out1 => "2d_4_H_Dir")
   END_RUNG
   RUNG wire#powerrail
      I_Contact( "Cnv2".Sect4.H.O_Motor_B )
      I_Contact( "Cnv2".Sect4.H.O_Motor_F )
      Move(in := 0, out1 => "2d_4_H_Stt", out2 => "2d_4_H_Dir")
   END_RUNG
   RUNG wire#powerrail
      Contact( "Cnv2".Sect4.L.O_Motor_B )
      wire#w7
      Move(in := 1, out1 => "2d_4_L_Stt")
   END_RUNG
   RUNG wire#w7
      Move(in := 2, out1 => "2d_4_L_Dir")
   END_RUNG
   RUNG wire#powerrail
      Contact( "Cnv2".Sect4.L.O_Motor_F )
      wire#w8
      Move(in := 1, out1 => "2d_4_L_Stt")
   END_RUNG
   RUNG wire#w8
      Move(in := 1, out1 => "2d_4_L_Dir")
   END_RUNG
   RUNG wire#powerrail
      I_Contact( "Cnv2".Sect4.L.O_Motor_B )
      I_Contact( "Cnv2".Sect4.L.O_Motor_F )
      Move(in := 0, out1 => "2d_4_L_Stt", out2 => "2d_4_L_Dir")
   END_RUNG
   // the same network as SCL:
   IF "Cnv2".Sect3.H.O_Motor_B THEN
       "2d_3_H_Stt" := 1;
       "2d_3_H_Dir" := 2;
   END_IF;
   IF "Cnv2".Sect3.H.O_Motor_F THEN
       "2d_3_H_Stt" := 1;
       "2d_3_H_Dir" := 1;
   END_IF;
   IF NOT "Cnv2".Sect3.H.O_Motor_B AND NOT "Cnv2".Sect3.H.O_Motor_F THEN
       "2d_3_H_Stt" := 0;
       "2d_3_H_Dir" := 0;
   END_IF;
   IF "Cnv2".Sect3.L.O_Motor_B THEN
       "2d_3_L_Stt" := 1;
       "2d_3_L_Dir" := 2;
   END_IF;
   IF "Cnv2".Sect3.L.O_Motor_F THEN
       "2d_3_L_Stt" := 1;
       "2d_3_L_Dir" := 1;
   END_IF;
   IF NOT "Cnv2".Sect3.L.O_Motor_B AND NOT "Cnv2".Sect3.L.O_Motor_F THEN
       "2d_3_L_Stt" := 0;
       "2d_3_L_Dir" := 0;
   END_IF;
   IF "Cnv2".Sect4.H.O_Motor_B THEN
       "2d_4_H_Stt" := 1;
       "2d_4_H_Dir" := 2;
   END_IF;
   IF "Cnv2".Sect4.H.O_Motor_F THEN
       "2d_4_H_Stt" := 1;
       "2d_4_H_Dir" := 1;
   END_IF;
   IF NOT "Cnv2".Sect4.H.O_Motor_B AND NOT "Cnv2".Sect4.H.O_Motor_F THEN
       "2d_4_H_Stt" := 0;
       "2d_4_H_Dir" := 0;
   END_IF;
   IF "Cnv2".Sect4.L.O_Motor_B THEN
       "2d_4_L_Stt" := 1;
       "2d_4_L_Dir" := 2;
   END_IF;
   IF "Cnv2".Sect4.L.O_Motor_F THEN
       "2d_4_L_Stt" := 1;
       "2d_4_L_Dir" := 1;
   END_IF;
   IF NOT "Cnv2".Sect4.L.O_Motor_B AND NOT "Cnv2".Sect4.L.O_Motor_F THEN
       "2d_4_L_Stt" := 0;
       "2d_4_L_Dir" := 0;
   END_IF;
END_REGION

